REGION Network 13: HOPPER TEMPERATURE LINE 2
   RUNG wire#powerrail
      Contact( #HMI_INPUT_MAN_MODE )
      wire#w1
      "FC21020_FEEDER_SCALING"(DINT_INPUT_VALUE := 0, REAL_INPUT_VALUE := #"iHMI_Values Setpoints".HopperTempNominalLine2, DINT_TO_REAL := false, REAL_TRANSFORM_FOR_FEEDER := true, OUTPUT_VALUE_PLC => #oPLC_Aux.o_rHopperTempNominal_Line2, OUTPUT_VALUE_FEEDER => #ioPowder_Feeder_Unit_In_Out.Outputs."PF Setpoints, Warnings and Alarms".o_rHopperTempNominal_Line2)
   END_RUNG
   RUNG wire#w1
      Not()
      "FC21020_FEEDER_SCALING"(DINT_INPUT_VALUE := 0, REAL_INPUT_VALUE := #"iCNC_Values Setpoints".HopperTempNominalLine2, DINT_TO_REAL := false, REAL_TRANSFORM_FOR_FEEDER := true, OUTPUT_VALUE_PLC => #oPLC_Aux.o_rHopperTempNominal_Line2, OUTPUT_VALUE_FEEDER => #ioPowder_Feeder_Unit_In_Out.Outputs."PF Setpoints, Warnings and Alarms".o_rHopperTempNominal_Line2)
   END_RUNG
   // the same network as SCL:
   IF #HMI_INPUT_MAN_MODE THEN
       "FC21020_FEEDER_SCALING"(DINT_INPUT_VALUE := 0,
                               REAL_INPUT_VALUE := #"iHMI_Values Setpoints".HopperTempNominalLine2,
                               DINT_TO_REAL := false,
                               REAL_TRANSFORM_FOR_FEEDER := true,
                               OUTPUT_VALUE_PLC => #oPLC_Aux.o_rHopperTempNominal_Line2,
                               OUTPUT_VALUE_FEEDER => #ioPowder_Feeder_Unit_In_Out.Outputs."PF Setpoints, Warnings and Alarms".o_rHopperTempNominal_Line2);
   END_IF;
   IF NOT #HMI_INPUT_MAN_MODE THEN
       "FC21020_FEEDER_SCALING"(DINT_INPUT_VALUE := 0,
                               REAL_INPUT_VALUE := #"iCNC_Values Setpoints".HopperTempNominalLine2,
                               DINT_TO_REAL := false,
                               REAL_TRANSFORM_FOR_FEEDER := true,
                               OUTPUT_VALUE_PLC => #oPLC_Aux.o_rHopperTempNominal_Line2,
                               OUTPUT_VALUE_FEEDER => #ioPowder_Feeder_Unit_In_Out.Outputs."PF Setpoints, Warnings and Alarms".o_rHopperTempNominal_Line2);
   END_IF;
END_REGION

REGION Network 14: COMMUNICATION IS RUNNING
   RUNG wire#powerrail
      Contact( "M_ONE" )
      wire#w1
      Coil( #ioPowder_Feeder_Unit_In_Out.Outputs.o_fCommunicationOk_Line1 )
   END_RUNG
   RUNG wire#w1
      Coil( #ioPowder_Feeder_Unit_In_Out.Outputs.o_fCommunicationOk_Line2 )
   END_RUNG
   // the same network as SCL:
   #ioPowder_Feeder_Unit_In_Out.Outputs.o_fCommunicationOk_Line1 := "M_ONE";
   #ioPowder_Feeder_Unit_In_Out.Outputs.o_fCommunicationOk_Line2 := "M_ONE";
END_REGION

REGION Network 15: VOLUMETRIC MODE ON
   // Volumetric Mode On = 1 for Twin 150
   // Gravimetric Mode - n/a for Twin 150
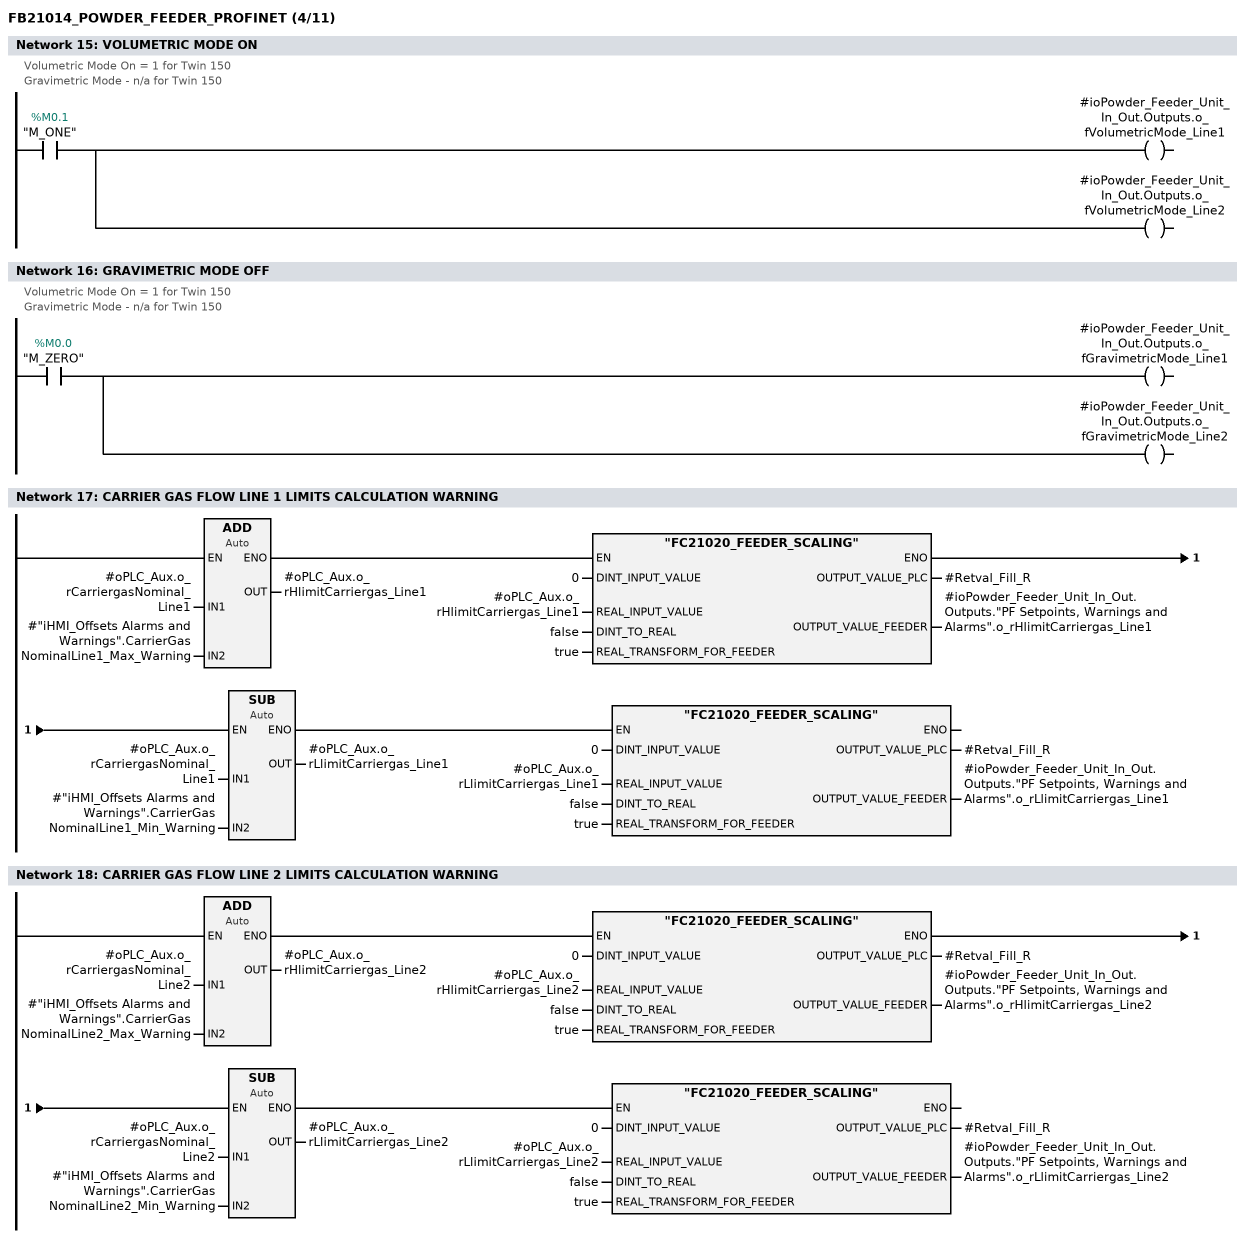
   RUNG wire#powerrail
      Contact( "M_ONE" )
      wire#w1
      Coil( #ioPowder_Feeder_Unit_In_Out.Outputs.o_fVolumetricMode_Line1 )
   END_RUNG
   RUNG wire#w1
      Coil( #ioPowder_Feeder_Unit_In_Out.Outputs.o_fVolumetricMode_Line2 )
   END_RUNG
   // the same network as SCL:
   #ioPowder_Feeder_Unit_In_Out.Outputs.o_fVolumetricMode_Line1 := "M_ONE";
   #ioPowder_Feeder_Unit_In_Out.Outputs.o_fVolumetricMode_Line2 := "M_ONE";
END_REGION

REGION Network 16: GRAVIMETRIC MODE OFF
   // Volumetric Mode On = 1 for Twin 150
   // Gravimetric Mode - n/a for Twin 150
   RUNG wire#powerrail
      Contact( "M_ZERO" )
      wire#w1
      Coil( #ioPowder_Feeder_Unit_In_Out.Outputs.o_fGravimetricMode_Line1 )
   END_RUNG
   RUNG wire#w1
      Coil( #ioPowder_Feeder_Unit_In_Out.Outputs.o_fGravimetricMode_Line2 )
   END_RUNG
   // the same network as SCL:
   #ioPowder_Feeder_Unit_In_Out.Outputs.o_fGravimetricMode_Line1 := "M_ZERO";
   #ioPowder_Feeder_Unit_In_Out.Outputs.o_fGravimetricMode_Line2 := "M_ZERO";
END_REGION

REGION Network 17: CARRIER GAS FLOW LINE 1 LIMITS CALCULATION WARNING
   RUNG wire#powerrail
      Add(in1 := #oPLC_Aux.o_rCarriergasNominal_Line1, in2 := #"iHMI_Offsets Alarms and Warnings".CarrierGasNominalLine1_Max_Warning, out => #oPLC_Aux.o_rHlimitCarriergas_Line1)
      "FC21020_FEEDER_SCALING"(DINT_INPUT_VALUE := 0, REAL_INPUT_VALUE := #oPLC_Aux.o_rHlimitCarriergas_Line1, DINT_TO_REAL := false, REAL_TRANSFORM_FOR_FEEDER := true, OUTPUT_VALUE_PLC => #Retval_Fill_R, OUTPUT_VALUE_FEEDER => #ioPowder_Feeder_Unit_In_Out.Outputs."PF Setpoints, Warnings and Alarms".o_rHlimitCarriergas_Line1)
      Sub(in1 := #oPLC_Aux.o_rCarriergasNominal_Line1, in2 := #"iHMI_Offsets Alarms and Warnings".CarrierGasNominalLine1_Min_Warning, out => #oPLC_Aux.o_rLlimitCarriergas_Line1)
      "FC21020_FEEDER_SCALING"(DINT_INPUT_VALUE := 0, REAL_INPUT_VALUE := #oPLC_Aux.o_rLlimitCarriergas_Line1, DINT_TO_REAL := false, REAL_TRANSFORM_FOR_FEEDER := true, OUTPUT_VALUE_PLC => #Retval_Fill_R, OUTPUT_VALUE_FEEDER => #ioPowder_Feeder_Unit_In_Out.Outputs."PF Setpoints, Warnings and Alarms".o_rLlimitCarriergas_Line1)
   END_RUNG
   // the same network as SCL:
   #oPLC_Aux.o_rHlimitCarriergas_Line1 := #oPLC_Aux.o_rCarriergasNominal_Line1 + #"iHMI_Offsets Alarms and Warnings".CarrierGasNominalLine1_Max_Warning;
   "FC21020_FEEDER_SCALING"(DINT_INPUT_VALUE := 0,
                           REAL_INPUT_VALUE := #oPLC_Aux.o_rHlimitCarriergas_Line1,
                           DINT_TO_REAL := false,
                           REAL_TRANSFORM_FOR_FEEDER := true,
                           OUTPUT_VALUE_PLC => #Retval_Fill_R,
                           OUTPUT_VALUE_FEEDER => #ioPowder_Feeder_Unit_In_Out.Outputs."PF Setpoints, Warnings and Alarms".o_rHlimitCarriergas_Line1,
                           ENO => #_w1);
   IF #_w1 THEN
       #oPLC_Aux.o_rLlimitCarriergas_Line1 := #oPLC_Aux.o_rCarriergasNominal_Line1 - #"iHMI_Offsets Alarms and Warnings".CarrierGasNominalLine1_Min_Warning;
       "FC21020_FEEDER_SCALING"(DINT_INPUT_VALUE := 0,
                               REAL_INPUT_VALUE := #oPLC_Aux.o_rLlimitCarriergas_Line1,
                               DINT_TO_REAL := false,
                               REAL_TRANSFORM_FOR_FEEDER := true,
                               OUTPUT_VALUE_PLC => #Retval_Fill_R,
                               OUTPUT_VALUE_FEEDER => #ioPowder_Feeder_Unit_In_Out.Outputs."PF Setpoints, Warnings and Alarms".o_rLlimitCarriergas_Line1);
   END_IF;
END_REGION

REGION Network 18: CARRIER GAS FLOW LINE 2 LIMITS CALCULATION WARNING
   RUNG wire#powerrail
      Add(in1 := #oPLC_Aux.o_rCarriergasNominal_Line2, in2 := #"iHMI_Offsets Alarms and Warnings".CarrierGasNominalLine2_Max_Warning, out => #oPLC_Aux.o_rHlimitCarriergas_Line2)
      "FC21020_FEEDER_SCALING"(DINT_INPUT_VALUE := 0, REAL_INPUT_VALUE := #oPLC_Aux.o_rHlimitCarriergas_Line2, DINT_TO_REAL := false, REAL_TRANSFORM_FOR_FEEDER := true, OUTPUT_VALUE_PLC => #Retval_Fill_R, OUTPUT_VALUE_FEEDER => #ioPowder_Feeder_Unit_In_Out.Outputs."PF Setpoints, Warnings and Alarms".o_rHlimitCarriergas_Line2)
      Sub(in1 := #oPLC_Aux.o_rCarriergasNominal_Line2, in2 := #"iHMI_Offsets Alarms and Warnings".CarrierGasNominalLine2_Min_Warning, out => #oPLC_Aux.o_rLlimitCarriergas_Line2)
      "FC21020_FEEDER_SCALING"(DINT_INPUT_VALUE := 0, REAL_INPUT_VALUE := #oPLC_Aux.o_rLlimitCarriergas_Line2, DINT_TO_REAL := false, REAL_TRANSFORM_FOR_FEEDER := true, OUTPUT_VALUE_PLC => #Retval_Fill_R, OUTPUT_VALUE_FEEDER => #ioPowder_Feeder_Unit_In_Out.Outputs."PF Setpoints, Warnings and Alarms".o_rLlimitCarriergas_Line2)
   END_RUNG
   // the same network as SCL:
   #oPLC_Aux.o_rHlimitCarriergas_Line2 := #oPLC_Aux.o_rCarriergasNominal_Line2 + #"iHMI_Offsets Alarms and Warnings".CarrierGasNominalLine2_Max_Warning;
   "FC21020_FEEDER_SCALING"(DINT_INPUT_VALUE := 0,
                           REAL_INPUT_VALUE := #oPLC_Aux.o_rHlimitCarriergas_Line2,
                           DINT_TO_REAL := false,
                           REAL_TRANSFORM_FOR_FEEDER := true,
                           OUTPUT_VALUE_PLC => #Retval_Fill_R,
                           OUTPUT_VALUE_FEEDER => #ioPowder_Feeder_Unit_In_Out.Outputs."PF Setpoints, Warnings and Alarms".o_rHlimitCarriergas_Line2,
                           ENO => #_w1);
   IF #_w1 THEN
       #oPLC_Aux.o_rLlimitCarriergas_Line2 := #oPLC_Aux.o_rCarriergasNominal_Line2 - #"iHMI_Offsets Alarms and Warnings".CarrierGasNominalLine2_Min_Warning;
       "FC21020_FEEDER_SCALING"(DINT_INPUT_VALUE := 0,
                               REAL_INPUT_VALUE := #oPLC_Aux.o_rLlimitCarriergas_Line2,
                               DINT_TO_REAL := false,
                               REAL_TRANSFORM_FOR_FEEDER := true,
                               OUTPUT_VALUE_PLC => #Retval_Fill_R,
                               OUTPUT_VALUE_FEEDER => #ioPowder_Feeder_Unit_In_Out.Outputs."PF Setpoints, Warnings and Alarms".o_rLlimitCarriergas_Line2);
   END_IF;
END_REGION

REGION Network 19: CARRIER GAS FLOW LINE 1 LIMITS CALCULATION ALARM
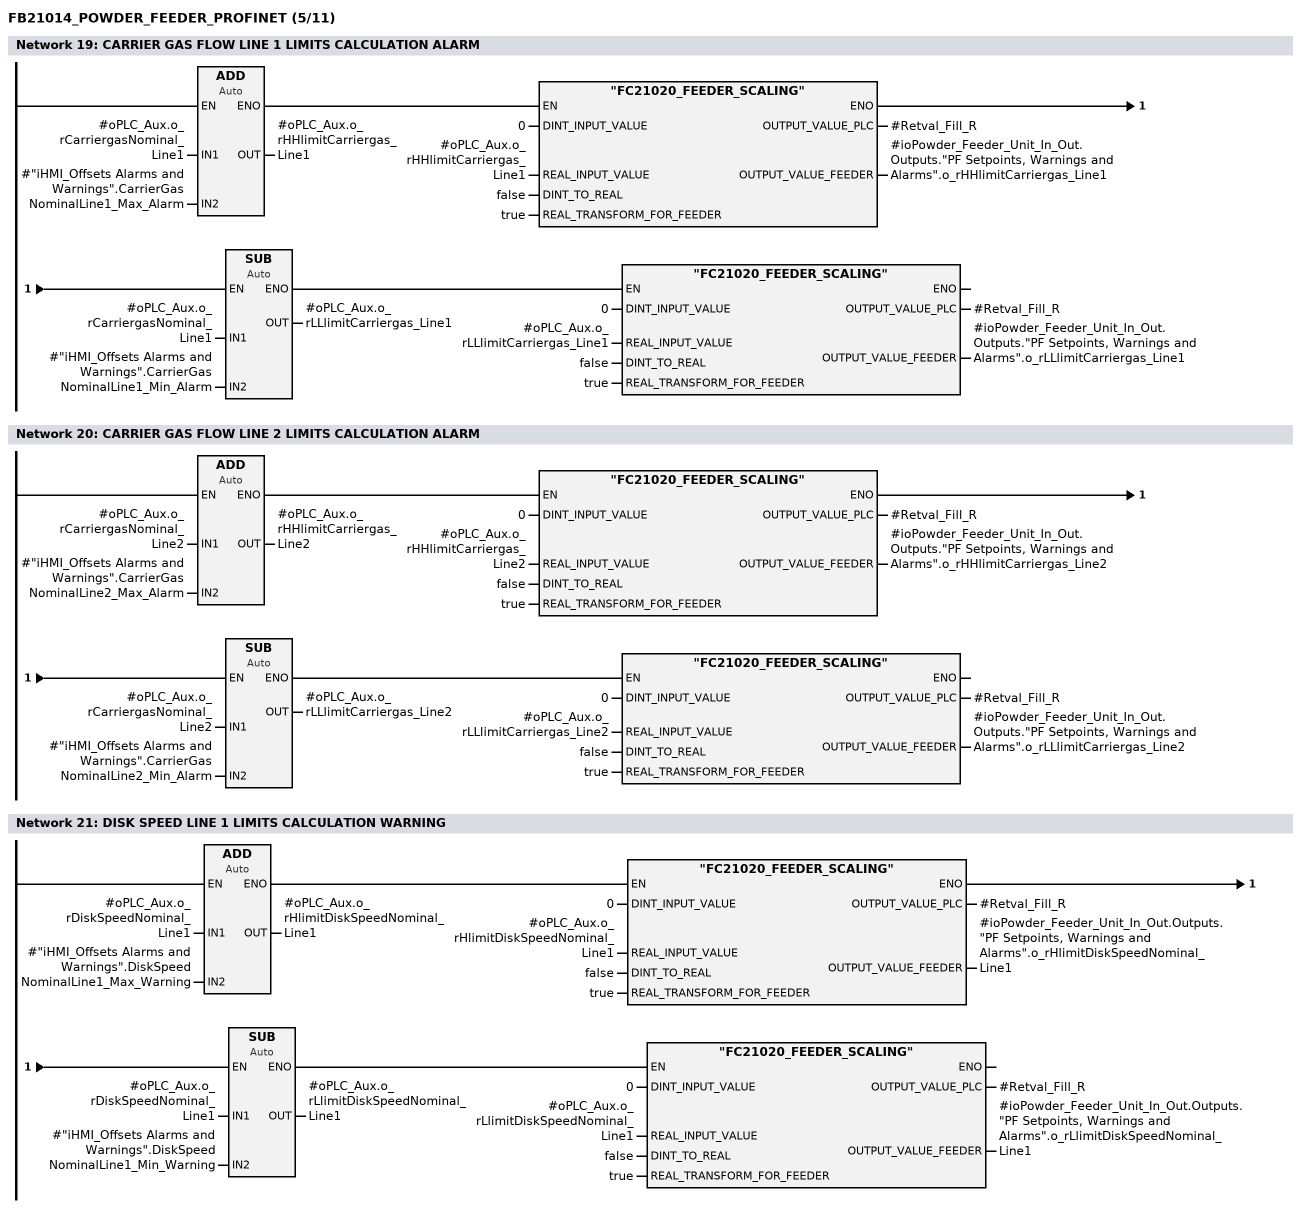
   RUNG wire#powerrail
      Add(in1 := #oPLC_Aux.o_rCarriergasNominal_Line1, in2 := #"iHMI_Offsets Alarms and Warnings".CarrierGasNominalLine1_Max_Alarm, out => #oPLC_Aux.o_rHHlimitCarriergas_Line1)
      "FC21020_FEEDER_SCALING"(DINT_INPUT_VALUE := 0, REAL_INPUT_VALUE := #oPLC_Aux.o_rHHlimitCarriergas_Line1, DINT_TO_REAL := false, REAL_TRANSFORM_FOR_FEEDER := true, OUTPUT_VALUE_PLC => #Retval_Fill_R, OUTPUT_VALUE_FEEDER => #ioPowder_Feeder_Unit_In_Out.Outputs."PF Setpoints, Warnings and Alarms".o_rHHlimitCarriergas_Line1)
      Sub(in1 := #oPLC_Aux.o_rCarriergasNominal_Line1, in2 := #"iHMI_Offsets Alarms and Warnings".CarrierGasNominalLine1_Min_Alarm, out => #oPLC_Aux.o_rLLlimitCarriergas_Line1)
      "FC21020_FEEDER_SCALING"(DINT_INPUT_VALUE := 0, REAL_INPUT_VALUE := #oPLC_Aux.o_rLLlimitCarriergas_Line1, DINT_TO_REAL := false, REAL_TRANSFORM_FOR_FEEDER := true, OUTPUT_VALUE_PLC => #Retval_Fill_R, OUTPUT_VALUE_FEEDER => #ioPowder_Feeder_Unit_In_Out.Outputs."PF Setpoints, Warnings and Alarms".o_rLLlimitCarriergas_Line1)
   END_RUNG
   // the same network as SCL:
   #oPLC_Aux.o_rHHlimitCarriergas_Line1 := #oPLC_Aux.o_rCarriergasNominal_Line1 + #"iHMI_Offsets Alarms and Warnings".CarrierGasNominalLine1_Max_Alarm;
   "FC21020_FEEDER_SCALING"(DINT_INPUT_VALUE := 0,
                           REAL_INPUT_VALUE := #oPLC_Aux.o_rHHlimitCarriergas_Line1,
                           DINT_TO_REAL := false,
                           REAL_TRANSFORM_FOR_FEEDER := true,
                           OUTPUT_VALUE_PLC => #Retval_Fill_R,
                           OUTPUT_VALUE_FEEDER => #ioPowder_Feeder_Unit_In_Out.Outputs."PF Setpoints, Warnings and Alarms".o_rHHlimitCarriergas_Line1,
                           ENO => #_w1);
   IF #_w1 THEN
       #oPLC_Aux.o_rLLlimitCarriergas_Line1 := #oPLC_Aux.o_rCarriergasNominal_Line1 - #"iHMI_Offsets Alarms and Warnings".CarrierGasNominalLine1_Min_Alarm;
       "FC21020_FEEDER_SCALING"(DINT_INPUT_VALUE := 0,
                               REAL_INPUT_VALUE := #oPLC_Aux.o_rLLlimitCarriergas_Line1,
                               DINT_TO_REAL := false,
                               REAL_TRANSFORM_FOR_FEEDER := true,
                               OUTPUT_VALUE_PLC => #Retval_Fill_R,
                               OUTPUT_VALUE_FEEDER => #ioPowder_Feeder_Unit_In_Out.Outputs."PF Setpoints, Warnings and Alarms".o_rLLlimitCarriergas_Line1);
   END_IF;
END_REGION

REGION Network 20: CARRIER GAS FLOW LINE 2 LIMITS CALCULATION ALARM
   RUNG wire#powerrail
      Add(in1 := #oPLC_Aux.o_rCarriergasNominal_Line2, in2 := #"iHMI_Offsets Alarms and Warnings".CarrierGasNominalLine2_Max_Alarm, out => #oPLC_Aux.o_rHHlimitCarriergas_Line2)
      "FC21020_FEEDER_SCALING"(DINT_INPUT_VALUE := 0, REAL_INPUT_VALUE := #oPLC_Aux.o_rHHlimitCarriergas_Line2, DINT_TO_REAL := false, REAL_TRANSFORM_FOR_FEEDER := true, OUTPUT_VALUE_PLC => #Retval_Fill_R, OUTPUT_VALUE_FEEDER => #ioPowder_Feeder_Unit_In_Out.Outputs."PF Setpoints, Warnings and Alarms".o_rHHlimitCarriergas_Line2)
      Sub(in1 := #oPLC_Aux.o_rCarriergasNominal_Line2, in2 := #"iHMI_Offsets Alarms and Warnings".CarrierGasNominalLine2_Min_Alarm, out => #oPLC_Aux.o_rLLlimitCarriergas_Line2)
      "FC21020_FEEDER_SCALING"(DINT_INPUT_VALUE := 0, REAL_INPUT_VALUE := #oPLC_Aux.o_rLLlimitCarriergas_Line2, DINT_TO_REAL := false, REAL_TRANSFORM_FOR_FEEDER := true, OUTPUT_VALUE_PLC => #Retval_Fill_R, OUTPUT_VALUE_FEEDER => #ioPowder_Feeder_Unit_In_Out.Outputs."PF Setpoints, Warnings and Alarms".o_rLLlimitCarriergas_Line2)
   END_RUNG
   // the same network as SCL:
   #oPLC_Aux.o_rHHlimitCarriergas_Line2 := #oPLC_Aux.o_rCarriergasNominal_Line2 + #"iHMI_Offsets Alarms and Warnings".CarrierGasNominalLine2_Max_Alarm;
   "FC21020_FEEDER_SCALING"(DINT_INPUT_VALUE := 0,
                           REAL_INPUT_VALUE := #oPLC_Aux.o_rHHlimitCarriergas_Line2,
                           DINT_TO_REAL := false,
                           REAL_TRANSFORM_FOR_FEEDER := true,
                           OUTPUT_VALUE_PLC => #Retval_Fill_R,
                           OUTPUT_VALUE_FEEDER => #ioPowder_Feeder_Unit_In_Out.Outputs."PF Setpoints, Warnings and Alarms".o_rHHlimitCarriergas_Line2,
                           ENO => #_w1);
   IF #_w1 THEN
       #oPLC_Aux.o_rLLlimitCarriergas_Line2 := #oPLC_Aux.o_rCarriergasNominal_Line2 - #"iHMI_Offsets Alarms and Warnings".CarrierGasNominalLine2_Min_Alarm;
       "FC21020_FEEDER_SCALING"(DINT_INPUT_VALUE := 0,
                               REAL_INPUT_VALUE := #oPLC_Aux.o_rLLlimitCarriergas_Line2,
                               DINT_TO_REAL := false,
                               REAL_TRANSFORM_FOR_FEEDER := true,
                               OUTPUT_VALUE_PLC => #Retval_Fill_R,
                               OUTPUT_VALUE_FEEDER => #ioPowder_Feeder_Unit_In_Out.Outputs."PF Setpoints, Warnings and Alarms".o_rLLlimitCarriergas_Line2);
   END_IF;
END_REGION

REGION Network 21: DISK SPEED LINE 1 LIMITS CALCULATION WARNING
   RUNG wire#powerrail
      Add(in1 := #oPLC_Aux.o_rDiskSpeedNominal_Line1, in2 := #"iHMI_Offsets Alarms and Warnings".DiskSpeedNominalLine1_Max_Warning, out => #oPLC_Aux.o_rHlimitDiskSpeedNominal_Line1)
      "FC21020_FEEDER_SCALING"(DINT_INPUT_VALUE := 0, REAL_INPUT_VALUE := #oPLC_Aux.o_rHlimitDiskSpeedNominal_Line1, DINT_TO_REAL := false, REAL_TRANSFORM_FOR_FEEDER := true, OUTPUT_VALUE_PLC => #Retval_Fill_R, OUTPUT_VALUE_FEEDER => #ioPowder_Feeder_Unit_In_Out.Outputs."PF Setpoints, Warnings and Alarms".o_rHlimitDiskSpeedNominal_Line1)
      Sub(in1 := #oPLC_Aux.o_rDiskSpeedNominal_Line1, in2 := #"iHMI_Offsets Alarms and Warnings".DiskSpeedNominalLine1_Min_Warning, out => #oPLC_Aux.o_rLlimitDiskSpeedNominal_Line1)
      "FC21020_FEEDER_SCALING"(DINT_INPUT_VALUE := 0, REAL_INPUT_VALUE := #oPLC_Aux.o_rLlimitDiskSpeedNominal_Line1, DINT_TO_REAL := false, REAL_TRANSFORM_FOR_FEEDER := true, OUTPUT_VALUE_PLC => #Retval_Fill_R, OUTPUT_VALUE_FEEDER => #ioPowder_Feeder_Unit_In_Out.Outputs."PF Setpoints, Warnings and Alarms".o_rLlimitDiskSpeedNominal_Line1)
   END_RUNG
   // the same network as SCL:
   #oPLC_Aux.o_rHlimitDiskSpeedNominal_Line1 := #oPLC_Aux.o_rDiskSpeedNominal_Line1 + #"iHMI_Offsets Alarms and Warnings".DiskSpeedNominalLine1_Max_Warning;
   "FC21020_FEEDER_SCALING"(DINT_INPUT_VALUE := 0,
                           REAL_INPUT_VALUE := #oPLC_Aux.o_rHlimitDiskSpeedNominal_Line1,
                           DINT_TO_REAL := false,
                           REAL_TRANSFORM_FOR_FEEDER := true,
                           OUTPUT_VALUE_PLC => #Retval_Fill_R,
                           OUTPUT_VALUE_FEEDER => #ioPowder_Feeder_Unit_In_Out.Outputs."PF Setpoints, Warnings and Alarms".o_rHlimitDiskSpeedNominal_Line1,
                           ENO => #_w1);
   IF #_w1 THEN
       #oPLC_Aux.o_rLlimitDiskSpeedNominal_Line1 := #oPLC_Aux.o_rDiskSpeedNominal_Line1 - #"iHMI_Offsets Alarms and Warnings".DiskSpeedNominalLine1_Min_Warning;
       "FC21020_FEEDER_SCALING"(DINT_INPUT_VALUE := 0,
                               REAL_INPUT_VALUE := #oPLC_Aux.o_rLlimitDiskSpeedNominal_Line1,
                               DINT_TO_REAL := false,
                               REAL_TRANSFORM_FOR_FEEDER := true,
                               OUTPUT_VALUE_PLC => #Retval_Fill_R,
                               OUTPUT_VALUE_FEEDER => #ioPowder_Feeder_Unit_In_Out.Outputs."PF Setpoints, Warnings and Alarms".o_rLlimitDiskSpeedNominal_Line1);
   END_IF;
END_REGION

REGION Network 22: DISK SPEED LINE 2 LIMITS CALCULATION WARNING
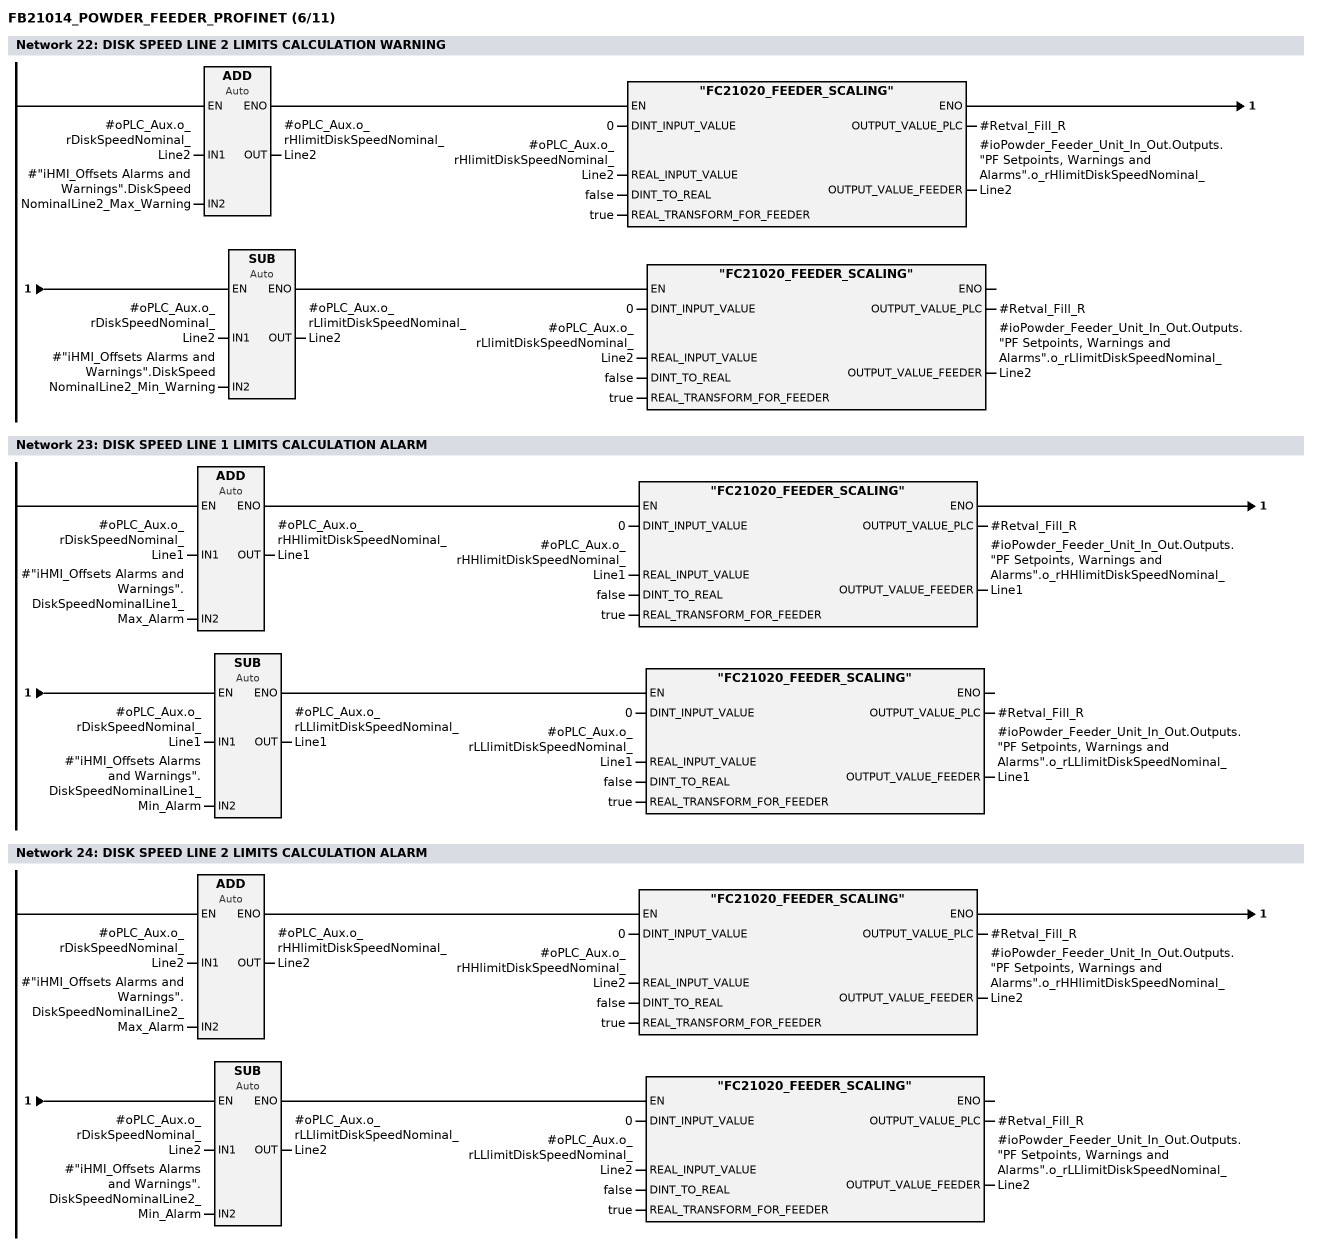
   RUNG wire#powerrail
      Add(in1 := #oPLC_Aux.o_rDiskSpeedNominal_Line2, in2 := #"iHMI_Offsets Alarms and Warnings".DiskSpeedNominalLine2_Max_Warning, out => #oPLC_Aux.o_rHlimitDiskSpeedNominal_Line2)
      "FC21020_FEEDER_SCALING"(DINT_INPUT_VALUE := 0, REAL_INPUT_VALUE := #oPLC_Aux.o_rHlimitDiskSpeedNominal_Line2, DINT_TO_REAL := false, REAL_TRANSFORM_FOR_FEEDER := true, OUTPUT_VALUE_PLC => #Retval_Fill_R, OUTPUT_VALUE_FEEDER => #ioPowder_Feeder_Unit_In_Out.Outputs."PF Setpoints, Warnings and Alarms".o_rHlimitDiskSpeedNominal_Line2)
      Sub(in1 := #oPLC_Aux.o_rDiskSpeedNominal_Line2, in2 := #"iHMI_Offsets Alarms and Warnings".DiskSpeedNominalLine2_Min_Warning, out => #oPLC_Aux.o_rLlimitDiskSpeedNominal_Line2)
      "FC21020_FEEDER_SCALING"(DINT_INPUT_VALUE := 0, REAL_INPUT_VALUE := #oPLC_Aux.o_rLlimitDiskSpeedNominal_Line2, DINT_TO_REAL := false, REAL_TRANSFORM_FOR_FEEDER := true, OUTPUT_VALUE_PLC => #Retval_Fill_R, OUTPUT_VALUE_FEEDER => #ioPowder_Feeder_Unit_In_Out.Outputs."PF Setpoints, Warnings and Alarms".o_rLlimitDiskSpeedNominal_Line2)
   END_RUNG
   // the same network as SCL:
   #oPLC_Aux.o_rHlimitDiskSpeedNominal_Line2 := #oPLC_Aux.o_rDiskSpeedNominal_Line2 + #"iHMI_Offsets Alarms and Warnings".DiskSpeedNominalLine2_Max_Warning;
   "FC21020_FEEDER_SCALING"(DINT_INPUT_VALUE := 0,
                           REAL_INPUT_VALUE := #oPLC_Aux.o_rHlimitDiskSpeedNominal_Line2,
                           DINT_TO_REAL := false,
                           REAL_TRANSFORM_FOR_FEEDER := true,
                           OUTPUT_VALUE_PLC => #Retval_Fill_R,
                           OUTPUT_VALUE_FEEDER => #ioPowder_Feeder_Unit_In_Out.Outputs."PF Setpoints, Warnings and Alarms".o_rHlimitDiskSpeedNominal_Line2,
                           ENO => #_w1);
   IF #_w1 THEN
       #oPLC_Aux.o_rLlimitDiskSpeedNominal_Line2 := #oPLC_Aux.o_rDiskSpeedNominal_Line2 - #"iHMI_Offsets Alarms and Warnings".DiskSpeedNominalLine2_Min_Warning;
       "FC21020_FEEDER_SCALING"(DINT_INPUT_VALUE := 0,
                               REAL_INPUT_VALUE := #oPLC_Aux.o_rLlimitDiskSpeedNominal_Line2,
                               DINT_TO_REAL := false,
                               REAL_TRANSFORM_FOR_FEEDER := true,
                               OUTPUT_VALUE_PLC => #Retval_Fill_R,
                               OUTPUT_VALUE_FEEDER => #ioPowder_Feeder_Unit_In_Out.Outputs."PF Setpoints, Warnings and Alarms".o_rLlimitDiskSpeedNominal_Line2);
   END_IF;
END_REGION

REGION Network 23: DISK SPEED LINE 1 LIMITS CALCULATION ALARM
   RUNG wire#powerrail
      Add(in1 := #oPLC_Aux.o_rDiskSpeedNominal_Line1, in2 := #"iHMI_Offsets Alarms and Warnings".DiskSpeedNominalLine1_Max_Alarm, out => #oPLC_Aux.o_rHHlimitDiskSpeedNominal_Line1)
      "FC21020_FEEDER_SCALING"(DINT_INPUT_VALUE := 0, REAL_INPUT_VALUE := #oPLC_Aux.o_rHHlimitDiskSpeedNominal_Line1, DINT_TO_REAL := false, REAL_TRANSFORM_FOR_FEEDER := true, OUTPUT_VALUE_PLC => #Retval_Fill_R, OUTPUT_VALUE_FEEDER => #ioPowder_Feeder_Unit_In_Out.Outputs."PF Setpoints, Warnings and Alarms".o_rHHlimitDiskSpeedNominal_Line1)
      Sub(in1 := #oPLC_Aux.o_rDiskSpeedNominal_Line1, in2 := #"iHMI_Offsets Alarms and Warnings".DiskSpeedNominalLine1_Min_Alarm, out => #oPLC_Aux.o_rLLlimitDiskSpeedNominal_Line1)
      "FC21020_FEEDER_SCALING"(DINT_INPUT_VALUE := 0, REAL_INPUT_VALUE := #oPLC_Aux.o_rLLlimitDiskSpeedNominal_Line1, DINT_TO_REAL := false, REAL_TRANSFORM_FOR_FEEDER := true, OUTPUT_VALUE_PLC => #Retval_Fill_R, OUTPUT_VALUE_FEEDER => #ioPowder_Feeder_Unit_In_Out.Outputs."PF Setpoints, Warnings and Alarms".o_rLLlimitDiskSpeedNominal_Line1)
   END_RUNG
   // the same network as SCL:
   #oPLC_Aux.o_rHHlimitDiskSpeedNominal_Line1 := #oPLC_Aux.o_rDiskSpeedNominal_Line1 + #"iHMI_Offsets Alarms and Warnings".DiskSpeedNominalLine1_Max_Alarm;
   "FC21020_FEEDER_SCALING"(DINT_INPUT_VALUE := 0,
                           REAL_INPUT_VALUE := #oPLC_Aux.o_rHHlimitDiskSpeedNominal_Line1,
                           DINT_TO_REAL := false,
                           REAL_TRANSFORM_FOR_FEEDER := true,
                           OUTPUT_VALUE_PLC => #Retval_Fill_R,
                           OUTPUT_VALUE_FEEDER => #ioPowder_Feeder_Unit_In_Out.Outputs."PF Setpoints, Warnings and Alarms".o_rHHlimitDiskSpeedNominal_Line1,
                           ENO => #_w1);
   IF #_w1 THEN
       #oPLC_Aux.o_rLLlimitDiskSpeedNominal_Line1 := #oPLC_Aux.o_rDiskSpeedNominal_Line1 - #"iHMI_Offsets Alarms and Warnings".DiskSpeedNominalLine1_Min_Alarm;
       "FC21020_FEEDER_SCALING"(DINT_INPUT_VALUE := 0,
                               REAL_INPUT_VALUE := #oPLC_Aux.o_rLLlimitDiskSpeedNominal_Line1,
                               DINT_TO_REAL := false,
                               REAL_TRANSFORM_FOR_FEEDER := true,
                               OUTPUT_VALUE_PLC => #Retval_Fill_R,
                               OUTPUT_VALUE_FEEDER => #ioPowder_Feeder_Unit_In_Out.Outputs."PF Setpoints, Warnings and Alarms".o_rLLlimitDiskSpeedNominal_Line1);
   END_IF;
END_REGION

REGION Network 24: DISK SPEED LINE 2 LIMITS CALCULATION ALARM
   RUNG wire#powerrail
      Add(in1 := #oPLC_Aux.o_rDiskSpeedNominal_Line2, in2 := #"iHMI_Offsets Alarms and Warnings".DiskSpeedNominalLine2_Max_Alarm, out => #oPLC_Aux.o_rHHlimitDiskSpeedNominal_Line2)
      "FC21020_FEEDER_SCALING"(DINT_INPUT_VALUE := 0, REAL_INPUT_VALUE := #oPLC_Aux.o_rHHlimitDiskSpeedNominal_Line2, DINT_TO_REAL := false, REAL_TRANSFORM_FOR_FEEDER := true, OUTPUT_VALUE_PLC => #Retval_Fill_R, OUTPUT_VALUE_FEEDER => #ioPowder_Feeder_Unit_In_Out.Outputs."PF Setpoints, Warnings and Alarms".o_rHHlimitDiskSpeedNominal_Line2)
      Sub(in1 := #oPLC_Aux.o_rDiskSpeedNominal_Line2, in2 := #"iHMI_Offsets Alarms and Warnings".DiskSpeedNominalLine2_Min_Alarm, out => #oPLC_Aux.o_rLLlimitDiskSpeedNominal_Line2)
      "FC21020_FEEDER_SCALING"(DINT_INPUT_VALUE := 0, REAL_INPUT_VALUE := #oPLC_Aux.o_rLLlimitDiskSpeedNominal_Line2, DINT_TO_REAL := false, REAL_TRANSFORM_FOR_FEEDER := true, OUTPUT_VALUE_PLC => #Retval_Fill_R, OUTPUT_VALUE_FEEDER => #ioPowder_Feeder_Unit_In_Out.Outputs."PF Setpoints, Warnings and Alarms".o_rLLlimitDiskSpeedNominal_Line2)
   END_RUNG
   // the same network as SCL:
   #oPLC_Aux.o_rHHlimitDiskSpeedNominal_Line2 := #oPLC_Aux.o_rDiskSpeedNominal_Line2 + #"iHMI_Offsets Alarms and Warnings".DiskSpeedNominalLine2_Max_Alarm;
   "FC21020_FEEDER_SCALING"(DINT_INPUT_VALUE := 0,
                           REAL_INPUT_VALUE := #oPLC_Aux.o_rHHlimitDiskSpeedNominal_Line2,
                           DINT_TO_REAL := false,
                           REAL_TRANSFORM_FOR_FEEDER := true,
                           OUTPUT_VALUE_PLC => #Retval_Fill_R,
                           OUTPUT_VALUE_FEEDER => #ioPowder_Feeder_Unit_In_Out.Outputs."PF Setpoints, Warnings and Alarms".o_rHHlimitDiskSpeedNominal_Line2,
                           ENO => #_w1);
   IF #_w1 THEN
       #oPLC_Aux.o_rLLlimitDiskSpeedNominal_Line2 := #oPLC_Aux.o_rDiskSpeedNominal_Line2 - #"iHMI_Offsets Alarms and Warnings".DiskSpeedNominalLine2_Min_Alarm;
       "FC21020_FEEDER_SCALING"(DINT_INPUT_VALUE := 0,
                               REAL_INPUT_VALUE := #oPLC_Aux.o_rLLlimitDiskSpeedNominal_Line2,
                               DINT_TO_REAL := false,
                               REAL_TRANSFORM_FOR_FEEDER := true,
                               OUTPUT_VALUE_PLC => #Retval_Fill_R,
                               OUTPUT_VALUE_FEEDER => #ioPowder_Feeder_Unit_In_Out.Outputs."PF Setpoints, Warnings and Alarms".o_rLLlimitDiskSpeedNominal_Line2);
   END_IF;
END_REGION

REGION Network 25: STIRRER SPEED LINE 1 LIMITS CALCULATION WARNING
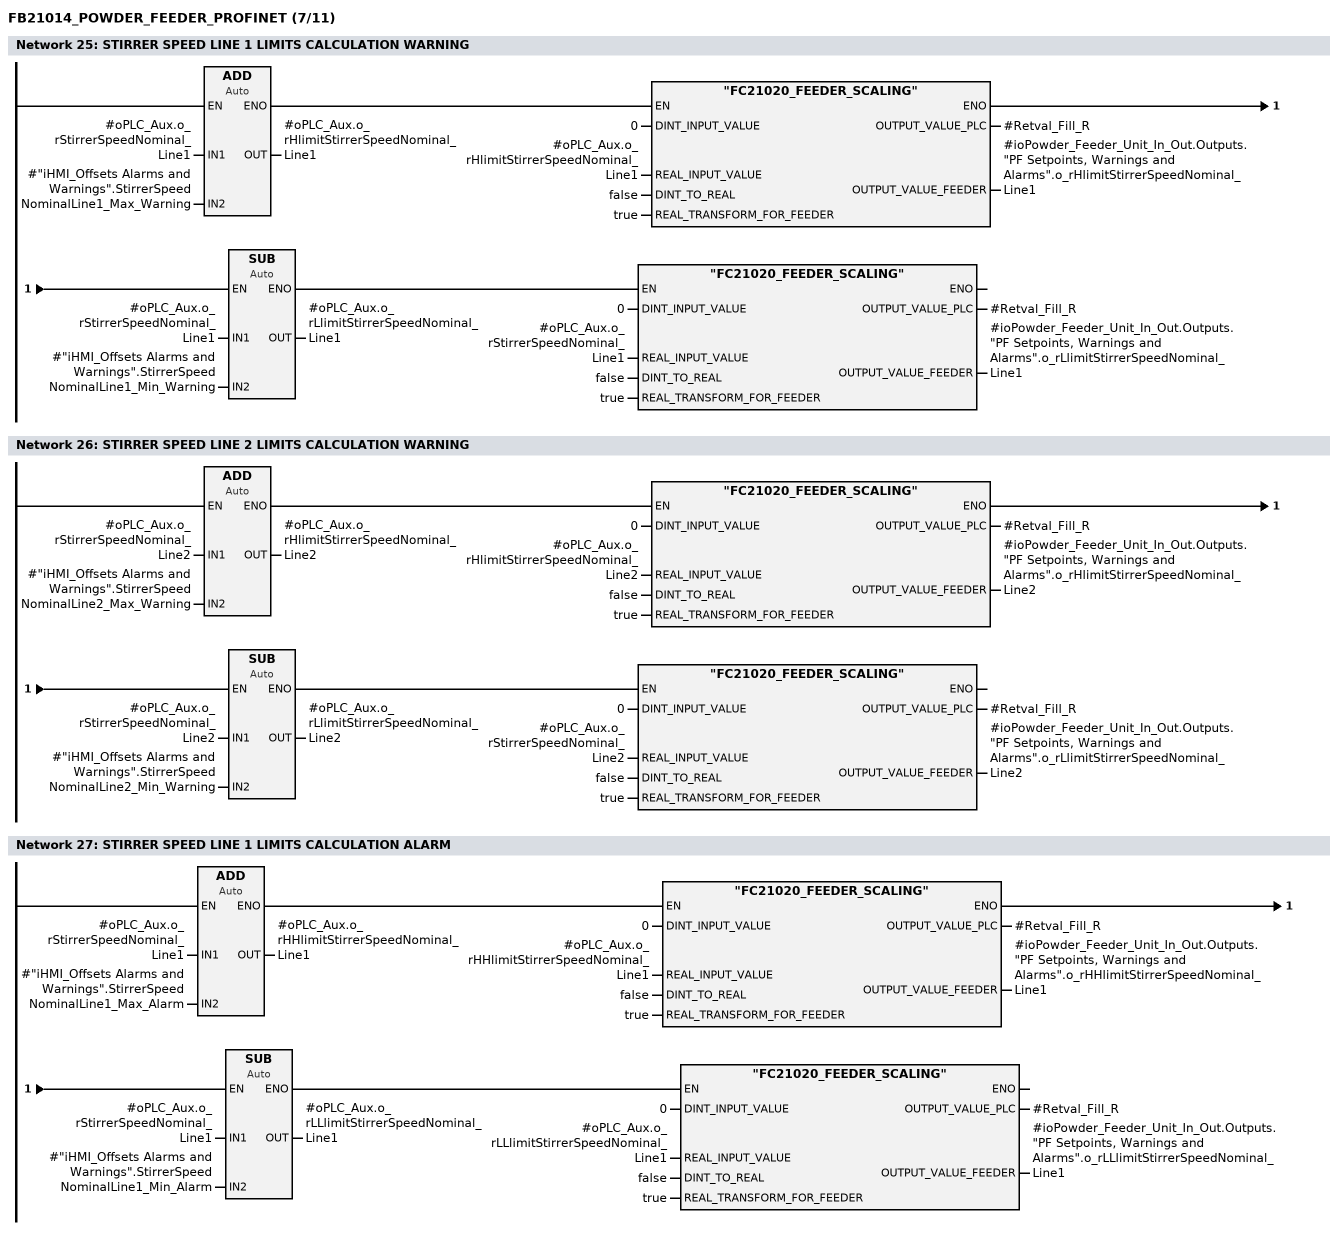
   RUNG wire#powerrail
      Add(in1 := #oPLC_Aux.o_rStirrerSpeedNominal_Line1, in2 := #"iHMI_Offsets Alarms and Warnings".StirrerSpeedNominalLine1_Max_Warning, out => #oPLC_Aux.o_rHlimitStirrerSpeedNominal_Line1)
      "FC21020_FEEDER_SCALING"(DINT_INPUT_VALUE := 0, REAL_INPUT_VALUE := #oPLC_Aux.o_rHlimitStirrerSpeedNominal_Line1, DINT_TO_REAL := false, REAL_TRANSFORM_FOR_FEEDER := true, OUTPUT_VALUE_PLC => #Retval_Fill_R, OUTPUT_VALUE_FEEDER => #ioPowder_Feeder_Unit_In_Out.Outputs."PF Setpoints, Warnings and Alarms".o_rHlimitStirrerSpeedNominal_Line1)
      Sub(in1 := #oPLC_Aux.o_rStirrerSpeedNominal_Line1, in2 := #"iHMI_Offsets Alarms and Warnings".StirrerSpeedNominalLine1_Min_Warning, out => #oPLC_Aux.o_rLlimitStirrerSpeedNominal_Line1)
      "FC21020_FEEDER_SCALING"(DINT_INPUT_VALUE := 0, REAL_INPUT_VALUE := #oPLC_Aux.o_rStirrerSpeedNominal_Line1, DINT_TO_REAL := false, REAL_TRANSFORM_FOR_FEEDER := true, OUTPUT_VALUE_PLC => #Retval_Fill_R, OUTPUT_VALUE_FEEDER => #ioPowder_Feeder_Unit_In_Out.Outputs."PF Setpoints, Warnings and Alarms".o_rLlimitStirrerSpeedNominal_Line1)
   END_RUNG
   // the same network as SCL:
   #oPLC_Aux.o_rHlimitStirrerSpeedNominal_Line1 := #oPLC_Aux.o_rStirrerSpeedNominal_Line1 + #"iHMI_Offsets Alarms and Warnings".StirrerSpeedNominalLine1_Max_Warning;
   "FC21020_FEEDER_SCALING"(DINT_INPUT_VALUE := 0,
                           REAL_INPUT_VALUE := #oPLC_Aux.o_rHlimitStirrerSpeedNominal_Line1,
                           DINT_TO_REAL := false,
                           REAL_TRANSFORM_FOR_FEEDER := true,
                           OUTPUT_VALUE_PLC => #Retval_Fill_R,
                           OUTPUT_VALUE_FEEDER => #ioPowder_Feeder_Unit_In_Out.Outputs."PF Setpoints, Warnings and Alarms".o_rHlimitStirrerSpeedNominal_Line1,
                           ENO => #_w1);
   IF #_w1 THEN
       #oPLC_Aux.o_rLlimitStirrerSpeedNominal_Line1 := #oPLC_Aux.o_rStirrerSpeedNominal_Line1 - #"iHMI_Offsets Alarms and Warnings".StirrerSpeedNominalLine1_Min_Warning;
       "FC21020_FEEDER_SCALING"(DINT_INPUT_VALUE := 0,
                               REAL_INPUT_VALUE := #oPLC_Aux.o_rStirrerSpeedNominal_Line1,
                               DINT_TO_REAL := false,
                               REAL_TRANSFORM_FOR_FEEDER := true,
                               OUTPUT_VALUE_PLC => #Retval_Fill_R,
                               OUTPUT_VALUE_FEEDER => #ioPowder_Feeder_Unit_In_Out.Outputs."PF Setpoints, Warnings and Alarms".o_rLlimitStirrerSpeedNominal_Line1);
   END_IF;
END_REGION

REGION Network 26: STIRRER SPEED LINE 2 LIMITS CALCULATION WARNING
   RUNG wire#powerrail
      Add(in1 := #oPLC_Aux.o_rStirrerSpeedNominal_Line2, in2 := #"iHMI_Offsets Alarms and Warnings".StirrerSpeedNominalLine2_Max_Warning, out => #oPLC_Aux.o_rHlimitStirrerSpeedNominal_Line2)
      "FC21020_FEEDER_SCALING"(DINT_INPUT_VALUE := 0, REAL_INPUT_VALUE := #oPLC_Aux.o_rHlimitStirrerSpeedNominal_Line2, DINT_TO_REAL := false, REAL_TRANSFORM_FOR_FEEDER := true, OUTPUT_VALUE_PLC => #Retval_Fill_R, OUTPUT_VALUE_FEEDER => #ioPowder_Feeder_Unit_In_Out.Outputs."PF Setpoints, Warnings and Alarms".o_rHlimitStirrerSpeedNominal_Line2)
      Sub(in1 := #oPLC_Aux.o_rStirrerSpeedNominal_Line2, in2 := #"iHMI_Offsets Alarms and Warnings".StirrerSpeedNominalLine2_Min_Warning, out => #oPLC_Aux.o_rLlimitStirrerSpeedNominal_Line2)
      "FC21020_FEEDER_SCALING"(DINT_INPUT_VALUE := 0, REAL_INPUT_VALUE := #oPLC_Aux.o_rStirrerSpeedNominal_Line2, DINT_TO_REAL := false, REAL_TRANSFORM_FOR_FEEDER := true, OUTPUT_VALUE_PLC => #Retval_Fill_R, OUTPUT_VALUE_FEEDER => #ioPowder_Feeder_Unit_In_Out.Outputs."PF Setpoints, Warnings and Alarms".o_rLlimitStirrerSpeedNominal_Line2)
   END_RUNG
   // the same network as SCL:
   #oPLC_Aux.o_rHlimitStirrerSpeedNominal_Line2 := #oPLC_Aux.o_rStirrerSpeedNominal_Line2 + #"iHMI_Offsets Alarms and Warnings".StirrerSpeedNominalLine2_Max_Warning;
   "FC21020_FEEDER_SCALING"(DINT_INPUT_VALUE := 0,
                           REAL_INPUT_VALUE := #oPLC_Aux.o_rHlimitStirrerSpeedNominal_Line2,
                           DINT_TO_REAL := false,
                           REAL_TRANSFORM_FOR_FEEDER := true,
                           OUTPUT_VALUE_PLC => #Retval_Fill_R,
                           OUTPUT_VALUE_FEEDER => #ioPowder_Feeder_Unit_In_Out.Outputs."PF Setpoints, Warnings and Alarms".o_rHlimitStirrerSpeedNominal_Line2,
                           ENO => #_w1);
   IF #_w1 THEN
       #oPLC_Aux.o_rLlimitStirrerSpeedNominal_Line2 := #oPLC_Aux.o_rStirrerSpeedNominal_Line2 - #"iHMI_Offsets Alarms and Warnings".StirrerSpeedNominalLine2_Min_Warning;
       "FC21020_FEEDER_SCALING"(DINT_INPUT_VALUE := 0,
                               REAL_INPUT_VALUE := #oPLC_Aux.o_rStirrerSpeedNominal_Line2,
                               DINT_TO_REAL := false,
                               REAL_TRANSFORM_FOR_FEEDER := true,
                               OUTPUT_VALUE_PLC => #Retval_Fill_R,
                               OUTPUT_VALUE_FEEDER => #ioPowder_Feeder_Unit_In_Out.Outputs."PF Setpoints, Warnings and Alarms".o_rLlimitStirrerSpeedNominal_Line2);
   END_IF;
END_REGION

REGION Network 27: STIRRER SPEED LINE 1 LIMITS CALCULATION ALARM
   RUNG wire#powerrail
      Add(in1 := #oPLC_Aux.o_rStirrerSpeedNominal_Line1, in2 := #"iHMI_Offsets Alarms and Warnings".StirrerSpeedNominalLine1_Max_Alarm, out => #oPLC_Aux.o_rHHlimitStirrerSpeedNominal_Line1)
      "FC21020_FEEDER_SCALING"(DINT_INPUT_VALUE := 0, REAL_INPUT_VALUE := #oPLC_Aux.o_rHHlimitStirrerSpeedNominal_Line1, DINT_TO_REAL := false, REAL_TRANSFORM_FOR_FEEDER := true, OUTPUT_VALUE_PLC => #Retval_Fill_R, OUTPUT_VALUE_FEEDER => #ioPowder_Feeder_Unit_In_Out.Outputs."PF Setpoints, Warnings and Alarms".o_rHHlimitStirrerSpeedNominal_Line1)
      Sub(in1 := #oPLC_Aux.o_rStirrerSpeedNominal_Line1, in2 := #"iHMI_Offsets Alarms and Warnings".StirrerSpeedNominalLine1_Min_Alarm, out => #oPLC_Aux.o_rLLlimitStirrerSpeedNominal_Line1)
      "FC21020_FEEDER_SCALING"(DINT_INPUT_VALUE := 0, REAL_INPUT_VALUE := #oPLC_Aux.o_rLLlimitStirrerSpeedNominal_Line1, DINT_TO_REAL := false, REAL_TRANSFORM_FOR_FEEDER := true, OUTPUT_VALUE_PLC => #Retval_Fill_R, OUTPUT_VALUE_FEEDER => #ioPowder_Feeder_Unit_In_Out.Outputs."PF Setpoints, Warnings and Alarms".o_rLLlimitStirrerSpeedNominal_Line1)
   END_RUNG
   // the same network as SCL:
   #oPLC_Aux.o_rHHlimitStirrerSpeedNominal_Line1 := #oPLC_Aux.o_rStirrerSpeedNominal_Line1 + #"iHMI_Offsets Alarms and Warnings".StirrerSpeedNominalLine1_Max_Alarm;
   "FC21020_FEEDER_SCALING"(DINT_INPUT_VALUE := 0,
                           REAL_INPUT_VALUE := #oPLC_Aux.o_rHHlimitStirrerSpeedNominal_Line1,
                           DINT_TO_REAL := false,
                           REAL_TRANSFORM_FOR_FEEDER := true,
                           OUTPUT_VALUE_PLC => #Retval_Fill_R,
                           OUTPUT_VALUE_FEEDER => #ioPowder_Feeder_Unit_In_Out.Outputs."PF Setpoints, Warnings and Alarms".o_rHHlimitStirrerSpeedNominal_Line1,
                           ENO => #_w1);
   IF #_w1 THEN
       #oPLC_Aux.o_rLLlimitStirrerSpeedNominal_Line1 := #oPLC_Aux.o_rStirrerSpeedNominal_Line1 - #"iHMI_Offsets Alarms and Warnings".StirrerSpeedNominalLine1_Min_Alarm;
       "FC21020_FEEDER_SCALING"(DINT_INPUT_VALUE := 0,
                               REAL_INPUT_VALUE := #oPLC_Aux.o_rLLlimitStirrerSpeedNominal_Line1,
                               DINT_TO_REAL := false,
                               REAL_TRANSFORM_FOR_FEEDER := true,
                               OUTPUT_VALUE_PLC => #Retval_Fill_R,
                               OUTPUT_VALUE_FEEDER => #ioPowder_Feeder_Unit_In_Out.Outputs."PF Setpoints, Warnings and Alarms".o_rLLlimitStirrerSpeedNominal_Line1);
   END_IF;
END_REGION

REGION Network 28: STIRRER SPEED LINE 2 LIMITS CALCULATION ALARM
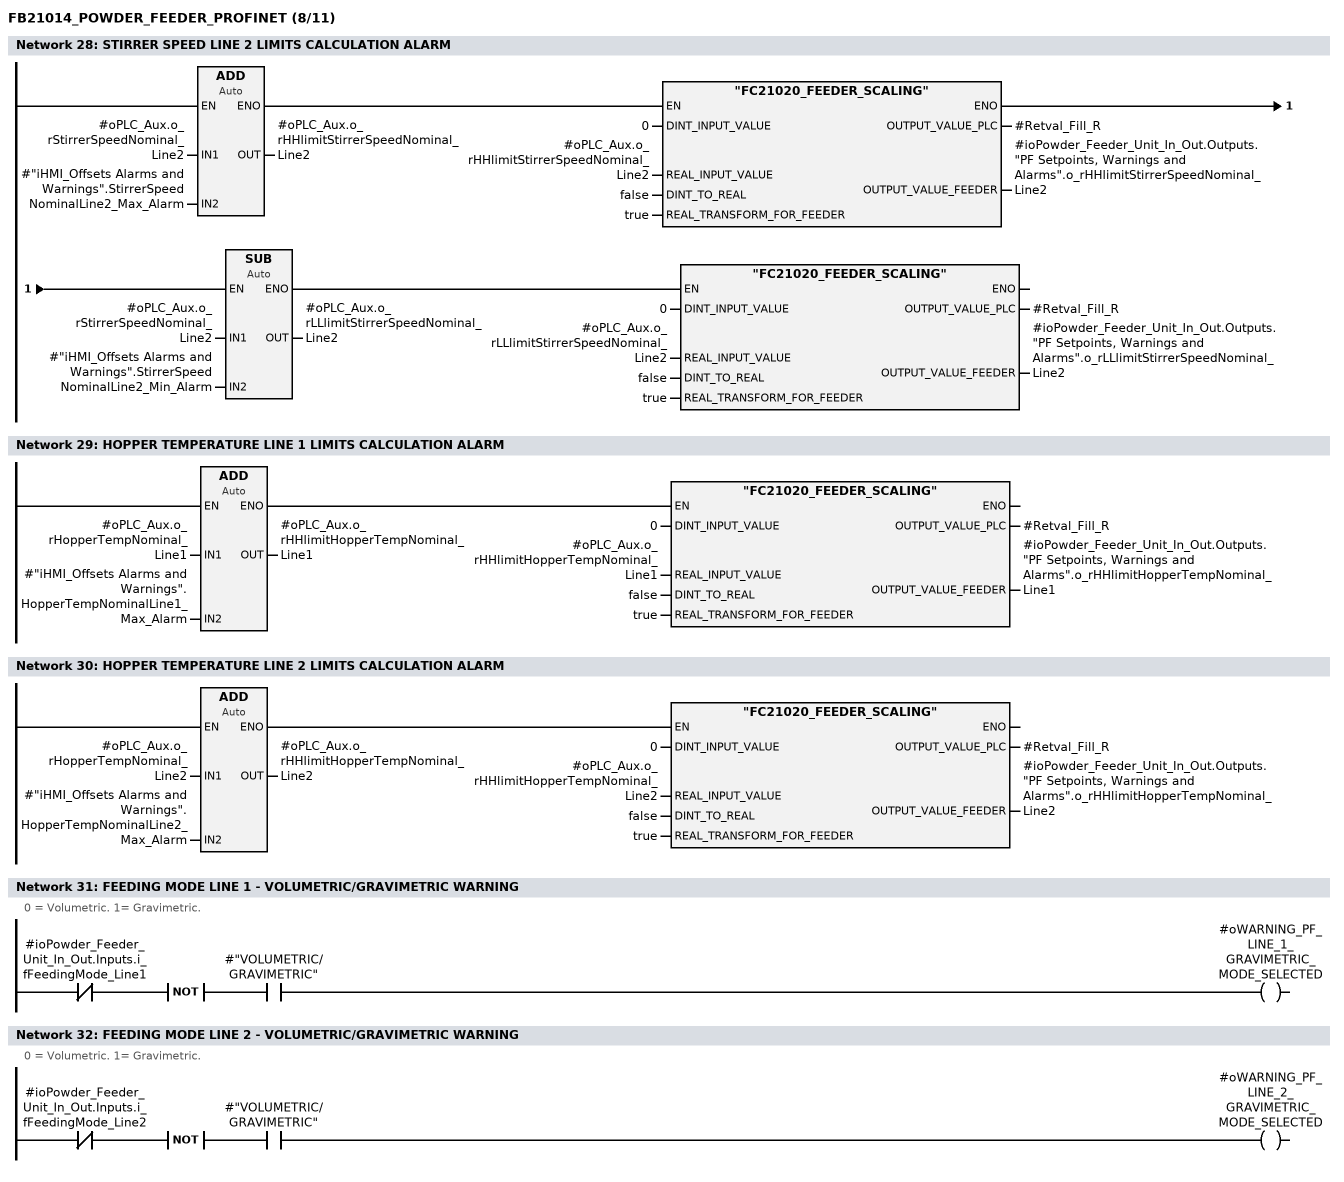
   RUNG wire#powerrail
      Add(in1 := #oPLC_Aux.o_rStirrerSpeedNominal_Line2, in2 := #"iHMI_Offsets Alarms and Warnings".StirrerSpeedNominalLine2_Max_Alarm, out => #oPLC_Aux.o_rHHlimitStirrerSpeedNominal_Line2)
      "FC21020_FEEDER_SCALING"(DINT_INPUT_VALUE := 0, REAL_INPUT_VALUE := #oPLC_Aux.o_rHHlimitStirrerSpeedNominal_Line2, DINT_TO_REAL := false, REAL_TRANSFORM_FOR_FEEDER := true, OUTPUT_VALUE_PLC => #Retval_Fill_R, OUTPUT_VALUE_FEEDER => #ioPowder_Feeder_Unit_In_Out.Outputs."PF Setpoints, Warnings and Alarms".o_rHHlimitStirrerSpeedNominal_Line2)
      Sub(in1 := #oPLC_Aux.o_rStirrerSpeedNominal_Line2, in2 := #"iHMI_Offsets Alarms and Warnings".StirrerSpeedNominalLine2_Min_Alarm, out => #oPLC_Aux.o_rLLlimitStirrerSpeedNominal_Line2)
      "FC21020_FEEDER_SCALING"(DINT_INPUT_VALUE := 0, REAL_INPUT_VALUE := #oPLC_Aux.o_rLLlimitStirrerSpeedNominal_Line2, DINT_TO_REAL := false, REAL_TRANSFORM_FOR_FEEDER := true, OUTPUT_VALUE_PLC => #Retval_Fill_R, OUTPUT_VALUE_FEEDER => #ioPowder_Feeder_Unit_In_Out.Outputs."PF Setpoints, Warnings and Alarms".o_rLLlimitStirrerSpeedNominal_Line2)
   END_RUNG
   // the same network as SCL:
   #oPLC_Aux.o_rHHlimitStirrerSpeedNominal_Line2 := #oPLC_Aux.o_rStirrerSpeedNominal_Line2 + #"iHMI_Offsets Alarms and Warnings".StirrerSpeedNominalLine2_Max_Alarm;
   "FC21020_FEEDER_SCALING"(DINT_INPUT_VALUE := 0,
                           REAL_INPUT_VALUE := #oPLC_Aux.o_rHHlimitStirrerSpeedNominal_Line2,
                           DINT_TO_REAL := false,
                           REAL_TRANSFORM_FOR_FEEDER := true,
                           OUTPUT_VALUE_PLC => #Retval_Fill_R,
                           OUTPUT_VALUE_FEEDER => #ioPowder_Feeder_Unit_In_Out.Outputs."PF Setpoints, Warnings and Alarms".o_rHHlimitStirrerSpeedNominal_Line2,
                           ENO => #_w1);
   IF #_w1 THEN
       #oPLC_Aux.o_rLLlimitStirrerSpeedNominal_Line2 := #oPLC_Aux.o_rStirrerSpeedNominal_Line2 - #"iHMI_Offsets Alarms and Warnings".StirrerSpeedNominalLine2_Min_Alarm;
       "FC21020_FEEDER_SCALING"(DINT_INPUT_VALUE := 0,
                               REAL_INPUT_VALUE := #oPLC_Aux.o_rLLlimitStirrerSpeedNominal_Line2,
                               DINT_TO_REAL := false,
                               REAL_TRANSFORM_FOR_FEEDER := true,
                               OUTPUT_VALUE_PLC => #Retval_Fill_R,
                               OUTPUT_VALUE_FEEDER => #ioPowder_Feeder_Unit_In_Out.Outputs."PF Setpoints, Warnings and Alarms".o_rLLlimitStirrerSpeedNominal_Line2);
   END_IF;
END_REGION

REGION Network 29: HOPPER TEMPERATURE LINE 1 LIMITS CALCULATION ALARM
   RUNG wire#powerrail
      Add(in1 := #oPLC_Aux.o_rHopperTempNominal_Line1, in2 := #"iHMI_Offsets Alarms and Warnings".HopperTempNominalLine1_Max_Alarm, out => #oPLC_Aux.o_rHHlimitHopperTempNominal_Line1)
      "FC21020_FEEDER_SCALING"(DINT_INPUT_VALUE := 0, REAL_INPUT_VALUE := #oPLC_Aux.o_rHHlimitHopperTempNominal_Line1, DINT_TO_REAL := false, REAL_TRANSFORM_FOR_FEEDER := true, OUTPUT_VALUE_PLC => #Retval_Fill_R, OUTPUT_VALUE_FEEDER => #ioPowder_Feeder_Unit_In_Out.Outputs."PF Setpoints, Warnings and Alarms".o_rHHlimitHopperTempNominal_Line1)
   END_RUNG
   // the same network as SCL:
   #oPLC_Aux.o_rHHlimitHopperTempNominal_Line1 := #oPLC_Aux.o_rHopperTempNominal_Line1 + #"iHMI_Offsets Alarms and Warnings".HopperTempNominalLine1_Max_Alarm;
   "FC21020_FEEDER_SCALING"(DINT_INPUT_VALUE := 0,
                           REAL_INPUT_VALUE := #oPLC_Aux.o_rHHlimitHopperTempNominal_Line1,
                           DINT_TO_REAL := false,
                           REAL_TRANSFORM_FOR_FEEDER := true,
                           OUTPUT_VALUE_PLC => #Retval_Fill_R,
                           OUTPUT_VALUE_FEEDER => #ioPowder_Feeder_Unit_In_Out.Outputs."PF Setpoints, Warnings and Alarms".o_rHHlimitHopperTempNominal_Line1);
END_REGION

REGION Network 30: HOPPER TEMPERATURE LINE 2 LIMITS CALCULATION ALARM
   RUNG wire#powerrail
      Add(in1 := #oPLC_Aux.o_rHopperTempNominal_Line2, in2 := #"iHMI_Offsets Alarms and Warnings".HopperTempNominalLine2_Max_Alarm, out => #oPLC_Aux.o_rHHlimitHopperTempNominal_Line2)
      "FC21020_FEEDER_SCALING"(DINT_INPUT_VALUE := 0, REAL_INPUT_VALUE := #oPLC_Aux.o_rHHlimitHopperTempNominal_Line2, DINT_TO_REAL := false, REAL_TRANSFORM_FOR_FEEDER := true, OUTPUT_VALUE_PLC => #Retval_Fill_R, OUTPUT_VALUE_FEEDER => #ioPowder_Feeder_Unit_In_Out.Outputs."PF Setpoints, Warnings and Alarms".o_rHHlimitHopperTempNominal_Line2)
   END_RUNG
   // the same network as SCL:
   #oPLC_Aux.o_rHHlimitHopperTempNominal_Line2 := #oPLC_Aux.o_rHopperTempNominal_Line2 + #"iHMI_Offsets Alarms and Warnings".HopperTempNominalLine2_Max_Alarm;
   "FC21020_FEEDER_SCALING"(DINT_INPUT_VALUE := 0,
                           REAL_INPUT_VALUE := #oPLC_Aux.o_rHHlimitHopperTempNominal_Line2,
                           DINT_TO_REAL := false,
                           REAL_TRANSFORM_FOR_FEEDER := true,
                           OUTPUT_VALUE_PLC => #Retval_Fill_R,
                           OUTPUT_VALUE_FEEDER => #ioPowder_Feeder_Unit_In_Out.Outputs."PF Setpoints, Warnings and Alarms".o_rHHlimitHopperTempNominal_Line2);
END_REGION

REGION Network 31: FEEDING MODE LINE 1 - VOLUMETRIC/GRAVIMETRIC WARNING
   // 0 = Volumetric. 1= Gravimetric.
   RUNG wire#powerrail
      I_Contact( #ioPowder_Feeder_Unit_In_Out.Inputs.i_fFeedingMode_Line1 )
      Not()
      Contact( #"VOLUMETRIC/GRAVIMETRIC" )
      Coil( #oWARNING_PF_LINE_1_GRAVIMETRIC_MODE_SELECTED )
   END_RUNG
   // the same network as SCL:
   #oWARNING_PF_LINE_1_GRAVIMETRIC_MODE_SELECTED := NOT (NOT #ioPowder_Feeder_Unit_In_Out.Inputs.i_fFeedingMode_Line1) AND #"VOLUMETRIC/GRAVIMETRIC";
END_REGION

REGION Network 32: FEEDING MODE LINE 2 - VOLUMETRIC/GRAVIMETRIC WARNING
   // 0 = Volumetric. 1= Gravimetric.
   RUNG wire#powerrail
      I_Contact( #ioPowder_Feeder_Unit_In_Out.Inputs.i_fFeedingMode_Line2 )
      Not()
      Contact( #"VOLUMETRIC/GRAVIMETRIC" )
      Coil( #oWARNING_PF_LINE_2_GRAVIMETRIC_MODE_SELECTED )
   END_RUNG
   // the same network as SCL:
   #oWARNING_PF_LINE_2_GRAVIMETRIC_MODE_SELECTED := NOT (NOT #ioPowder_Feeder_Unit_In_Out.Inputs.i_fFeedingMode_Line2) AND #"VOLUMETRIC/GRAVIMETRIC";
END_REGION

REGION Network 33: WARNING
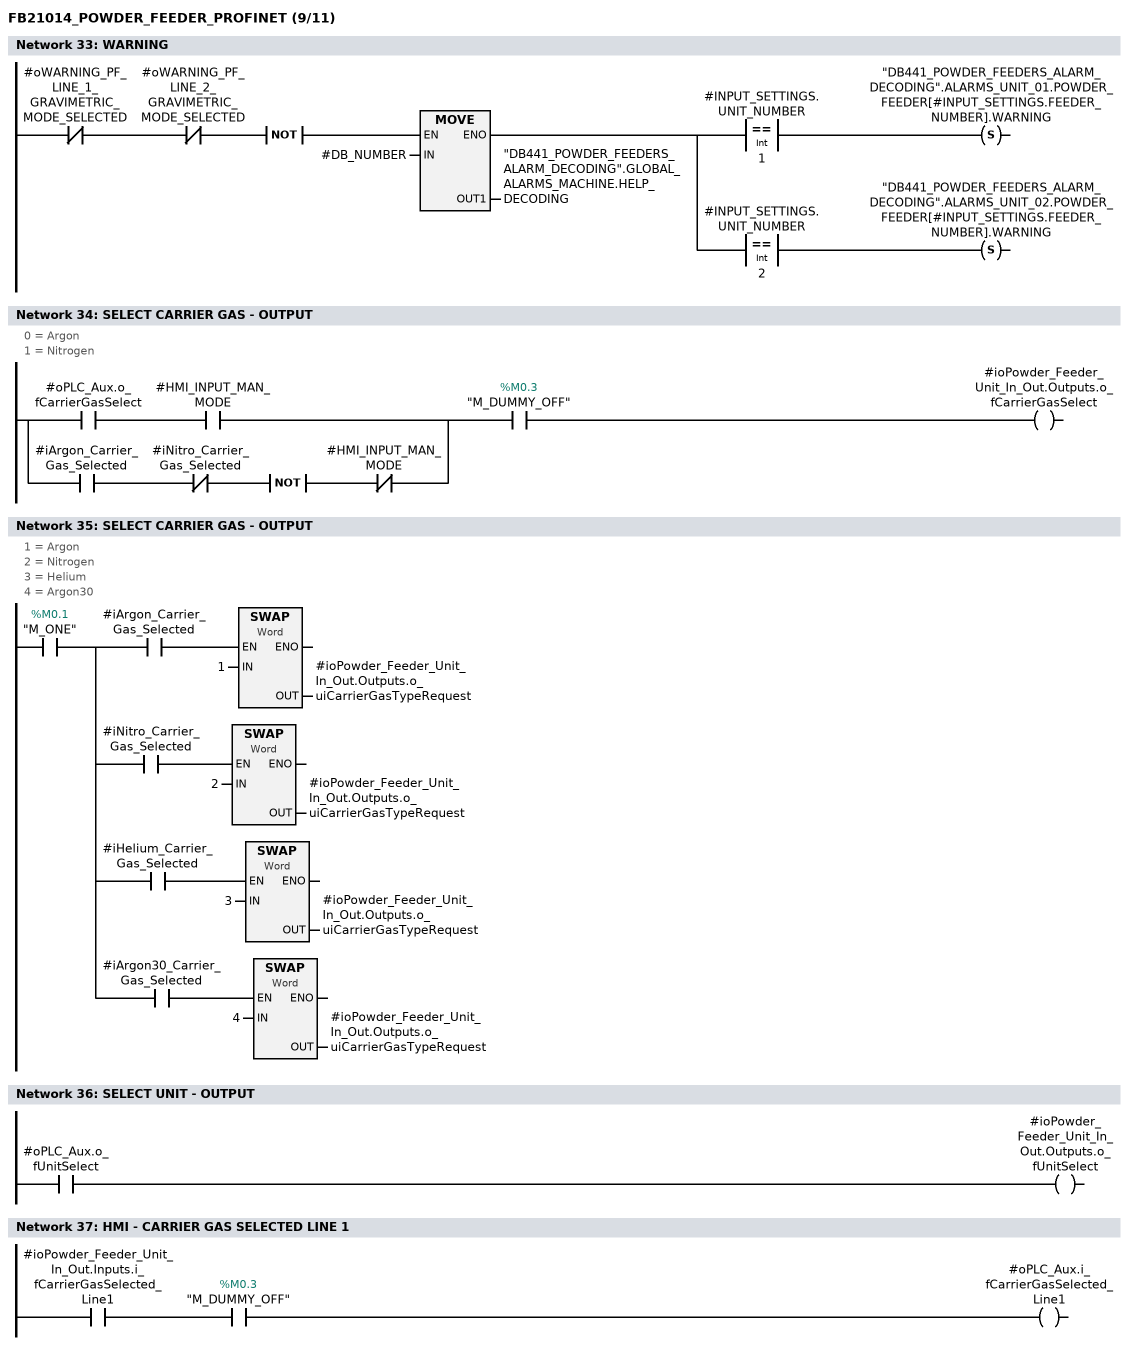
   RUNG wire#powerrail
      I_Contact( #oWARNING_PF_LINE_1_GRAVIMETRIC_MODE_SELECTED )
      I_Contact( #oWARNING_PF_LINE_2_GRAVIMETRIC_MODE_SELECTED )
      Not()
      Move(in := #DB_NUMBER, out1 => "DB441_POWDER_FEEDERS_ALARM_DECODING".GLOBAL_ALARMS_MACHINE.HELP_DECODING)
      wire#w1
      { S7_Templates := "SrcType := Int" } EQ_Contact(in1 := #INPUT_SETTINGS.UNIT_NUMBER, in2 := 1)
      S_Coil( "DB441_POWDER_FEEDERS_ALARM_DECODING".ALARMS_UNIT_01.POWDER_FEEDER[#INPUT_SETTINGS.FEEDER_NUMBER].WARNING )
   END_RUNG
   RUNG wire#w1
      { S7_Templates := "SrcType := Int" } EQ_Contact(in1 := #INPUT_SETTINGS.UNIT_NUMBER, in2 := 2)
      S_Coil( "DB441_POWDER_FEEDERS_ALARM_DECODING".ALARMS_UNIT_02.POWDER_FEEDER[#INPUT_SETTINGS.FEEDER_NUMBER].WARNING )
   END_RUNG
   // the same network as SCL:
   #_w1 := NOT (NOT #oWARNING_PF_LINE_1_GRAVIMETRIC_MODE_SELECTED AND NOT #oWARNING_PF_LINE_2_GRAVIMETRIC_MODE_SELECTED);
   IF #_w1 THEN
       "DB441_POWDER_FEEDERS_ALARM_DECODING".GLOBAL_ALARMS_MACHINE.HELP_DECODING := #DB_NUMBER;
   END_IF;
   IF #_w1 AND (#INPUT_SETTINGS.UNIT_NUMBER = 1) THEN
       "DB441_POWDER_FEEDERS_ALARM_DECODING".ALARMS_UNIT_01.POWDER_FEEDER[#INPUT_SETTINGS.FEEDER_NUMBER].WARNING := TRUE;
   END_IF;
   IF #_w1 AND (#INPUT_SETTINGS.UNIT_NUMBER = 2) THEN
       "DB441_POWDER_FEEDERS_ALARM_DECODING".ALARMS_UNIT_02.POWDER_FEEDER[#INPUT_SETTINGS.FEEDER_NUMBER].WARNING := TRUE;
   END_IF;
END_REGION

REGION Network 34: SELECT CARRIER GAS - OUTPUT
   // 0 = Argon
   // 1 = Nitrogen
   RUNG wire#powerrail
      Contact( #oPLC_Aux.o_fCarrierGasSelect )
      Contact( #HMI_INPUT_MAN_MODE )
      wire#w1
      Contact( "M_DUMMY_OFF" )
      Coil( #ioPowder_Feeder_Unit_In_Out.Outputs.o_fCarrierGasSelect )
   END_RUNG
   RUNG wire#powerrail
      Contact( #iArgon_Carrier_Gas_Selected )
      I_Contact( #iNitro_Carrier_Gas_Selected )
      Not()
      I_Contact( #HMI_INPUT_MAN_MODE )
   END_RUNG wire#w1
   // the same network as SCL:
   #ioPowder_Feeder_Unit_In_Out.Outputs.o_fCarrierGasSelect := ((#oPLC_Aux.o_fCarrierGasSelect AND #HMI_INPUT_MAN_MODE) OR (NOT (#iArgon_Carrier_Gas_Selected AND NOT #iNitro_Carrier_Gas_Selected) AND NOT #HMI_INPUT_MAN_MODE)) AND "M_DUMMY_OFF";
END_REGION

REGION Network 35: SELECT CARRIER GAS - OUTPUT
   // 1 = Argon
   // 2 = Nitrogen
   // 3 = Helium
   // 4 = Argon30
   IF "M_ONE" AND #iArgon_Carrier_Gas_Selected THEN
       #ioPowder_Feeder_Unit_In_Out.Outputs.o_uiCarrierGasTypeRequest := SWAP(1);
   END_IF;
   IF "M_ONE" AND #iNitro_Carrier_Gas_Selected THEN
       #ioPowder_Feeder_Unit_In_Out.Outputs.o_uiCarrierGasTypeRequest := SWAP(2);
   END_IF;
   IF "M_ONE" AND #iHelium_Carrier_Gas_Selected THEN
       #ioPowder_Feeder_Unit_In_Out.Outputs.o_uiCarrierGasTypeRequest := SWAP(3);
   END_IF;
   IF "M_ONE" AND #iArgon30_Carrier_Gas_Selected THEN
       #ioPowder_Feeder_Unit_In_Out.Outputs.o_uiCarrierGasTypeRequest := SWAP(4);
   END_IF;
END_REGION

REGION Network 36: SELECT UNIT - OUTPUT
   RUNG wire#powerrail
      Contact( #oPLC_Aux.o_fUnitSelect )
      Coil( #ioPowder_Feeder_Unit_In_Out.Outputs.o_fUnitSelect )
   END_RUNG
   // the same network as SCL:
   #ioPowder_Feeder_Unit_In_Out.Outputs.o_fUnitSelect := #oPLC_Aux.o_fUnitSelect;
END_REGION

REGION Network 37: HMI - CARRIER GAS SELECTED LINE 1
   RUNG wire#powerrail
      Contact( #ioPowder_Feeder_Unit_In_Out.Inputs.i_fCarrierGasSelected_Line1 )
      Contact( "M_DUMMY_OFF" )
      Coil( #oPLC_Aux.i_fCarrierGasSelected_Line1 )
   END_RUNG
   // the same network as SCL:
   #oPLC_Aux.i_fCarrierGasSelected_Line1 := #ioPowder_Feeder_Unit_In_Out.Inputs.i_fCarrierGasSelected_Line1 AND "M_DUMMY_OFF";
END_REGION

REGION Network 38: HMI - CARRIER GAS SELECTED LINE 2
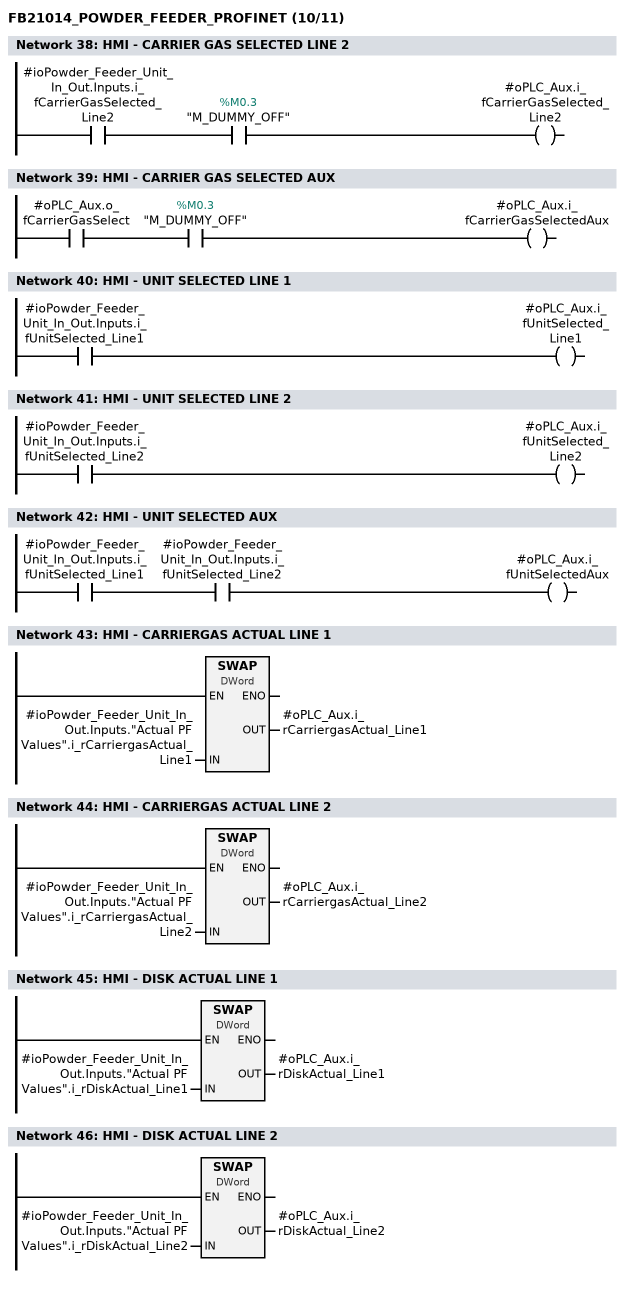
   RUNG wire#powerrail
      Contact( #ioPowder_Feeder_Unit_In_Out.Inputs.i_fCarrierGasSelected_Line2 )
      Contact( "M_DUMMY_OFF" )
      Coil( #oPLC_Aux.i_fCarrierGasSelected_Line2 )
   END_RUNG
   // the same network as SCL:
   #oPLC_Aux.i_fCarrierGasSelected_Line2 := #ioPowder_Feeder_Unit_In_Out.Inputs.i_fCarrierGasSelected_Line2 AND "M_DUMMY_OFF";
END_REGION

REGION Network 39: HMI - CARRIER GAS SELECTED AUX
   RUNG wire#powerrail
      Contact( #oPLC_Aux.o_fCarrierGasSelect )
      Contact( "M_DUMMY_OFF" )
      Coil( #oPLC_Aux.i_fCarrierGasSelectedAux )
   END_RUNG
   // the same network as SCL:
   #oPLC_Aux.i_fCarrierGasSelectedAux := #oPLC_Aux.o_fCarrierGasSelect AND "M_DUMMY_OFF";
END_REGION

REGION Network 40: HMI - UNIT SELECTED LINE 1
   RUNG wire#powerrail
      Contact( #ioPowder_Feeder_Unit_In_Out.Inputs.i_fUnitSelected_Line1 )
      Coil( #oPLC_Aux.i_fUnitSelected_Line1 )
   END_RUNG
   // the same network as SCL:
   #oPLC_Aux.i_fUnitSelected_Line1 := #ioPowder_Feeder_Unit_In_Out.Inputs.i_fUnitSelected_Line1;
END_REGION

REGION Network 41: HMI - UNIT SELECTED LINE 2
   RUNG wire#powerrail
      Contact( #ioPowder_Feeder_Unit_In_Out.Inputs.i_fUnitSelected_Line2 )
      Coil( #oPLC_Aux.i_fUnitSelected_Line2 )
   END_RUNG
   // the same network as SCL:
   #oPLC_Aux.i_fUnitSelected_Line2 := #ioPowder_Feeder_Unit_In_Out.Inputs.i_fUnitSelected_Line2;
END_REGION

REGION Network 42: HMI - UNIT SELECTED AUX
   RUNG wire#powerrail
      Contact( #ioPowder_Feeder_Unit_In_Out.Inputs.i_fUnitSelected_Line1 )
      Contact( #ioPowder_Feeder_Unit_In_Out.Inputs.i_fUnitSelected_Line2 )
      Coil( #oPLC_Aux.i_fUnitSelectedAux )
   END_RUNG
   // the same network as SCL:
   #oPLC_Aux.i_fUnitSelectedAux := #ioPowder_Feeder_Unit_In_Out.Inputs.i_fUnitSelected_Line1 AND #ioPowder_Feeder_Unit_In_Out.Inputs.i_fUnitSelected_Line2;
END_REGION

REGION Network 43: HMI - CARRIERGAS ACTUAL LINE 1
   #oPLC_Aux.i_rCarriergasActual_Line1 := SWAP(#ioPowder_Feeder_Unit_In_Out.Inputs."Actual PF Values".i_rCarriergasActual_Line1);
END_REGION

REGION Network 44: HMI - CARRIERGAS ACTUAL LINE 2
   #oPLC_Aux.i_rCarriergasActual_Line2 := SWAP(#ioPowder_Feeder_Unit_In_Out.Inputs."Actual PF Values".i_rCarriergasActual_Line2);
END_REGION

REGION Network 45: HMI - DISK ACTUAL LINE 1
   #oPLC_Aux.i_rDiskActual_Line1 := SWAP(#ioPowder_Feeder_Unit_In_Out.Inputs."Actual PF Values".i_rDiskActual_Line1);
END_REGION

REGION Network 46: HMI - DISK ACTUAL LINE 2
   #oPLC_Aux.i_rDiskActual_Line2 := SWAP(#ioPowder_Feeder_Unit_In_Out.Inputs."Actual PF Values".i_rDiskActual_Line2);
END_REGION

REGION Network 47: HMI - STIRRER ACTUAL LINE 1
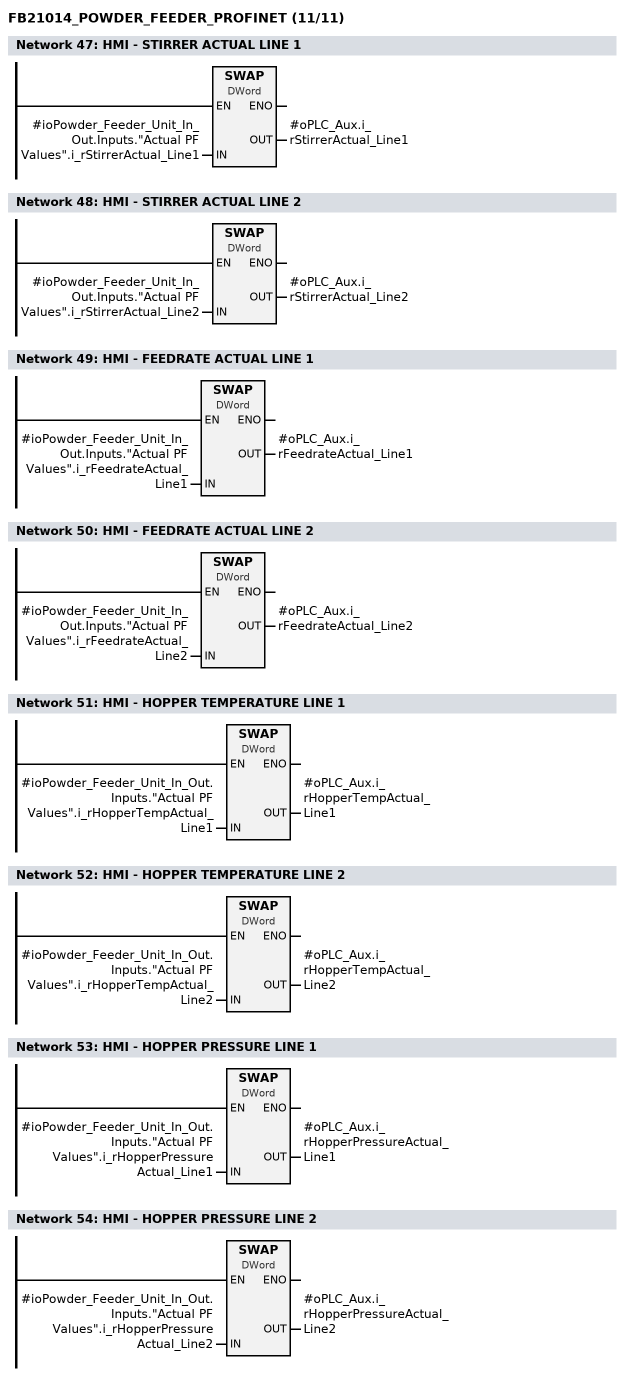
   #oPLC_Aux.i_rStirrerActual_Line1 := SWAP(#ioPowder_Feeder_Unit_In_Out.Inputs."Actual PF Values".i_rStirrerActual_Line1);
END_REGION

REGION Network 48: HMI - STIRRER ACTUAL LINE 2
   #oPLC_Aux.i_rStirrerActual_Line2 := SWAP(#ioPowder_Feeder_Unit_In_Out.Inputs."Actual PF Values".i_rStirrerActual_Line2);
END_REGION

REGION Network 49: HMI - FEEDRATE ACTUAL LINE 1
   #oPLC_Aux.i_rFeedrateActual_Line1 := SWAP(#ioPowder_Feeder_Unit_In_Out.Inputs."Actual PF Values".i_rFeedrateActual_Line1);
END_REGION

REGION Network 50: HMI - FEEDRATE ACTUAL LINE 2
   #oPLC_Aux.i_rFeedrateActual_Line2 := SWAP(#ioPowder_Feeder_Unit_In_Out.Inputs."Actual PF Values".i_rFeedrateActual_Line2);
END_REGION

REGION Network 51: HMI - HOPPER TEMPERATURE LINE 1
   #oPLC_Aux.i_rHopperTempActual_Line1 := SWAP(#ioPowder_Feeder_Unit_In_Out.Inputs."Actual PF Values".i_rHopperTempActual_Line1);
END_REGION

REGION Network 52: HMI - HOPPER TEMPERATURE LINE 2
   #oPLC_Aux.i_rHopperTempActual_Line2 := SWAP(#ioPowder_Feeder_Unit_In_Out.Inputs."Actual PF Values".i_rHopperTempActual_Line2);
END_REGION

REGION Network 53: HMI - HOPPER PRESSURE LINE 1
   #oPLC_Aux.i_rHopperPressureActual_Line1 := SWAP(#ioPowder_Feeder_Unit_In_Out.Inputs."Actual PF Values".i_rHopperPressureActual_Line1);
END_REGION

REGION Network 54: HMI - HOPPER PRESSURE LINE 2
   #oPLC_Aux.i_rHopperPressureActual_Line2 := SWAP(#ioPowder_Feeder_Unit_In_Out.Inputs."Actual PF Values".i_rHopperPressureActual_Line2);
END_REGION
END_FUNCTION_BLOCK

FUNCTION "FC21020_FEEDER_SCALING" : Void   // FC21020, LAD
TITLE = Robot-PLC Scaling
{ S7_Optimized_Access := 'TRUE' }
AUTHOR : Jbarturen
VERSION : 0.1
// stored: AutoNumber false, IsIECCheckEnabled false, SetENOAutomatically false, UDAEnableTagReadback false
   VAR_INPUT
      DINT_INPUT_VALUE : DInt;
      REAL_INPUT_VALUE : Real;
      DINT_TO_REAL : Bool;
      REAL_TRANSFORM_FOR_FEEDER : Bool;
   END_VAR
   VAR_OUTPUT
      OUTPUT_VALUE_PLC : Real;
      OUTPUT_VALUE_FEEDER : Real;
   END_VAR
   VAR_TEMP
      Value_Swapped : DInt;
      Value_Real : Real;
      Value_PLC : Real;
      Value_DWord : DWord;
      Value_DWord_Swapped : DWord;
   END_VAR
BEGIN

REGION Network 1: DATA TYPE CONVERTION / Robot-PLC
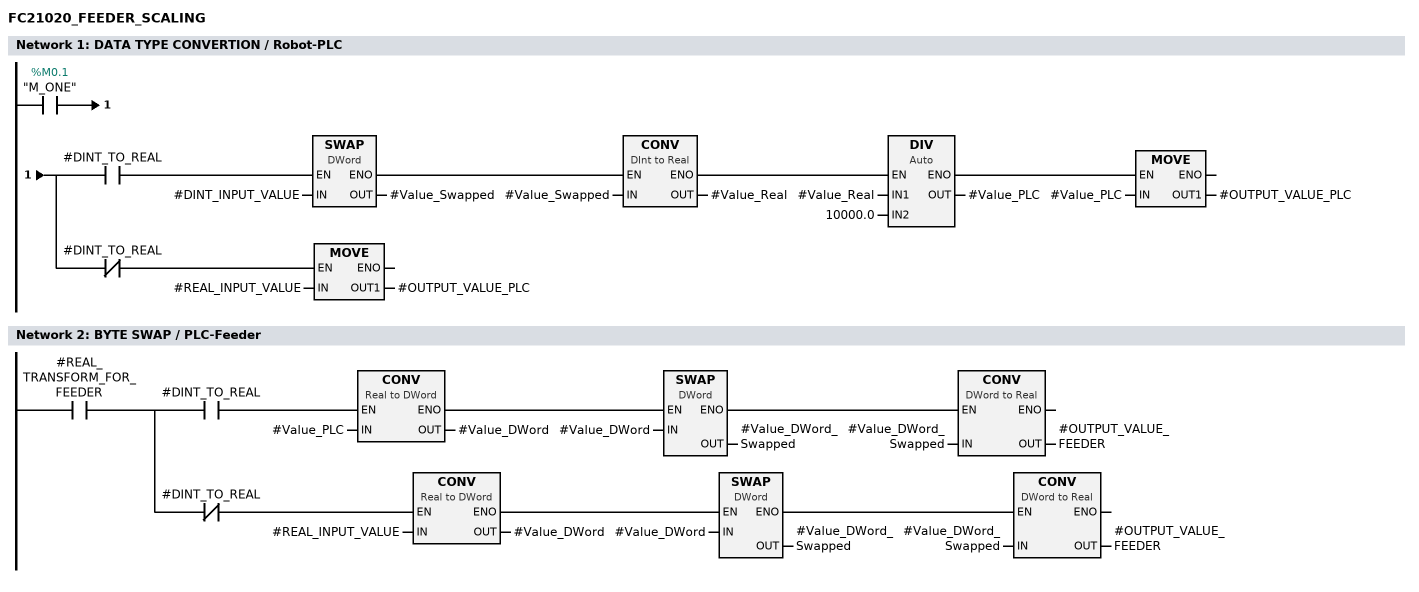
   IF "M_ONE" AND #DINT_TO_REAL THEN
       #Value_Swapped := SWAP(#DINT_INPUT_VALUE);
       #Value_Real := DINT_TO_REAL(#Value_Swapped);
       #Value_PLC := #Value_Real / 10000.0;
       #OUTPUT_VALUE_PLC := #Value_PLC;
   END_IF;
   IF "M_ONE" AND NOT #DINT_TO_REAL THEN #OUTPUT_VALUE_PLC := #REAL_INPUT_VALUE; END_IF;
END_REGION

REGION Network 2: BYTE SWAP / PLC-Feeder
   IF #REAL_TRANSFORM_FOR_FEEDER AND #DINT_TO_REAL THEN
       #Value_DWord := REAL_TO_DWORD(#Value_PLC);
       #Value_DWord_Swapped := SWAP(#Value_DWord);
       #OUTPUT_VALUE_FEEDER := DWORD_TO_REAL(#Value_DWord_Swapped);
   END_IF;
   IF #REAL_TRANSFORM_FOR_FEEDER AND NOT #DINT_TO_REAL THEN
       #Value_DWord := REAL_TO_DWORD(#REAL_INPUT_VALUE);
       #Value_DWord_Swapped := SWAP(#Value_DWord);
       #OUTPUT_VALUE_FEEDER := DWORD_TO_REAL(#Value_DWord_Swapped);
   END_IF;
END_REGION
END_FUNCTION

FUNCTION "FC21200_POWDER_FLOW_SENSOR_MEDICOAT" : Void   // FC21200, LAD
{ S7_Optimized_Access := 'TRUE' }
VERSION : 0.1
// stored: AutoNumber false, IsIECCheckEnabled false, SetENOAutomatically false, UDAEnableTagReadback false
BEGIN

REGION Network 1: /////_UNIT_01_/////
END_REGION

REGION Network 2: OERLIKON 1 LINE 1 OUTPUT MEDICOAT
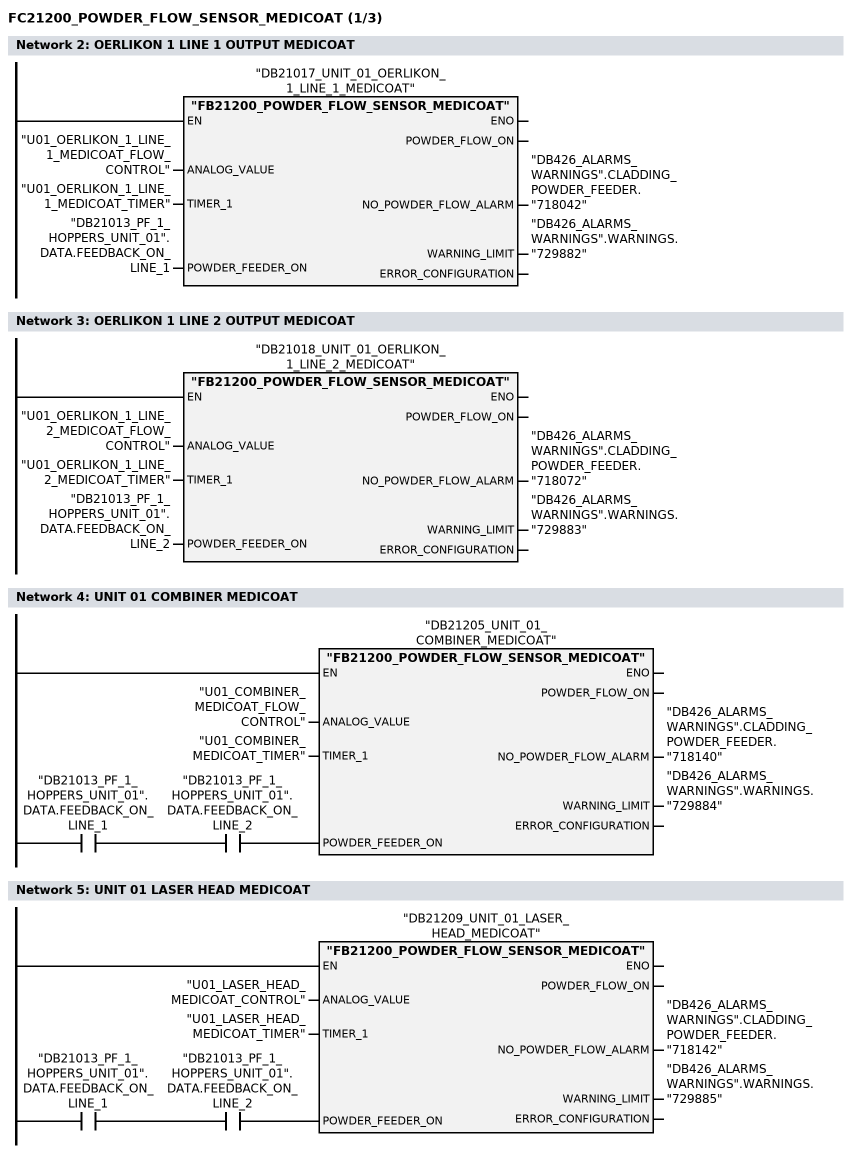
   RUNG wire#powerrail
      "DB21017_UNIT_01_OERLIKON_1_LINE_1_MEDICOAT"(ANALOG_VALUE := "U01_OERLIKON_1_LINE_1_MEDICOAT_FLOW_CONTROL", TIMER_1 := "U01_OERLIKON_1_LINE_1_MEDICOAT_TIMER", POWDER_FEEDER_ON := "DB21013_PF_1_HOPPERS_UNIT_01".DATA.FEEDBACK_ON_LINE_1, POWDER_FLOW_ON =>, NO_POWDER_FLOW_ALARM => "DB426_ALARMS_WARNINGS".CLADDING_POWDER_FEEDER."718042", WARNING_LIMIT => "DB426_ALARMS_WARNINGS".WARNINGS."729882", ERROR_CONFIGURATION =>)
   END_RUNG
   // the same network as SCL:
   "DB21017_UNIT_01_OERLIKON_1_LINE_1_MEDICOAT"(ANALOG_VALUE := "U01_OERLIKON_1_LINE_1_MEDICOAT_FLOW_CONTROL",   // "FB21200_POWDER_FLOW_SENSOR_MEDICOAT"
                           TIMER_1 := "U01_OERLIKON_1_LINE_1_MEDICOAT_TIMER",
                           POWDER_FEEDER_ON := "DB21013_PF_1_HOPPERS_UNIT_01".DATA.FEEDBACK_ON_LINE_1,
                           NO_POWDER_FLOW_ALARM => "DB426_ALARMS_WARNINGS".CLADDING_POWDER_FEEDER."718042",
                           WARNING_LIMIT => "DB426_ALARMS_WARNINGS".WARNINGS."729882");
END_REGION

REGION Network 3: OERLIKON 1 LINE 2 OUTPUT MEDICOAT
   RUNG wire#powerrail
      "DB21018_UNIT_01_OERLIKON_1_LINE_2_MEDICOAT"(ANALOG_VALUE := "U01_OERLIKON_1_LINE_2_MEDICOAT_FLOW_CONTROL", TIMER_1 := "U01_OERLIKON_1_LINE_2_MEDICOAT_TIMER", POWDER_FEEDER_ON := "DB21013_PF_1_HOPPERS_UNIT_01".DATA.FEEDBACK_ON_LINE_2, POWDER_FLOW_ON =>, NO_POWDER_FLOW_ALARM => "DB426_ALARMS_WARNINGS".CLADDING_POWDER_FEEDER."718072", WARNING_LIMIT => "DB426_ALARMS_WARNINGS".WARNINGS."729883", ERROR_CONFIGURATION =>)
   END_RUNG
   // the same network as SCL:
   "DB21018_UNIT_01_OERLIKON_1_LINE_2_MEDICOAT"(ANALOG_VALUE := "U01_OERLIKON_1_LINE_2_MEDICOAT_FLOW_CONTROL",   // "FB21200_POWDER_FLOW_SENSOR_MEDICOAT"
                           TIMER_1 := "U01_OERLIKON_1_LINE_2_MEDICOAT_TIMER",
                           POWDER_FEEDER_ON := "DB21013_PF_1_HOPPERS_UNIT_01".DATA.FEEDBACK_ON_LINE_2,
                           NO_POWDER_FLOW_ALARM => "DB426_ALARMS_WARNINGS".CLADDING_POWDER_FEEDER."718072",
                           WARNING_LIMIT => "DB426_ALARMS_WARNINGS".WARNINGS."729883");
END_REGION

REGION Network 4: UNIT 01 COMBINER MEDICOAT
   RUNG wire#powerrail
      "DB21205_UNIT_01_COMBINER_MEDICOAT"(POWDER_FEEDER_ON := wire#w1, ANALOG_VALUE := "U01_COMBINER_MEDICOAT_FLOW_CONTROL", TIMER_1 := "U01_COMBINER_MEDICOAT_TIMER", POWDER_FLOW_ON =>, NO_POWDER_FLOW_ALARM => "DB426_ALARMS_WARNINGS".CLADDING_POWDER_FEEDER."718140", WARNING_LIMIT => "DB426_ALARMS_WARNINGS".WARNINGS."729884", ERROR_CONFIGURATION =>)
   END_RUNG
   RUNG wire#powerrail
      Contact( "DB21013_PF_1_HOPPERS_UNIT_01".DATA.FEEDBACK_ON_LINE_1 )
      Contact( "DB21013_PF_1_HOPPERS_UNIT_01".DATA.FEEDBACK_ON_LINE_2 )
   END_RUNG wire#w1
   // the same network as SCL:
   "DB21205_UNIT_01_COMBINER_MEDICOAT"(ANALOG_VALUE := "U01_COMBINER_MEDICOAT_FLOW_CONTROL",   // "FB21200_POWDER_FLOW_SENSOR_MEDICOAT"
                           TIMER_1 := "U01_COMBINER_MEDICOAT_TIMER",
                           POWDER_FEEDER_ON := "DB21013_PF_1_HOPPERS_UNIT_01".DATA.FEEDBACK_ON_LINE_1 AND "DB21013_PF_1_HOPPERS_UNIT_01".DATA.FEEDBACK_ON_LINE_2,
                           NO_POWDER_FLOW_ALARM => "DB426_ALARMS_WARNINGS".CLADDING_POWDER_FEEDER."718140",
                           WARNING_LIMIT => "DB426_ALARMS_WARNINGS".WARNINGS."729884");
END_REGION

REGION Network 5: UNIT 01 LASER HEAD MEDICOAT
   RUNG wire#powerrail
      "DB21209_UNIT_01_LASER_HEAD_MEDICOAT"(POWDER_FEEDER_ON := wire#w1, ANALOG_VALUE := "U01_LASER_HEAD_MEDICOAT_CONTROL", TIMER_1 := "U01_LASER_HEAD_MEDICOAT_TIMER", POWDER_FLOW_ON =>, NO_POWDER_FLOW_ALARM => "DB426_ALARMS_WARNINGS".CLADDING_POWDER_FEEDER."718142", WARNING_LIMIT => "DB426_ALARMS_WARNINGS".WARNINGS."729885", ERROR_CONFIGURATION =>)
   END_RUNG
   RUNG wire#powerrail
      Contact( "DB21013_PF_1_HOPPERS_UNIT_01".DATA.FEEDBACK_ON_LINE_1 )
      Contact( "DB21013_PF_1_HOPPERS_UNIT_01".DATA.FEEDBACK_ON_LINE_2 )
   END_RUNG wire#w1
   // the same network as SCL:
   "DB21209_UNIT_01_LASER_HEAD_MEDICOAT"(ANALOG_VALUE := "U01_LASER_HEAD_MEDICOAT_CONTROL",   // "FB21200_POWDER_FLOW_SENSOR_MEDICOAT"
                           TIMER_1 := "U01_LASER_HEAD_MEDICOAT_TIMER",
                           POWDER_FEEDER_ON := "DB21013_PF_1_HOPPERS_UNIT_01".DATA.FEEDBACK_ON_LINE_1 AND "DB21013_PF_1_HOPPERS_UNIT_01".DATA.FEEDBACK_ON_LINE_2,
                           NO_POWDER_FLOW_ALARM => "DB426_ALARMS_WARNINGS".CLADDING_POWDER_FEEDER."718142",
                           WARNING_LIMIT => "DB426_ALARMS_WARNINGS".WARNINGS."729885");
END_REGION

REGION Network 6: /////_UNIT_02_/////
END_REGION

REGION Network 7: UNIT 02 OERLIKON 1 LINE 1 OUTPUT MEDICOAT
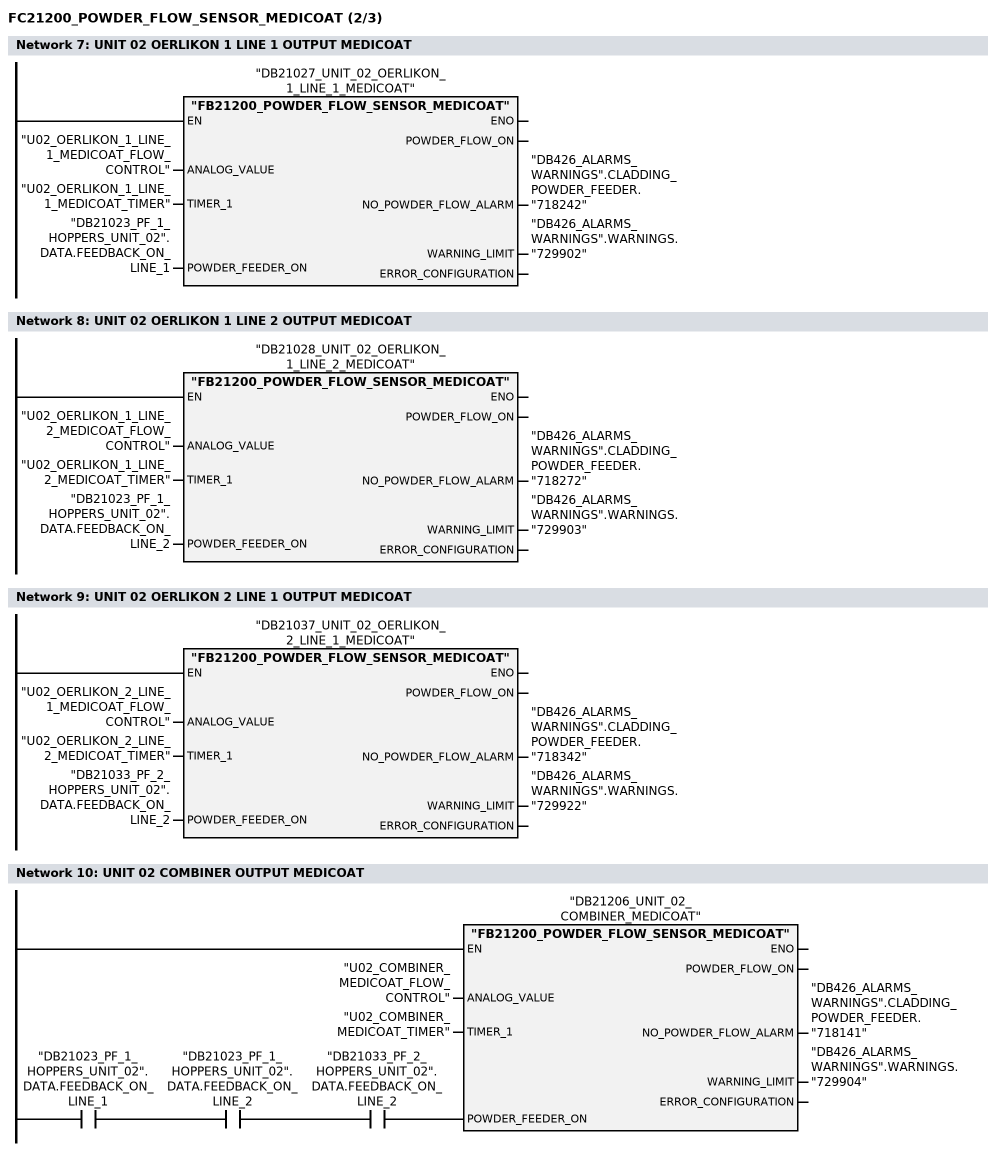
   RUNG wire#powerrail
      "DB21027_UNIT_02_OERLIKON_1_LINE_1_MEDICOAT"(ANALOG_VALUE := "U02_OERLIKON_1_LINE_1_MEDICOAT_FLOW_CONTROL", TIMER_1 := "U02_OERLIKON_1_LINE_1_MEDICOAT_TIMER", POWDER_FEEDER_ON := "DB21023_PF_1_HOPPERS_UNIT_02".DATA.FEEDBACK_ON_LINE_1, POWDER_FLOW_ON =>, NO_POWDER_FLOW_ALARM => "DB426_ALARMS_WARNINGS".CLADDING_POWDER_FEEDER."718242", WARNING_LIMIT => "DB426_ALARMS_WARNINGS".WARNINGS."729902", ERROR_CONFIGURATION =>)
   END_RUNG
   // the same network as SCL:
   "DB21027_UNIT_02_OERLIKON_1_LINE_1_MEDICOAT"(ANALOG_VALUE := "U02_OERLIKON_1_LINE_1_MEDICOAT_FLOW_CONTROL",   // "FB21200_POWDER_FLOW_SENSOR_MEDICOAT"
                           TIMER_1 := "U02_OERLIKON_1_LINE_1_MEDICOAT_TIMER",
                           POWDER_FEEDER_ON := "DB21023_PF_1_HOPPERS_UNIT_02".DATA.FEEDBACK_ON_LINE_1,
                           NO_POWDER_FLOW_ALARM => "DB426_ALARMS_WARNINGS".CLADDING_POWDER_FEEDER."718242",
                           WARNING_LIMIT => "DB426_ALARMS_WARNINGS".WARNINGS."729902");
END_REGION

REGION Network 8: UNIT 02 OERLIKON 1 LINE 2 OUTPUT MEDICOAT
   RUNG wire#powerrail
      "DB21028_UNIT_02_OERLIKON_1_LINE_2_MEDICOAT"(ANALOG_VALUE := "U02_OERLIKON_1_LINE_2_MEDICOAT_FLOW_CONTROL", TIMER_1 := "U02_OERLIKON_1_LINE_2_MEDICOAT_TIMER", POWDER_FEEDER_ON := "DB21023_PF_1_HOPPERS_UNIT_02".DATA.FEEDBACK_ON_LINE_2, POWDER_FLOW_ON =>, NO_POWDER_FLOW_ALARM => "DB426_ALARMS_WARNINGS".CLADDING_POWDER_FEEDER."718272", WARNING_LIMIT => "DB426_ALARMS_WARNINGS".WARNINGS."729903", ERROR_CONFIGURATION =>)
   END_RUNG
   // the same network as SCL:
   "DB21028_UNIT_02_OERLIKON_1_LINE_2_MEDICOAT"(ANALOG_VALUE := "U02_OERLIKON_1_LINE_2_MEDICOAT_FLOW_CONTROL",   // "FB21200_POWDER_FLOW_SENSOR_MEDICOAT"
                           TIMER_1 := "U02_OERLIKON_1_LINE_2_MEDICOAT_TIMER",
                           POWDER_FEEDER_ON := "DB21023_PF_1_HOPPERS_UNIT_02".DATA.FEEDBACK_ON_LINE_2,
                           NO_POWDER_FLOW_ALARM => "DB426_ALARMS_WARNINGS".CLADDING_POWDER_FEEDER."718272",
                           WARNING_LIMIT => "DB426_ALARMS_WARNINGS".WARNINGS."729903");
END_REGION

REGION Network 9: UNIT 02 OERLIKON 2 LINE 1 OUTPUT MEDICOAT
   RUNG wire#powerrail
      "DB21037_UNIT_02_OERLIKON_2_LINE_1_MEDICOAT"(ANALOG_VALUE := "U02_OERLIKON_2_LINE_1_MEDICOAT_FLOW_CONTROL", TIMER_1 := "U02_OERLIKON_2_LINE_2_MEDICOAT_TIMER", POWDER_FEEDER_ON := "DB21033_PF_2_HOPPERS_UNIT_02".DATA.FEEDBACK_ON_LINE_2, POWDER_FLOW_ON =>, NO_POWDER_FLOW_ALARM => "DB426_ALARMS_WARNINGS".CLADDING_POWDER_FEEDER."718342", WARNING_LIMIT => "DB426_ALARMS_WARNINGS".WARNINGS."729922", ERROR_CONFIGURATION =>)
   END_RUNG
   // the same network as SCL:
   "DB21037_UNIT_02_OERLIKON_2_LINE_1_MEDICOAT"(ANALOG_VALUE := "U02_OERLIKON_2_LINE_1_MEDICOAT_FLOW_CONTROL",   // "FB21200_POWDER_FLOW_SENSOR_MEDICOAT"
                           TIMER_1 := "U02_OERLIKON_2_LINE_2_MEDICOAT_TIMER",
                           POWDER_FEEDER_ON := "DB21033_PF_2_HOPPERS_UNIT_02".DATA.FEEDBACK_ON_LINE_2,
                           NO_POWDER_FLOW_ALARM => "DB426_ALARMS_WARNINGS".CLADDING_POWDER_FEEDER."718342",
                           WARNING_LIMIT => "DB426_ALARMS_WARNINGS".WARNINGS."729922");
END_REGION

REGION Network 10: UNIT 02 COMBINER OUTPUT MEDICOAT
   RUNG wire#powerrail
      "DB21206_UNIT_02_COMBINER_MEDICOAT"(POWDER_FEEDER_ON := wire#w1, ANALOG_VALUE := "U02_COMBINER_MEDICOAT_FLOW_CONTROL", TIMER_1 := "U02_COMBINER_MEDICOAT_TIMER", POWDER_FLOW_ON =>, NO_POWDER_FLOW_ALARM => "DB426_ALARMS_WARNINGS".CLADDING_POWDER_FEEDER."718141", WARNING_LIMIT => "DB426_ALARMS_WARNINGS".WARNINGS."729904", ERROR_CONFIGURATION =>)
   END_RUNG
   RUNG wire#powerrail
      Contact( "DB21023_PF_1_HOPPERS_UNIT_02".DATA.FEEDBACK_ON_LINE_1 )
      Contact( "DB21023_PF_1_HOPPERS_UNIT_02".DATA.FEEDBACK_ON_LINE_2 )
      Contact( "DB21033_PF_2_HOPPERS_UNIT_02".DATA.FEEDBACK_ON_LINE_2 )
   END_RUNG wire#w1
   // the same network as SCL:
   "DB21206_UNIT_02_COMBINER_MEDICOAT"(ANALOG_VALUE := "U02_COMBINER_MEDICOAT_FLOW_CONTROL",   // "FB21200_POWDER_FLOW_SENSOR_MEDICOAT"
                           TIMER_1 := "U02_COMBINER_MEDICOAT_TIMER",
                           POWDER_FEEDER_ON := "DB21023_PF_1_HOPPERS_UNIT_02".DATA.FEEDBACK_ON_LINE_1 AND "DB21023_PF_1_HOPPERS_UNIT_02".DATA.FEEDBACK_ON_LINE_2 AND "DB21033_PF_2_HOPPERS_UNIT_02".DATA.FEEDBACK_ON_LINE_2,
                           NO_POWDER_FLOW_ALARM => "DB426_ALARMS_WARNINGS".CLADDING_POWDER_FEEDER."718141",
                           WARNING_LIMIT => "DB426_ALARMS_WARNINGS".WARNINGS."729904");
END_REGION

REGION Network 11: UNIT 02 LASER HEAD OUTPUT MEDICOAT
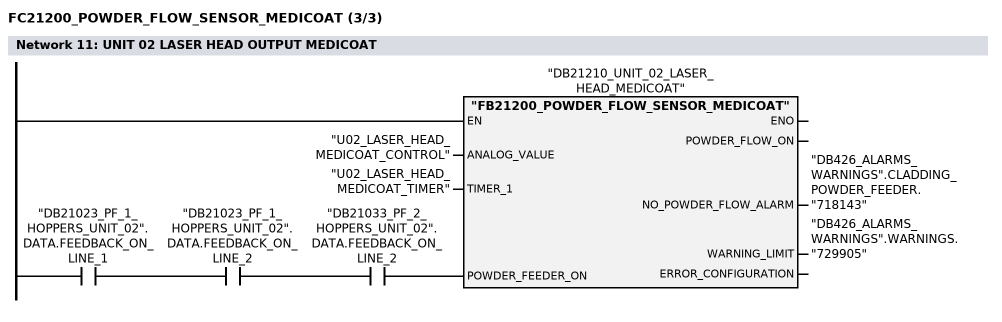
   RUNG wire#powerrail
      "DB21210_UNIT_02_LASER_HEAD_MEDICOAT"(POWDER_FEEDER_ON := wire#w1, ANALOG_VALUE := "U02_LASER_HEAD_MEDICOAT_CONTROL", TIMER_1 := "U02_LASER_HEAD_MEDICOAT_TIMER", POWDER_FLOW_ON =>, NO_POWDER_FLOW_ALARM => "DB426_ALARMS_WARNINGS".CLADDING_POWDER_FEEDER."718143", WARNING_LIMIT => "DB426_ALARMS_WARNINGS".WARNINGS."729905", ERROR_CONFIGURATION =>)
   END_RUNG
   RUNG wire#powerrail
      Contact( "DB21023_PF_1_HOPPERS_UNIT_02".DATA.FEEDBACK_ON_LINE_1 )
      Contact( "DB21023_PF_1_HOPPERS_UNIT_02".DATA.FEEDBACK_ON_LINE_2 )
      Contact( "DB21033_PF_2_HOPPERS_UNIT_02".DATA.FEEDBACK_ON_LINE_2 )
   END_RUNG wire#w1
   // the same network as SCL:
   "DB21210_UNIT_02_LASER_HEAD_MEDICOAT"(ANALOG_VALUE := "U02_LASER_HEAD_MEDICOAT_CONTROL",   // "FB21200_POWDER_FLOW_SENSOR_MEDICOAT"
                           TIMER_1 := "U02_LASER_HEAD_MEDICOAT_TIMER",
                           POWDER_FEEDER_ON := "DB21023_PF_1_HOPPERS_UNIT_02".DATA.FEEDBACK_ON_LINE_1 AND "DB21023_PF_1_HOPPERS_UNIT_02".DATA.FEEDBACK_ON_LINE_2 AND "DB21033_PF_2_HOPPERS_UNIT_02".DATA.FEEDBACK_ON_LINE_2,
                           NO_POWDER_FLOW_ALARM => "DB426_ALARMS_WARNINGS".CLADDING_POWDER_FEEDER."718143",
                           WARNING_LIMIT => "DB426_ALARMS_WARNINGS".WARNINGS."729905");
END_REGION
END_FUNCTION

FUNCTION_BLOCK "FB21200_POWDER_FLOW_SENSOR_MEDICOAT"   // FB21200, LAD
{ S7_Optimized_Access := 'FALSE' }
VERSION : 0.1
// stored: AutoNumber false, IsIECCheckEnabled false, SetENOAutomatically false, UDAEnableTagReadback false
   VAR_INPUT
      ANALOG_VALUE : Int;   // SENSOR VALUE INPUT
      TIMER_1 : Timer;   // TIMER FOR NOT FLOW ALARM
      POWDER_FEEDER_ON { ExternalVisible := 'False'; ExternalWritable := 'False'} : Bool;   // POWDER FEEDER SWITCHED ON
   END_VAR
   VAR_OUTPUT
      POWDER_FLOW_ON : Bool;   // POWDER FLOW OK
      NO_POWDER_FLOW_ALARM : Bool;   // NO POWDER FLOW ALARM
      WARNING_LIMIT : Bool;   // WARNING FLOW OUT OF LIMITS
      ERROR_CONFIGURATION : Bool;   // WRONG CONFIGURATION ERROR
   END_VAR
   VAR DB_SPECIFIC
      OUTPUT : Struct
         VALUE_REAL : Real;   // POWDER FLOW VALUE
         VALUE_INT : Int;
      END_STRUCT;
      INPUT_SETTINGS : Struct
         LOW_RANGE : Real;   // LOWER VALUE TO SCALE ANALOG SIGNAL
         HIGH_RANGE : Real;   // HIGHER VALUE TO SCALE ANALOG SIGNAL
         LOW_LIMIT_TO_POWDER_FLOW_ON : Real;   // MINIMUM VALUE TO POWDER FLOW OK
         UNIT_NUMBER : Int;
         FEEDER_NUMBER : Int;
      END_STRUCT;
      ALARMS_SETTINGS : Struct
         WARN_LIMIT_LOW : Real;   // LOWER LIMIT FOR WARNING
         WARN_LIMIT_HIGH : Real;   // HIGHER LIMIT FOR WARNING
      END_STRUCT;
      LOG : Struct
         DATE_MAX_MASS : Date_And_Time;
         VALUE_MAX_MASS : Real;
      END_STRUCT;
   END_VAR
   VAR_TEMP
      NORM_VALUE : Real;
      RETVAL : Word;
      DB_NUMBER : DInt;
   END_VAR
   VAR_TEMP   // added for the SCL form of the ladder/FBD networks
      _w1 : Bool;
      _s5time1 : S5Time;
   END_VAR
BEGIN

NETWORK
TITLE = READ INSTANCE DB NUMBER
      L     DINO;
      +     10#800000;
      T     #DB_NUMBER;

REGION Network 2: INPUTS
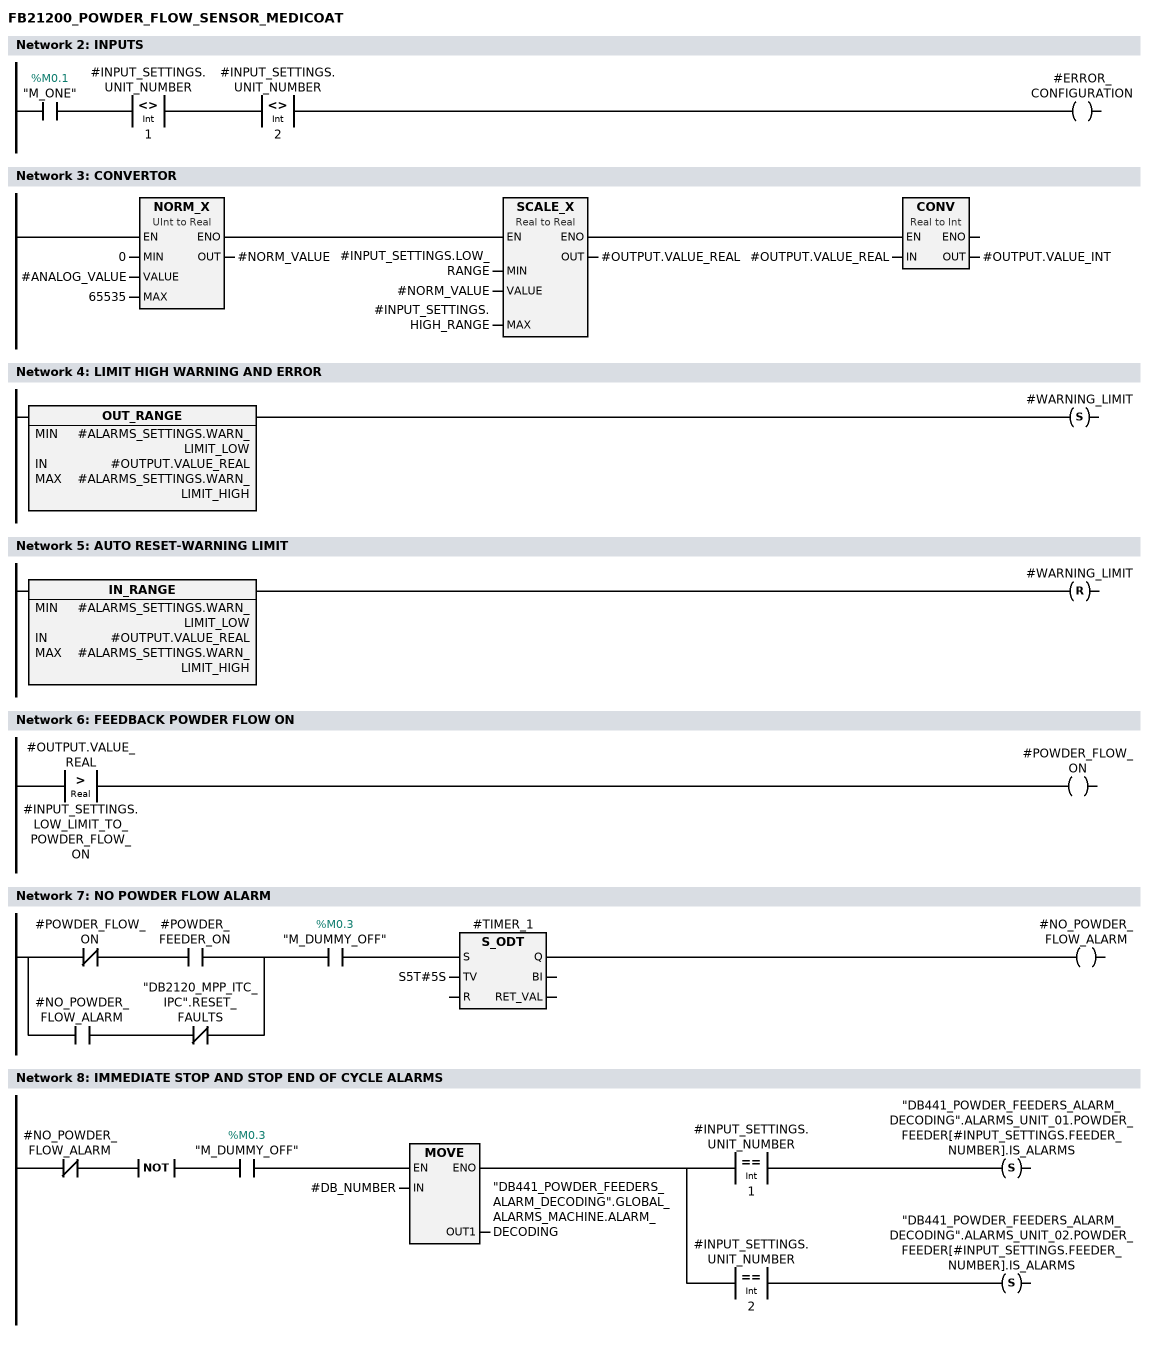
   RUNG wire#powerrail
      Contact( "M_ONE" )
      { S7_Templates := "SrcType := Int" } NE_Contact(in1 := #INPUT_SETTINGS.UNIT_NUMBER, in2 := 1)
      { S7_Templates := "SrcType := Int" } NE_Contact(in1 := #INPUT_SETTINGS.UNIT_NUMBER, in2 := 2)
      Coil( #ERROR_CONFIGURATION )
   END_RUNG
   // the same network as SCL:
   #ERROR_CONFIGURATION := "M_ONE" AND (#INPUT_SETTINGS.UNIT_NUMBER <> 1) AND (#INPUT_SETTINGS.UNIT_NUMBER <> 2);
END_REGION

REGION Network 3: CONVERTOR
   RUNG wire#powerrail
      { S7_Templates := "[SrcType := UInt, DestType := Real]" } Normalize(min := 0, value := #ANALOG_VALUE, max := 65535, out => #NORM_VALUE)
      { S7_Templates := "[SrcType := Real, DestType := Real]" } Scale(min := #INPUT_SETTINGS.LOW_RANGE, value := #NORM_VALUE, max := #INPUT_SETTINGS.HIGH_RANGE, out => #OUTPUT.VALUE_REAL)
      { S7_Templates := "[SrcType := Real, DestType := Int]" } Convert(in := #OUTPUT.VALUE_REAL, out => #OUTPUT.VALUE_INT)
   END_RUNG
   // the same network as SCL:
   #NORM_VALUE := NORM_X(MIN := 0, VALUE := #ANALOG_VALUE, MAX := 65535);
   #OUTPUT.VALUE_REAL := SCALE_X(MIN := #INPUT_SETTINGS.LOW_RANGE, VALUE := #NORM_VALUE, MAX := #INPUT_SETTINGS.HIGH_RANGE);
   #OUTPUT.VALUE_INT := REAL_TO_INT(#OUTPUT.VALUE_REAL);
END_REGION

REGION Network 4: LIMIT HIGH WARNING AND ERROR
   IF (#OUTPUT.VALUE_REAL < #ALARMS_SETTINGS.WARN_LIMIT_LOW) OR (#OUTPUT.VALUE_REAL > #ALARMS_SETTINGS.WARN_LIMIT_HIGH) THEN
       #WARNING_LIMIT := TRUE;
   END_IF;
END_REGION

REGION Network 5: AUTO RESET-WARNING LIMIT
   RUNG wire#powerrail
      { S7_Templates := "SrcType := Real" } InRange(min := #ALARMS_SETTINGS.WARN_LIMIT_LOW, in := #OUTPUT.VALUE_REAL, max := #ALARMS_SETTINGS.WARN_LIMIT_HIGH)
      R_Coil( #WARNING_LIMIT )
   END_RUNG
   // the same network as SCL:
   IF (#ALARMS_SETTINGS.WARN_LIMIT_LOW <= #OUTPUT.VALUE_REAL) AND (#OUTPUT.VALUE_REAL <= #ALARMS_SETTINGS.WARN_LIMIT_HIGH) THEN
       #WARNING_LIMIT := FALSE;
   END_IF;
END_REGION

REGION Network 6: FEEDBACK POWDER FLOW ON
   RUNG wire#powerrail
      { S7_Templates := "SrcType := Real" } GT_Contact(in1 := #OUTPUT.VALUE_REAL, in2 := #INPUT_SETTINGS.LOW_LIMIT_TO_POWDER_FLOW_ON)
      Coil( #POWDER_FLOW_ON )
   END_RUNG
   // the same network as SCL:
   #POWDER_FLOW_ON := #OUTPUT.VALUE_REAL > #INPUT_SETTINGS.LOW_LIMIT_TO_POWDER_FLOW_ON;
END_REGION

REGION Network 7: NO POWDER FLOW ALARM
   RUNG wire#powerrail
      I_Contact( #POWDER_FLOW_ON )
      Contact( #POWDER_FEEDER_ON )
      wire#w1
      Contact( "M_DUMMY_OFF" )
      S_ODT(T_NO := #TIMER_1, TV := S5T#5S, R :=, BI =>, RET_VAL =>)
      Coil( #NO_POWDER_FLOW_ALARM )
   END_RUNG
   RUNG wire#powerrail
      Contact( #NO_POWDER_FLOW_ALARM )
      I_Contact( "DB2120_MPP_ITC_IPC".RESET_FAULTS )
   END_RUNG wire#w1
   // the same network as SCL:
   #_s5time1 := S_ODT(T_NO := #TIMER_1,
                      S := ((NOT #POWDER_FLOW_ON AND #POWDER_FEEDER_ON) OR (#NO_POWDER_FLOW_ALARM AND NOT "DB2120_MPP_ITC_IPC".RESET_FAULTS)) AND "M_DUMMY_OFF",
                      TV := S5T#5S,
                      Q => #_w1);
   #NO_POWDER_FLOW_ALARM := #_w1;
END_REGION

REGION Network 8: IMMEDIATE STOP AND STOP END OF CYCLE ALARMS
   RUNG wire#powerrail
      I_Contact( #NO_POWDER_FLOW_ALARM )
      Not()
      Contact( "M_DUMMY_OFF" )
      Move(in := #DB_NUMBER, out1 => "DB441_POWDER_FEEDERS_ALARM_DECODING".GLOBAL_ALARMS_MACHINE.ALARM_DECODING)
      wire#w1
      { S7_Templates := "SrcType := Int" } EQ_Contact(in1 := #INPUT_SETTINGS.UNIT_NUMBER, in2 := 1)
      S_Coil( "DB441_POWDER_FEEDERS_ALARM_DECODING".ALARMS_UNIT_01.POWDER_FEEDER[#INPUT_SETTINGS.FEEDER_NUMBER].IS_ALARMS )
   END_RUNG
   RUNG wire#w1
      { S7_Templates := "SrcType := Int" } EQ_Contact(in1 := #INPUT_SETTINGS.UNIT_NUMBER, in2 := 2)
      S_Coil( "DB441_POWDER_FEEDERS_ALARM_DECODING".ALARMS_UNIT_02.POWDER_FEEDER[#INPUT_SETTINGS.FEEDER_NUMBER].IS_ALARMS )
   END_RUNG
   // the same network as SCL:
   #_w1 := NOT (NOT #NO_POWDER_FLOW_ALARM) AND "M_DUMMY_OFF";
   IF #_w1 THEN
       "DB441_POWDER_FEEDERS_ALARM_DECODING".GLOBAL_ALARMS_MACHINE.ALARM_DECODING := #DB_NUMBER;
   END_IF;
   IF #_w1 AND (#INPUT_SETTINGS.UNIT_NUMBER = 1) THEN
       "DB441_POWDER_FEEDERS_ALARM_DECODING".ALARMS_UNIT_01.POWDER_FEEDER[#INPUT_SETTINGS.FEEDER_NUMBER].IS_ALARMS := TRUE;
   END_IF;
   IF #_w1 AND (#INPUT_SETTINGS.UNIT_NUMBER = 2) THEN
       "DB441_POWDER_FEEDERS_ALARM_DECODING".ALARMS_UNIT_02.POWDER_FEEDER[#INPUT_SETTINGS.FEEDER_NUMBER].IS_ALARMS := TRUE;
   END_IF;
END_REGION
END_FUNCTION_BLOCK

FUNCTION "FC16000_OPC_UA_GENERAL" : Void   // FC16000, LAD
{ S7_Optimized_Access := 'TRUE' }
VERSION : 0.1
// stored: AutoNumber false, IsIECCheckEnabled false, SetENOAutomatically false, UDAEnableTagReadback false
BEGIN

REGION Network 1
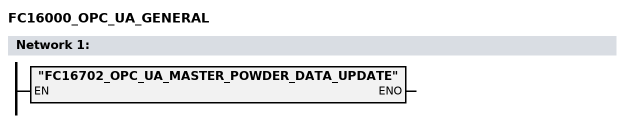
   RUNG wire#powerrail
      "FC16702_OPC_UA_MASTER_POWDER_DATA_UPDATE"()
   END_RUNG
   // the same network as SCL:
   "FC16702_OPC_UA_MASTER_POWDER_DATA_UPDATE"();
END_REGION
END_FUNCTION

ORGANIZATION_BLOCK "Cyclic interrupt"   // OB30, LAD, CyclicInterrupt
{ S7_Optimized_Access := 'TRUE' }
VERSION : 0.1
// stored: AutoNumber false, IsIECCheckEnabled false, SetENOAutomatically false
   VAR_INPUT
      Initial_Call : Bool;   // Initial call of this OB
      Event_Count : Int;   // Events discarded
   END_VAR
   VAR_TEMP
      LOOP_COUNT : Int;
   END_VAR
BEGIN

REGION Network 1: INITIALIZING OF ARRAY POINTERS FOR LOOP / Initializing of array pointers for loop
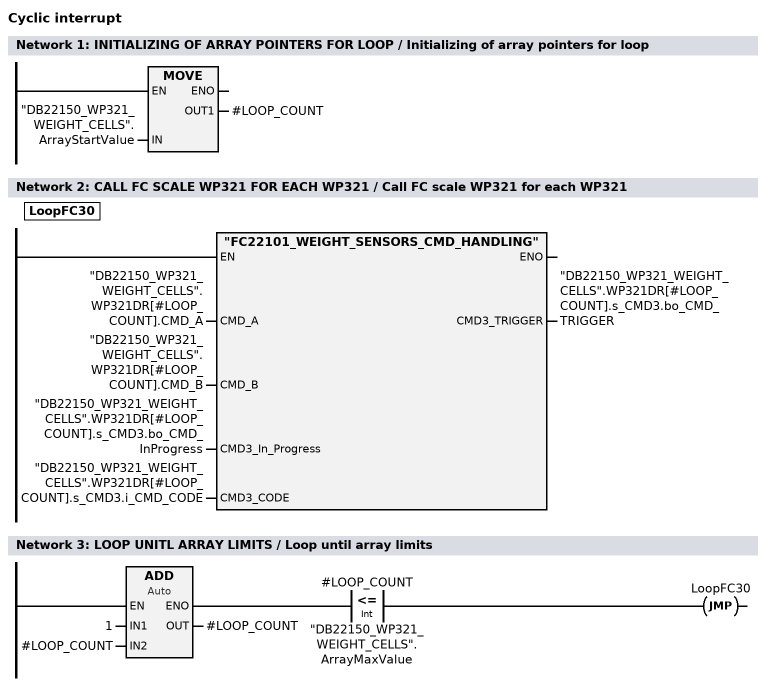
   RUNG wire#powerrail
      Move(in := "DB22150_WP321_WEIGHT_CELLS".ArrayStartValue, out1 => #LOOP_COUNT)
   END_RUNG
   // the same network as SCL:
   #LOOP_COUNT := "DB22150_WP321_WEIGHT_CELLS".ArrayStartValue;
END_REGION

REGION Network 2: CALL FC SCALE WP321 FOR EACH WP321 / Call FC scale WP321 for each WP321
   Label( LoopFC30 )
   RUNG wire#powerrail
      "FC22101_WEIGHT_SENSORS_CMD_HANDLING"(CMD_A := "DB22150_WP321_WEIGHT_CELLS".WP321DR[#LOOP_COUNT].CMD_A, CMD_B := "DB22150_WP321_WEIGHT_CELLS".WP321DR[#LOOP_COUNT].CMD_B, CMD3_In_Progress := "DB22150_WP321_WEIGHT_CELLS".WP321DR[#LOOP_COUNT].s_CMD3.bo_CMD_InProgress, CMD3_CODE := "DB22150_WP321_WEIGHT_CELLS".WP321DR[#LOOP_COUNT].s_CMD3.i_CMD_CODE, CMD3_TRIGGER => "DB22150_WP321_WEIGHT_CELLS".WP321DR[#LOOP_COUNT].s_CMD3.bo_CMD_TRIGGER)
   END_RUNG
   // the same network as SCL:
   LoopFC30:
   "FC22101_WEIGHT_SENSORS_CMD_HANDLING"(CMD_A := "DB22150_WP321_WEIGHT_CELLS".WP321DR[#LOOP_COUNT].CMD_A,
                           CMD_B := "DB22150_WP321_WEIGHT_CELLS".WP321DR[#LOOP_COUNT].CMD_B,
                           CMD3_In_Progress := "DB22150_WP321_WEIGHT_CELLS".WP321DR[#LOOP_COUNT].s_CMD3.bo_CMD_InProgress,
                           CMD3_CODE := "DB22150_WP321_WEIGHT_CELLS".WP321DR[#LOOP_COUNT].s_CMD3.i_CMD_CODE,
                           CMD3_TRIGGER => "DB22150_WP321_WEIGHT_CELLS".WP321DR[#LOOP_COUNT].s_CMD3.bo_CMD_TRIGGER);
END_REGION

REGION Network 3: LOOP UNITL ARRAY LIMITS / Loop until array limits
   RUNG wire#powerrail
      Add(in1 := 1, in2 := #LOOP_COUNT, out => #LOOP_COUNT)
      { S7_Templates := "SrcType := Int" } LE_Contact(in1 := #LOOP_COUNT, in2 := "DB22150_WP321_WEIGHT_CELLS".ArrayMaxValue)
      JumpCoil( LoopFC30 )
   END_RUNG
   // the same network as SCL:
   #LOOP_COUNT := 1 + #LOOP_COUNT;
   IF #LOOP_COUNT <= "DB22150_WP321_WEIGHT_CELLS".ArrayMaxValue THEN GOTO LoopFC30; END_IF;
END_REGION
END_ORGANIZATION_BLOCK

ORGANIZATION_BLOCK "OB100_RESTART"   // OB100, LAD, Startup
TITLE = "Complete Restart"
{ S7_Optimized_Access := 'FALSE' }
AUTHOR : ETXETAR
VERSION : 1.0
// stored: AutoNumber false, IsIECCheckEnabled false, SetENOAutomatically false
   VAR_TEMP
      OB100_EV_CLASS : Byte;
      OB100_STRTUP : Byte;
      OB100_PRIORITY : Byte;
      OB100_OB_NUMBR : Byte;
      OB100_RESERVED_1 : Byte;
      OB100_RESERVED_2 : Byte;
      OB100_STOP : Word;
      OB100_RESERVED_3 : Word;
      OB100_RESERVED_4 : Word;
      OB100_DATE_TIME : Date_And_Time;
      __PlcmigTempFillBits_20B0 : Array[0..7] of Bool;
   END_VAR
BEGIN

REGION Network 1: M_ONE / ESTABLISH "LOGIC 1" BIT
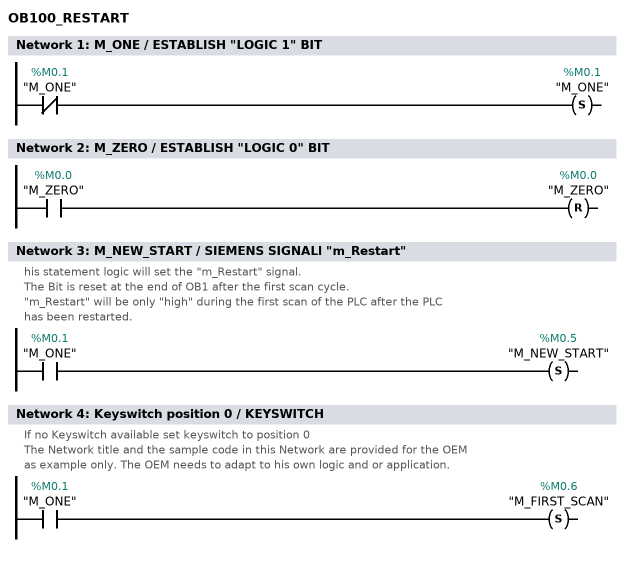
   RUNG wire#powerrail
      I_Contact( "M_ONE" )
      S_Coil( "M_ONE" )
   END_RUNG
   // the same network as SCL:
   IF NOT "M_ONE" THEN "M_ONE" := TRUE; END_IF;
END_REGION

REGION Network 2: M_ZERO / ESTABLISH "LOGIC 0" BIT
   RUNG wire#powerrail
      Contact( "M_ZERO" )
      R_Coil( "M_ZERO" )
   END_RUNG
   // the same network as SCL:
   IF "M_ZERO" THEN "M_ZERO" := FALSE; END_IF;
END_REGION

REGION Network 3: M_NEW_START / SIEMENS SIGNALl "m_Restart"
   // his statement logic will set the "m_Restart" signal.
   // The Bit is reset at the end of OB1 after the first scan cycle.
   // 
   // "m_Restart" will be only "high" during the first scan of the PLC after the PLC 
   // has been restarted.
   RUNG wire#powerrail
      Contact( "M_ONE" )
      S_Coil( "M_NEW_START" )
   END_RUNG
   // the same network as SCL:
   IF "M_ONE" THEN "M_NEW_START" := TRUE; END_IF;
END_REGION

REGION Network 4: Keyswitch position 0 / KEYSWITCH
   // If no Keyswitch available set keyswitch to position 0
   // 
   // The Network title and the sample code in this Network are provided for the OEM 
   // as example only. The OEM needs to adapt to his own logic and or application.
   RUNG wire#powerrail
      Contact( "M_ONE" )
      S_Coil( "M_FIRST_SCAN" )
   END_RUNG
   // the same network as SCL:
   IF "M_ONE" THEN "M_FIRST_SCAN" := TRUE; END_IF;
END_REGION
END_ORGANIZATION_BLOCK

ORGANIZATION_BLOCK "OB121_SYNCHRONF1"   // OB121, LAD, ProgrammingError
{ S7_Optimized_Access := 'FALSE' }
VERSION : 0.0
// stored: IsIECCheckEnabled false, SetENOAutomatically false
   VAR_TEMP
      TEMP0 : Byte;
      TEMP1 : Byte;
      TEMP2 : Byte;
      TEMP3 : Byte;
      TEMP4 : Byte;
      TEMP5 : Byte;
      TEMP6 : Word;
      TEMP7 : Word;
      TEMP8 : Word;
      TEMP9 : Date_And_Time;
   END_VAR
BEGIN
END_ORGANIZATION_BLOCK

ORGANIZATION_BLOCK "OB122_SYNCHRONF2"   // OB122, LAD, IOAccessError
{ S7_Optimized_Access := 'FALSE' }
VERSION : 0.0
// stored: IsIECCheckEnabled false, SetENOAutomatically false
   VAR_TEMP
      TEMP0 : Byte;
      TEMP1 : Byte;
      TEMP2 : Byte;
      TEMP3 : Byte;
      TEMP4 : Byte;
      TEMP5 : Byte;
      TEMP6 : Word;
      TEMP7 : Word;
      TEMP8 : Word;
      TEMP9 : Date_And_Time;
   END_VAR
BEGIN
END_ORGANIZATION_BLOCK

ORGANIZATION_BLOCK "OB40 Hardware interrupt"   // OB40, LAD, HardwareInterrupt
{ S7_Optimized_Access := 'TRUE' }
VERSION : 0.1
// stored: AutoNumber true, IsIECCheckEnabled false, SetENOAutomatically false
   VAR_INPUT
      LADDR : HW_IO;   // Hardware identifier
      USI : Word;   // User structure identifier
      IChannel : USInt;   // Interrupt channel number
      EventType : Byte;   // EventType
      PointAddr : DWord;
   END_VAR
   VAR_TEMP
      FLAG : Variant;
   END_VAR
BEGIN
END_ORGANIZATION_BLOCK

FUNCTION "FC2142_HOPPERS_SIGNAL_TOWER" : Void   // FC2142, LAD
{ S7_Optimized_Access := 'TRUE' }
VERSION : 0.1
// stored: AutoNumber false, IsIECCheckEnabled false, SetENOAutomatically false, UDAEnableTagReadback false
BEGIN

REGION Network 2: SIGNAL TOWER GREEN LIGHT OUTPUT / SIGNAL TOWER, GREEN LIGHT
   // M0.3 agregar las señales de starved y blocked de la celula / GREEN LIGHT
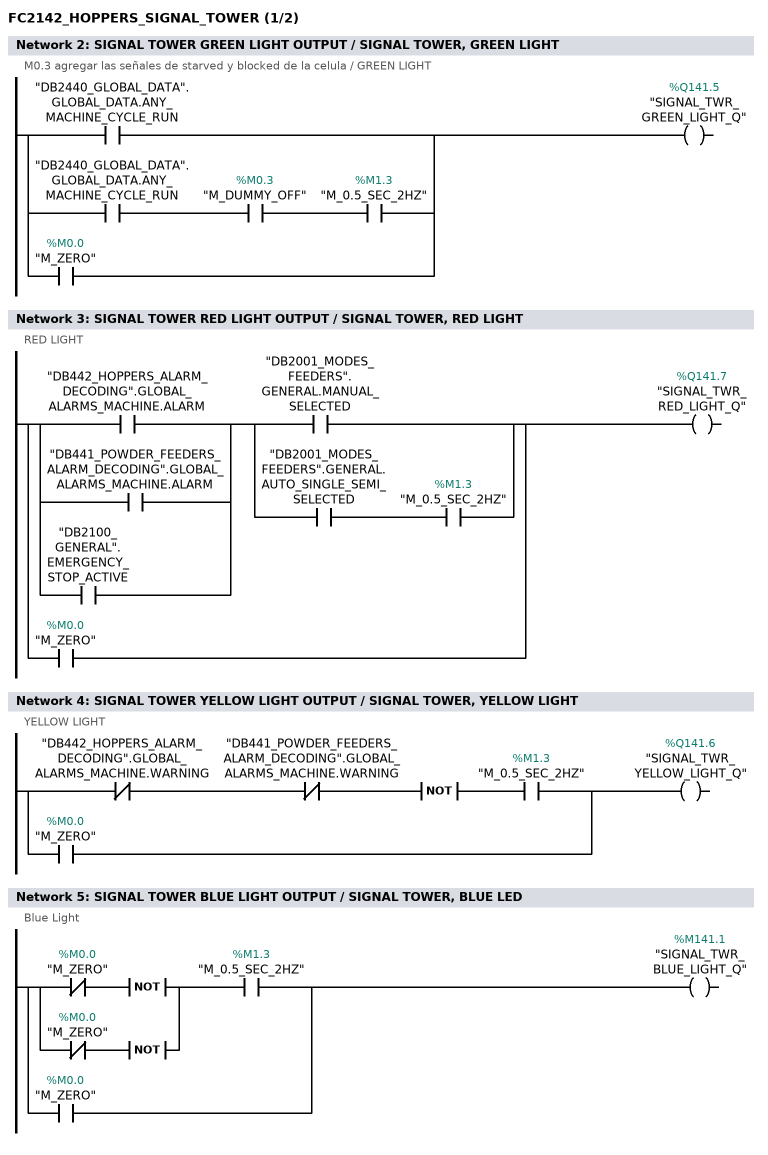
   RUNG wire#powerrail
      Contact( "DB2440_GLOBAL_DATA".GLOBAL_DATA.ANY_MACHINE_CYCLE_RUN )
      wire#w1
      Coil( "SIGNAL_TWR_GREEN_LIGHT_Q" )
   END_RUNG
   RUNG wire#powerrail
      Contact( "DB2440_GLOBAL_DATA".GLOBAL_DATA.ANY_MACHINE_CYCLE_RUN )
      Contact( "M_DUMMY_OFF" )
      Contact( "M_0.5_SEC_2HZ" )
   END_RUNG wire#w1
   RUNG wire#powerrail
      Contact( "M_ZERO" )
   END_RUNG wire#w1
   // the same network as SCL:
   "SIGNAL_TWR_GREEN_LIGHT_Q" := "DB2440_GLOBAL_DATA".GLOBAL_DATA.ANY_MACHINE_CYCLE_RUN OR ("DB2440_GLOBAL_DATA".GLOBAL_DATA.ANY_MACHINE_CYCLE_RUN AND "M_DUMMY_OFF" AND "M_0.5_SEC_2HZ") OR "M_ZERO";
END_REGION

REGION Network 3: SIGNAL TOWER RED LIGHT OUTPUT / SIGNAL TOWER, RED LIGHT
   // RED LIGHT
   RUNG wire#powerrail
      Contact( "DB442_HOPPERS_ALARM_DECODING".GLOBAL_ALARMS_MACHINE.ALARM )
      wire#w1
      Contact( "DB2001_MODES_FEEDERS".GENERAL.MANUAL_SELECTED )
      wire#w2
      Coil( "SIGNAL_TWR_RED_LIGHT_Q" )
   END_RUNG
   RUNG wire#powerrail
      Contact( "DB441_POWDER_FEEDERS_ALARM_DECODING".GLOBAL_ALARMS_MACHINE.ALARM )
   END_RUNG wire#w1
   RUNG wire#powerrail
      Contact( "DB2100_GENERAL".EMERGENCY_STOP_ACTIVE )
   END_RUNG wire#w1
   RUNG wire#w1
      Contact( "DB2001_MODES_FEEDERS".GENERAL.AUTO_SINGLE_SEMI_SELECTED )
      Contact( "M_0.5_SEC_2HZ" )
   END_RUNG wire#w2
   RUNG wire#powerrail
      Contact( "M_ZERO" )
   END_RUNG wire#w2
   // the same network as SCL:
   "SIGNAL_TWR_RED_LIGHT_Q" := (("DB442_HOPPERS_ALARM_DECODING".GLOBAL_ALARMS_MACHINE.ALARM OR "DB441_POWDER_FEEDERS_ALARM_DECODING".GLOBAL_ALARMS_MACHINE.ALARM OR "DB2100_GENERAL".EMERGENCY_STOP_ACTIVE) AND ("DB2001_MODES_FEEDERS".GENERAL.MANUAL_SELECTED OR ("DB2001_MODES_FEEDERS".GENERAL.AUTO_SINGLE_SEMI_SELECTED AND "M_0.5_SEC_2HZ"))) OR "M_ZERO";
END_REGION

REGION Network 4: SIGNAL TOWER YELLOW LIGHT OUTPUT / SIGNAL TOWER, YELLOW LIGHT
   // YELLOW LIGHT
   RUNG wire#powerrail
      I_Contact( "DB442_HOPPERS_ALARM_DECODING".GLOBAL_ALARMS_MACHINE.WARNING )
      I_Contact( "DB441_POWDER_FEEDERS_ALARM_DECODING".GLOBAL_ALARMS_MACHINE.WARNING )
      Not()
      Contact( "M_0.5_SEC_2HZ" )
      wire#w1
      Coil( "SIGNAL_TWR_YELLOW_LIGHT_Q" )
   END_RUNG
   RUNG wire#powerrail
      Contact( "M_ZERO" )
   END_RUNG wire#w1
   // the same network as SCL:
   "SIGNAL_TWR_YELLOW_LIGHT_Q" := (NOT (NOT "DB442_HOPPERS_ALARM_DECODING".GLOBAL_ALARMS_MACHINE.WARNING AND NOT "DB441_POWDER_FEEDERS_ALARM_DECODING".GLOBAL_ALARMS_MACHINE.WARNING) AND "M_0.5_SEC_2HZ") OR "M_ZERO";
END_REGION

REGION Network 5: SIGNAL TOWER BLUE LIGHT OUTPUT / SIGNAL TOWER, BLUE LED
   // Blue Light
   RUNG wire#powerrail
      I_Contact( "M_ZERO" )
      Not()
      wire#w1
      Contact( "M_0.5_SEC_2HZ" )
      wire#w2
      Coil( "SIGNAL_TWR_BLUE_LIGHT_Q" )
   END_RUNG
   RUNG wire#powerrail
      I_Contact( "M_ZERO" )
      Not()
   END_RUNG wire#w1
   RUNG wire#powerrail
      Contact( "M_ZERO" )
   END_RUNG wire#w2
   // the same network as SCL:
   "SIGNAL_TWR_BLUE_LIGHT_Q" := ((NOT (NOT "M_ZERO") OR NOT (NOT "M_ZERO")) AND "M_0.5_SEC_2HZ") OR "M_ZERO";
END_REGION

REGION Network 6: SIGNAL TOWER WHITE LIGHT OUTPUT / SIGNAL TOWER, BLUE LED
   // Blue Light
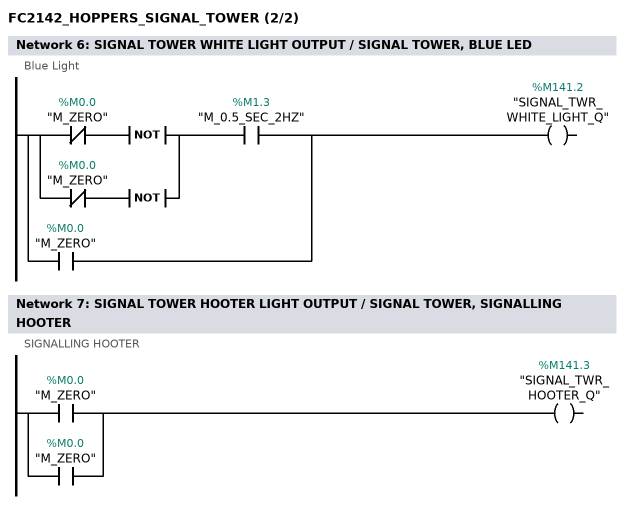
   RUNG wire#powerrail
      I_Contact( "M_ZERO" )
      Not()
      wire#w1
      Contact( "M_0.5_SEC_2HZ" )
      wire#w2
      Coil( "SIGNAL_TWR_WHITE_LIGHT_Q" )
   END_RUNG
   RUNG wire#powerrail
      I_Contact( "M_ZERO" )
      Not()
   END_RUNG wire#w1
   RUNG wire#powerrail
      Contact( "M_ZERO" )
   END_RUNG wire#w2
   // the same network as SCL:
   "SIGNAL_TWR_WHITE_LIGHT_Q" := ((NOT (NOT "M_ZERO") OR NOT (NOT "M_ZERO")) AND "M_0.5_SEC_2HZ") OR "M_ZERO";
END_REGION

REGION Network 7: SIGNAL TOWER HOOTER LIGHT OUTPUT / SIGNAL TOWER, SIGNALLING HOOTER
   // SIGNALLING HOOTER
   RUNG wire#powerrail
      Contact( "M_ZERO" )
      wire#w1
      Coil( "SIGNAL_TWR_HOOTER_Q" )
   END_RUNG
   RUNG wire#powerrail
      Contact( "M_ZERO" )
   END_RUNG wire#w1
   // the same network as SCL:
   "SIGNAL_TWR_HOOTER_Q" := "M_ZERO" OR "M_ZERO";
END_REGION
END_FUNCTION

FUNCTION_BLOCK "FB31_SPINDLE"   // FB31, LAD
{ S7_Optimized_Access := 'FALSE' }
AUTHOR : ETXETAR
VERSION : 1.0
// stored: AutoNumber false, IsIECCheckEnabled false, SetENOAutomatically false, UDAEnableTagReadback false
   VAR_INPUT
      OPTIONS_0 : Byte := 2#0000_0000;   // OPTIONS 0
      OPTIONS_1 : Byte := 2#0000_0000;   // OPTIONS 1
      SAFETY_BYPASS : Bool;   // MUST BE ALWAYS OFF, ACTIVATE ONLY FOR TEST
      OPTIMIZATION_BYPASS : Bool;   // MUST BE ALWAYS OFF, ACTIVATE ONLY FOR OPTIMIZATION TEST
      RPMS_REACHED : Bool;   // RPMS REACHED / N.O
      BELT_BROKEN : Bool;   // BELT BROKEN / N.C
      COOLING_SYS_IN_SERVICE : Bool;   // COOLING SYSTEM IN SERVICE
      MQL_HP_IN_SERVICE : Bool;   // MQL OR HP IN SERVICE
      TEMPERATURE_SENSOR : Word;   // TEMPERATURE SENSOR
      TEMPERATURE_SENSOR_PTC : Bool;   // TEMPERATURE SENSOR PTC
      VPM_READY : Bool;   // VOLTAGE PROTECTION MODULE READY
      ENABLE : Bool;   // ENABLE
      FEED_HOLD_COND : Bool;   // FEED HOLD CONDITION
      UNIT_SEQ_RUNNING : Bool;   // UNIT SEQUENCE RUNNING
      SAFE_ENABLED : Bool;   // SAFETY ENABLED
      TEST_STOP_INTERNAL_PULSES : Bool;   // TEST STOP INTERNAL PULSES
      FEED_OVERRIDE : Byte;   // FEED OVERRIDE
      SPINDLE_OVERRIDE : Byte;   // SPINDLE OVERRIDE
      HMI_SP_SELECTED : Bool;   // HMI SPINDLE SELECTED
      HMI_REQ_LINE : Bool;   // HMI REQUEST LINE
      CHANNEL_M3 : Bool;   // CHANNEL M3
      CHANNEL_M300 : Bool;   // CHANNEL M300
      M_VERIFY_CLAMP_F1 : Bool;   // M VERIFY CLAMPED FIXTURE 1
      M_VERIFY_CLAMP_F2 : Bool;   // M VERIFY CLAMPED FIXTURE 2
      SP_CLAMP : Bool;   // SPINDLE CLAMPING UNIT CLAMP
      SP_CLAMPED : Bool;   // SPINDLE CLAMPING UNIT CLAMPED
      SP_CLAMPED_WITH_TOOL : Bool;   // SPINDLE CLAMPING UNIT CLAMPED WITH TOOL
      HARDWARE_ENABLE : Bool;   // HARDWARE ENABLE
      TOOL_CHANGE_POS : Bool;   // TOOL CHANGE POSITION
      FIXTURE_1_PART_OK : Bool;   // FIXTURE 1 PART OK
      FIXTURE_2_PART_OK : Bool;   // FIXTURE 2 PART OK
      READ_POS : DWord;   // READ POSITION
      UNIT_ALARM : UInt;   // UNIT NUMBER MAX. NUMBER=10
      STATION_ALARM : UInt;   // STATION NUMBER MIN. NUMBER=0 MAX. NUMBER=4
      DESELECT_SPINDLE_STO : Bool;   // DESELECT SPINDLE STO
   END_VAR
   VAR_OUTPUT
      DELAYED_ENABLE : Bool;   // DELAYED ENABLE
      FEED_HOLD_CONDITIONS : Bool;   // FEED HOLD CONDITIONS
      FEED_HOLD_CONDITIONS_HMI : Bool;   // HMI FEED HOLD CONDITIONS
      SP_DESELECTED : Bool;   // SPINDLE DESELECTED
      SPEED_NOT_REACHED_ALARM : Bool;   // SPEED NOT REACHED ALARM
      BELT_BROKEN_ALARM : Bool;   // BELT BROKEN ALARM
      COOLING_ALARM : Bool;   // COOLING ALARM
      MQL_HP_ALARM : Bool;   // MQL HP ALARM
      HIGH_TEMP_ALARM : Bool;   // HIGH TEMPERATURE ALARM
      HIGH_TEMP_PTC_ALARM : Bool;   // HIGH TEMPERATURE PTC ALARM
      VPM_READY_ALARM : Bool;   // VPM READY ALARM
      HIGH_TEMP_PREALM : Bool;   // HIGH TEMPERATURE PREALARM
      SPINDLE_POS : Real;   // SPINDLE POSITION
      HMI_MOTION_EXECUTABILITY_LEFT : Bool;   // HMI MOTION EXECUTABILITY LEFT
      HMI_MOTION_EXECUTABILITY_RIGHT : Bool;   // HMI MOTION EXECUTABILITY RIGHT
      HMI_MOTION_END_POS_LEFT : Bool;   // HMI MOTION END POSITION LEFT
      HMI_MOTION_END_POS_RIGHT : Bool;   // HMI MOTION END POSITION RIGHT
   END_VAR
   VAR_IN_OUT
      SpindleDB : "LBP_typeAxisX";
   END_VAR
   VAR DB_SPECIFIC
      SP : "SPINDLE";
      SP_TEMPERATURE : Real;   // SPINDLE TEMPERATURE
      TEMP_MUL_VAL { S7_SetPoint := 'True'} : Real := 800.0;   // CONVERSION VALUE TO MUL THE INPUT
      TEMP_DIV_VAL { S7_SetPoint := 'True'} : Real := 16383.0;   // CONVERSION VALUE TO DIV THE MUL VALUE
      TEMP_SUB_VAL { S7_SetPoint := 'True'} : Real := 200.0;   // CONVERSION VALUE TO SUB TO THE SUB VALUE
      TEMP_PREALARM_VAL { S7_SetPoint := 'True'} : Real := 40.0;   // TEMPERATURE PREALARM VALUE
      TEMP_ALARM_VAL { S7_SetPoint := 'True'} : Real := 45.0;   // TEMPERATURE ALARM VALUE
      WARNING_GONE { S7_SetPoint := 'True'} : Bool;   // WARNING GONE
      TIMER_ENABLE_PULSE { S7_SetPoint := 'True'} : TOF_TIME;   // ENABLE PULSE TIMER
      TIMER_DELETE_DIST_TO_GO { S7_SetPoint := 'True'} : TON_TIME;   // DELETE DISTANCE TO GO TIMER
      TIMER_SPEED_NOT_REACHED { S7_SetPoint := 'True'} : TOF_TIME;   // SPEED NOT REACHED TIMER
      TIMER_BELT_BROKEN_ALARM { S7_SetPoint := 'True'} : TON_TIME;   // BELT BROKEN TIMER
      TIMER_MQL_HP_FAULT { S7_SetPoint := 'True'} : TON_TIME;   // MQL OR HP FAULT TIMER
      TIMER_COMMAND_JOG_PLUS { S7_SetPoint := 'True'} : TON_TIME;   // COMMAND JOG PLUS TIMER
   END_VAR
   VAR
      SAFETY_POSITIONS { S7_SetPoint := 'True'} : "FB33_SAFETY_POSITIONS";
   END_VAR
   VAR_TEMP
      INPUTS_MASK : Byte;   // INPUT MASK
      O_BYTE_0 : Struct   // OPTION BYTE 0
         MEASURING_SYSTEM_2 : Bool;   // MEASURING SYSTEM 2 OPTION / ALWAYS ON OR ALWAYS OFF
         BELT_BROKEN : Bool;   // BELT BROKEN OPTION
         COOLING : Bool;   // COOLING OPTION / ALWAYS ON OR ALWAYS OFF
         MQL_OR_HP : Bool;   // MQL OR HP OPTION / ALWAYS ON OR ALWAYS OFF
         ANALOG_TEMPERATURE_SENSOR : Bool;   // ANALOG TEMPERATURE SENSOR OPTION
         PTC_TEMP_SENSOR : Bool;   // PTC TEMPERATURE SENSOR OPTION
         TWIN_KESSLER_VPM_READY : Bool;   // TWIN KESSLER VPM READY OPTION
         MPP_SP_OVERRIDE : Bool;   // MPP SPINDLE OVERRIDE OPTION
      END_STRUCT;
      O_BYTE_1 : Struct   // OPTION BYTE 1
         SPARE_0 : Bool;   // SPARE OPTION / ALWAYS ON OR ALWAYS OFF
         SPARE_1 : Bool;   // SPARE OPTION
         SPARE_2 : Bool;   // SPARE OPTION / ALWAYS ON OR ALWAYS OFF
         SPARE_3 : Bool;   // SPARE OPTION / ALWAYS ON OR ALWAYS OFF
         SPARE_4 : Bool;   // SPARE OPTION
         SPARE_5 : Bool;   // SPARE OPTION
         SPARE_6 : Bool;   // SPARE OPTION
         SPARE_7 : Bool;   // SPARE OPTION
      END_STRUCT;
      TEMP_INPUT : DInt;   // TEMPERATURE INPUR SHIFTED
      TEMP_REAL : Real;   // TEMPERATURE IN REAL
      DB_NUMBER : DInt;   // DB NUMBER FOR ALARMS AND HELP DECODING
   END_VAR
   // TIMER_ENABLE_PULSE.PT := T#1s;
   // TIMER_DELETE_DIST_TO_GO.PT := T#20ms;
   // TIMER_SPEED_NOT_REACHED.PT := T#100ms;
   // TIMER_BELT_BROKEN_ALARM.PT := T#150ms;
   // TIMER_MQL_HP_FAULT.PT := T#50ms;
   // TIMER_COMMAND_JOG_PLUS.PT := T#100ms;
   VAR_TEMP   // added for the SCL form of the ladder/FBD networks
      _w1 : Bool;
      _w2 : Bool;
      _w3 : Bool;
      _w4 : Bool;
      _w5 : Bool;
      _w6 : Bool;
      _w7 : Bool;
      _w8 : Bool;
      _w9 : Bool;
      _w10 : Bool;
      _w11 : Bool;
      _w12 : Bool;
      _w13 : Bool;
      _w14 : Bool;
      _w15 : Bool;
   END_VAR
BEGIN

NETWORK
TITLE = READ INSTANCE DB
      L     DINO;
      +     10#800000;
      T     #DB_NUMBER;


REGION Network 2: OPTIONS
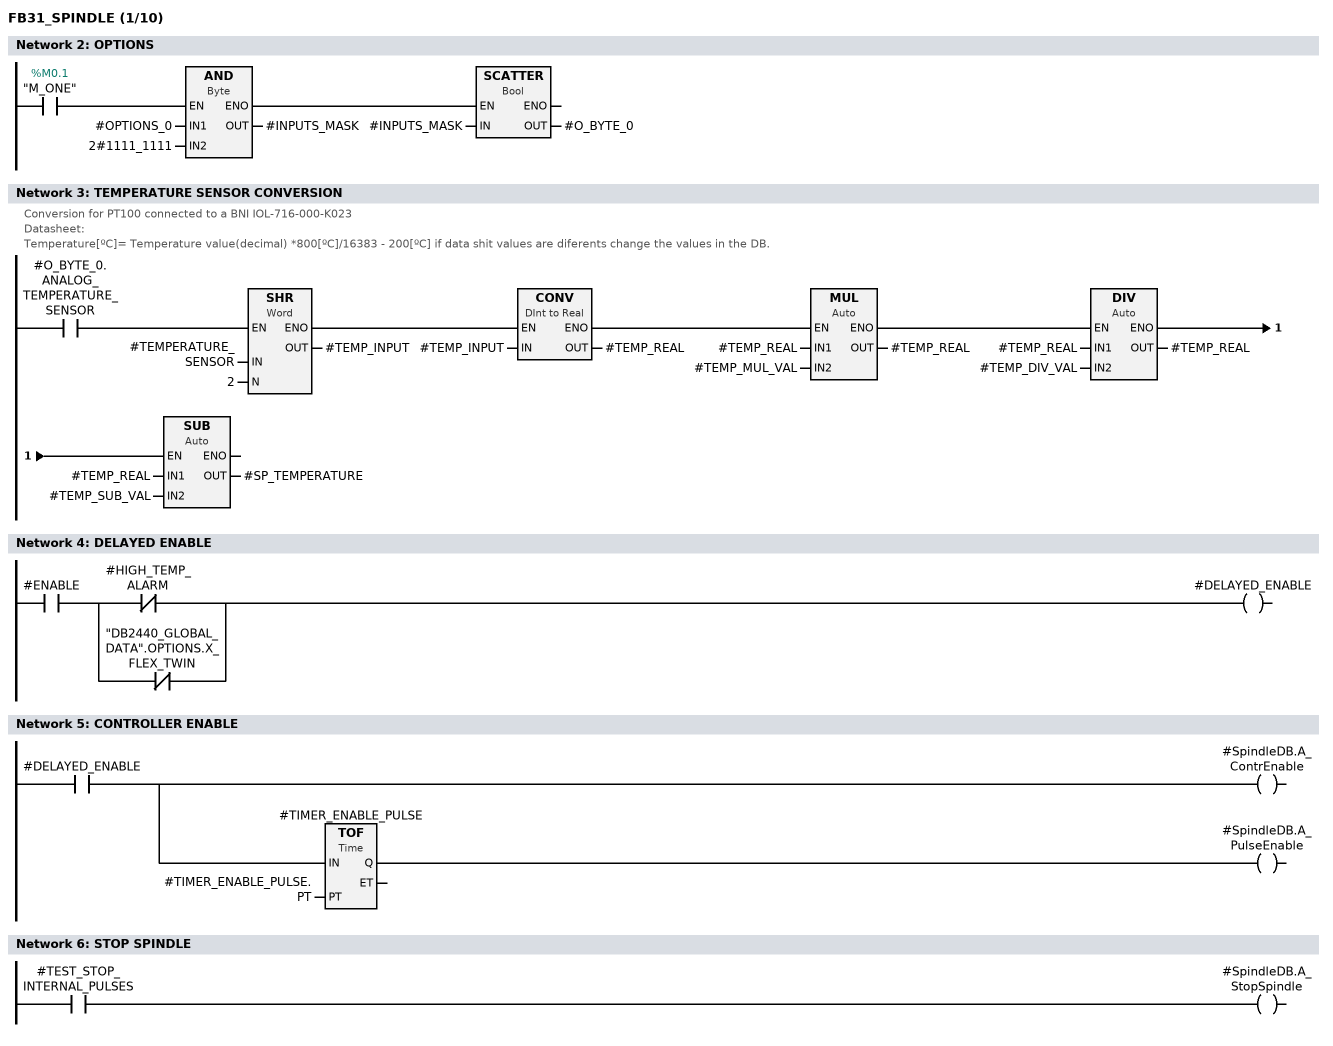
   RUNG wire#powerrail
      Contact( "M_ONE" )
      { S7_Templates := "SrcType := Byte"; S7_GenerateENO := "TRUE" } And(in1 := #OPTIONS_0, in2 := 2#1111_1111, out => #INPUTS_MASK)
      { S7_Templates := "[dest_type := Bool, src_type := Byte]" } SCATTER(IN := #INPUTS_MASK, OUT => #O_BYTE_0)
   END_RUNG
   // the same network as SCL:
   IF "M_ONE" THEN
       #INPUTS_MASK := #OPTIONS_0 AND 2#1111_1111;
       SCATTER(IN := #INPUTS_MASK, OUT => #O_BYTE_0);
   END_IF;
END_REGION

REGION Network 3: TEMPERATURE SENSOR CONVERSION
   // Conversion for PT100 connected to a BNI IOL-716-000-K023
   // 
   // Datasheet:
   // 
   //  Temperature[ºC]= Temperature value(decimal) *800[ºC]/16383 - 200[ºC] if data shit values are diferents change the values in the DB.
   RUNG wire#powerrail
      Contact( #O_BYTE_0.ANALOG_TEMPERATURE_SENSOR )
      { S7_Templates := "SrcType := Word" } Shr(in := #TEMPERATURE_SENSOR, n := 2, out => #TEMP_INPUT)
      { S7_Templates := "[SrcType := DInt, DestType := Real]" } Convert(in := #TEMP_INPUT, out => #TEMP_REAL)
      Mul(in1 := #TEMP_REAL, in2 := #TEMP_MUL_VAL, out => #TEMP_REAL)
      Div(in1 := #TEMP_REAL, in2 := #TEMP_DIV_VAL, out => #TEMP_REAL)
      Sub(in1 := #TEMP_REAL, in2 := #TEMP_SUB_VAL, out => #SP_TEMPERATURE)
   END_RUNG
   // the same network as SCL:
   IF #O_BYTE_0.ANALOG_TEMPERATURE_SENSOR THEN
       #TEMP_INPUT := SHR(IN := #TEMPERATURE_SENSOR, N := 2);
       #TEMP_REAL := DINT_TO_REAL(#TEMP_INPUT);
       #TEMP_REAL := #TEMP_REAL * #TEMP_MUL_VAL;
       #TEMP_REAL := #TEMP_REAL / #TEMP_DIV_VAL;
       #SP_TEMPERATURE := #TEMP_REAL - #TEMP_SUB_VAL;
   END_IF;
END_REGION

REGION Network 4: DELAYED ENABLE
   RUNG wire#powerrail
      Contact( #ENABLE )
      wire#w1
      I_Contact( #HIGH_TEMP_ALARM )
      wire#w2
      Coil( #DELAYED_ENABLE )
   END_RUNG
   RUNG wire#w1
      I_Contact( "DB2440_GLOBAL_DATA".OPTIONS.X_FLEX_TWIN )
   END_RUNG wire#w2
   // the same network as SCL:
   #DELAYED_ENABLE := #ENABLE AND (NOT #HIGH_TEMP_ALARM OR NOT "DB2440_GLOBAL_DATA".OPTIONS.X_FLEX_TWIN);
END_REGION

REGION Network 5: CONTROLLER ENABLE
   RUNG wire#powerrail
      Contact( #DELAYED_ENABLE )
      wire#w1
      Coil( #SpindleDB.A_ContrEnable )
   END_RUNG
   RUNG wire#w1
      { S7_Templates := "time_type := Time" } #TIMER_ENABLE_PULSE.TOF(pt := #TIMER_ENABLE_PULSE.PT, et =>)
      Coil( #SpindleDB.A_PulseEnable )
   END_RUNG
   // the same network as SCL:
   #SpindleDB.A_ContrEnable := #DELAYED_ENABLE;
   #TIMER_ENABLE_PULSE(IN := #DELAYED_ENABLE, PT := #TIMER_ENABLE_PULSE.PT);   // TOF
   #SpindleDB.A_PulseEnable := #TIMER_ENABLE_PULSE.Q;
END_REGION

REGION Network 6: STOP SPINDLE
   RUNG wire#powerrail
      Contact( #TEST_STOP_INTERNAL_PULSES )
      Coil( #SpindleDB.A_StopSpindle )
   END_RUNG
   // the same network as SCL:
   #SpindleDB.A_StopSpindle := #TEST_STOP_INTERNAL_PULSES;
END_REGION

REGION Network 7: DELETE DISTANCE TO GO / DELETE S VALUE
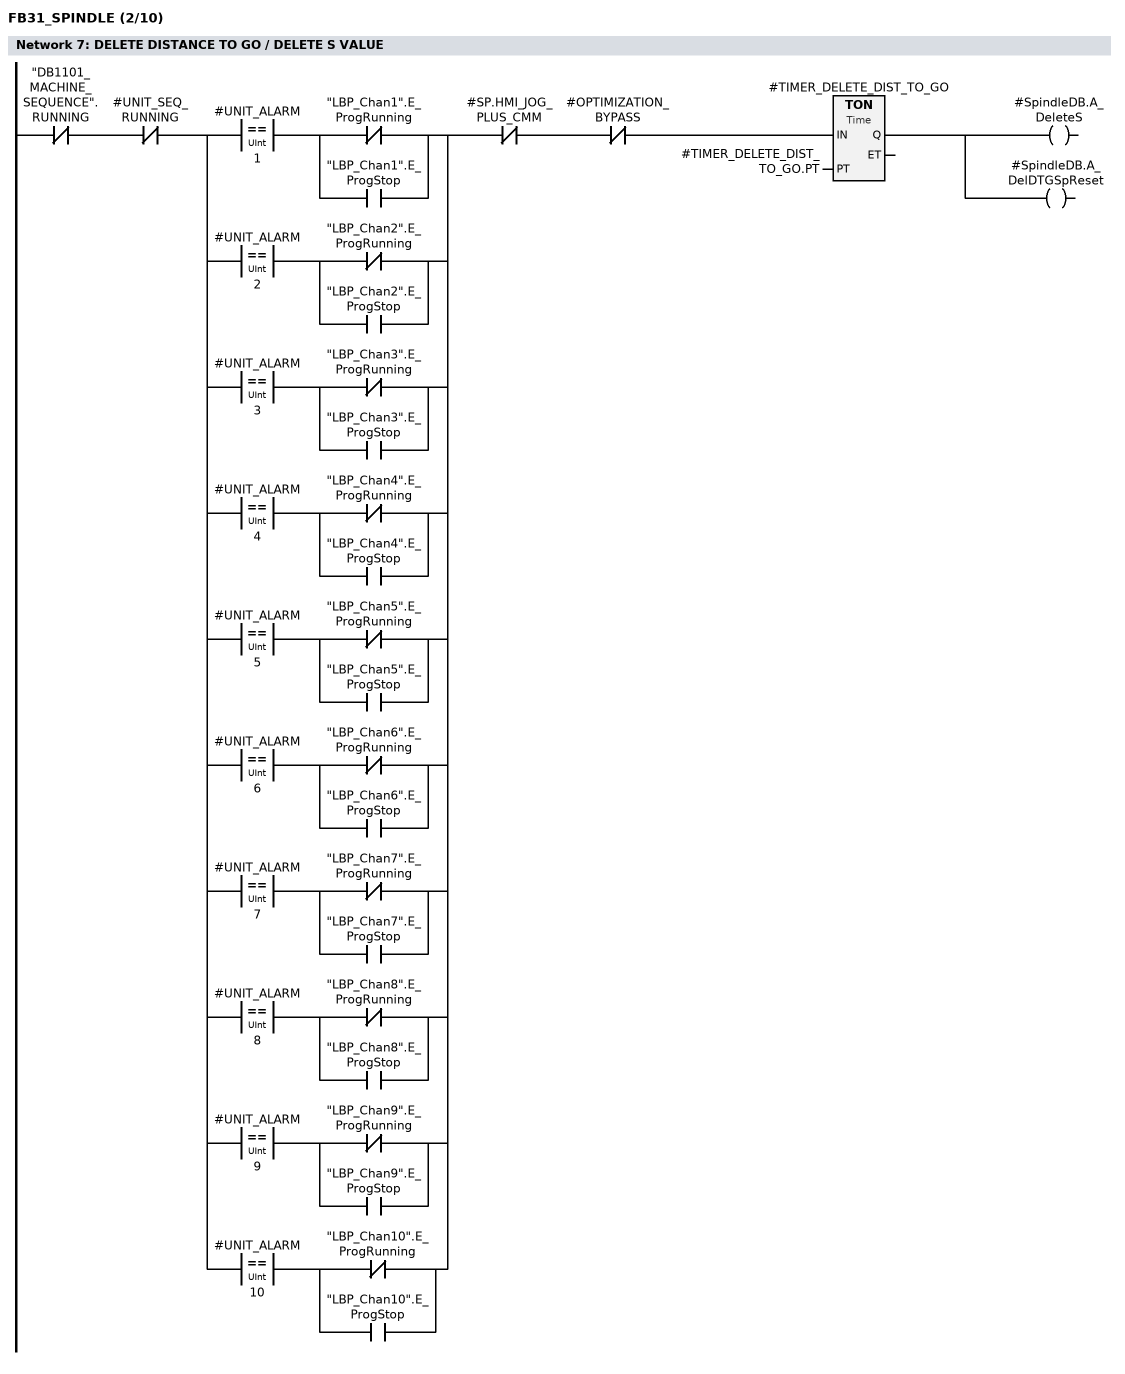
   RUNG wire#powerrail
      I_Contact( "DB1101_MACHINE_SEQUENCE".RUNNING )
      I_Contact( #UNIT_SEQ_RUNNING )
      wire#w1
      { S7_Templates := "SrcType := UInt" } EQ_Contact(in1 := #UNIT_ALARM, in2 := 1)
      wire#w2
      I_Contact( "LBP_Chan1".E_ProgRunning )
      wire#w3
      I_Contact( #SP.HMI_JOG_PLUS_CMM )
      I_Contact( #OPTIMIZATION_BYPASS )
      { S7_Templates := "time_type := Time" } #TIMER_DELETE_DIST_TO_GO.TON(pt := #TIMER_DELETE_DIST_TO_GO.PT, et =>)
      wire#w13
      Coil( #SpindleDB.A_DeleteS )
   END_RUNG
   RUNG wire#w2
      Contact( "LBP_Chan1".E_ProgStop )
   END_RUNG wire#w3
   RUNG wire#w1
      { S7_Templates := "SrcType := UInt" } EQ_Contact(in1 := #UNIT_ALARM, in2 := 2)
      wire#w4
      I_Contact( "LBP_Chan2".E_ProgRunning )
   END_RUNG wire#w3
   RUNG wire#w4
      Contact( "LBP_Chan2".E_ProgStop )
   END_RUNG wire#w3
   RUNG wire#w1
      { S7_Templates := "SrcType := UInt" } EQ_Contact(in1 := #UNIT_ALARM, in2 := 3)
      wire#w5
      I_Contact( "LBP_Chan3".E_ProgRunning )
   END_RUNG wire#w3
   RUNG wire#w5
      Contact( "LBP_Chan3".E_ProgStop )
   END_RUNG wire#w3
   RUNG wire#w1
      { S7_Templates := "SrcType := UInt" } EQ_Contact(in1 := #UNIT_ALARM, in2 := 4)
      wire#w6
      I_Contact( "LBP_Chan4".E_ProgRunning )
   END_RUNG wire#w3
   RUNG wire#w6
      Contact( "LBP_Chan4".E_ProgStop )
   END_RUNG wire#w3
   RUNG wire#w1
      { S7_Templates := "SrcType := UInt" } EQ_Contact(in1 := #UNIT_ALARM, in2 := 5)
      wire#w7
      I_Contact( "LBP_Chan5".E_ProgRunning )
   END_RUNG wire#w3
   RUNG wire#w7
      Contact( "LBP_Chan5".E_ProgStop )
   END_RUNG wire#w3
   RUNG wire#w1
      { S7_Templates := "SrcType := UInt" } EQ_Contact(in1 := #UNIT_ALARM, in2 := 6)
      wire#w8
      I_Contact( "LBP_Chan6".E_ProgRunning )
   END_RUNG wire#w3
   RUNG wire#w8
      Contact( "LBP_Chan6".E_ProgStop )
   END_RUNG wire#w3
   RUNG wire#w1
      { S7_Templates := "SrcType := UInt" } EQ_Contact(in1 := #UNIT_ALARM, in2 := 7)
      wire#w9
      I_Contact( "LBP_Chan7".E_ProgRunning )
   END_RUNG wire#w3
   RUNG wire#w9
      Contact( "LBP_Chan7".E_ProgStop )
   END_RUNG wire#w3
   RUNG wire#w1
      { S7_Templates := "SrcType := UInt" } EQ_Contact(in1 := #UNIT_ALARM, in2 := 8)
      wire#w10
      I_Contact( "LBP_Chan8".E_ProgRunning )
   END_RUNG wire#w3
   RUNG wire#w10
      Contact( "LBP_Chan8".E_ProgStop )
   END_RUNG wire#w3
   RUNG wire#w1
      { S7_Templates := "SrcType := UInt" } EQ_Contact(in1 := #UNIT_ALARM, in2 := 9)
      wire#w11
      I_Contact( "LBP_Chan9".E_ProgRunning )
   END_RUNG wire#w3
   RUNG wire#w11
      Contact( "LBP_Chan9".E_ProgStop )
   END_RUNG wire#w3
   RUNG wire#w1
      { S7_Templates := "SrcType := UInt" } EQ_Contact(in1 := #UNIT_ALARM, in2 := 10)
      wire#w12
      I_Contact( "LBP_Chan10".E_ProgRunning )
   END_RUNG wire#w3
   RUNG wire#w12
      Contact( "LBP_Chan10".E_ProgStop )
   END_RUNG wire#w3
   RUNG wire#w13
      Coil( #SpindleDB.A_DelDTGSpReset )
   END_RUNG
   // the same network as SCL:
   #TIMER_DELETE_DIST_TO_GO(IN := NOT "DB1101_MACHINE_SEQUENCE".RUNNING AND NOT #UNIT_SEQ_RUNNING AND (((#UNIT_ALARM = 1) AND (NOT "LBP_Chan1".E_ProgRunning OR "LBP_Chan1".E_ProgStop)) OR ((#UNIT_ALARM = 2) AND (NOT "LBP_Chan2".E_ProgRunning OR "LBP_Chan2".E_ProgStop)) OR ((#UNIT_ALARM = 3) AND (NOT "LBP_Chan3".E_ProgRunning OR "LBP_Chan3".E_ProgStop)) OR ((#UNIT_ALARM = 4) AND (NOT "LBP_Chan4".E_ProgRunning OR "LBP_Chan4".E_ProgStop)) OR ((#UNIT_ALARM = 5) AND (NOT "LBP_Chan5".E_ProgRunning OR "LBP_Chan5".E_ProgStop)) OR ((#UNIT_ALARM = 6) AND (NOT "LBP_Chan6".E_ProgRunning OR "LBP_Chan6".E_ProgStop)) OR ((#UNIT_ALARM = 7) AND (NOT "LBP_Chan7".E_ProgRunning OR "LBP_Chan7".E_ProgStop)) OR ((#UNIT_ALARM = 8) AND (NOT "LBP_Chan8".E_ProgRunning OR "LBP_Chan8".E_ProgStop)) OR ((#UNIT_ALARM = 9) AND (NOT "LBP_Chan9".E_ProgRunning OR "LBP_Chan9".E_ProgStop)) OR ((#UNIT_ALARM = 10) AND (NOT "LBP_Chan10".E_ProgRunning OR "LBP_Chan10".E_ProgStop))) AND NOT #SP.HMI_JOG_PLUS_CMM AND NOT #OPTIMIZATION_BYPASS,   // TON
                           PT := #TIMER_DELETE_DIST_TO_GO.PT);
   #SpindleDB.A_DeleteS := #TIMER_DELETE_DIST_TO_GO.Q;
   #SpindleDB.A_DelDTGSpReset := #TIMER_DELETE_DIST_TO_GO.Q;
END_REGION

REGION Network 8: POSITION MEASURING SYTEM
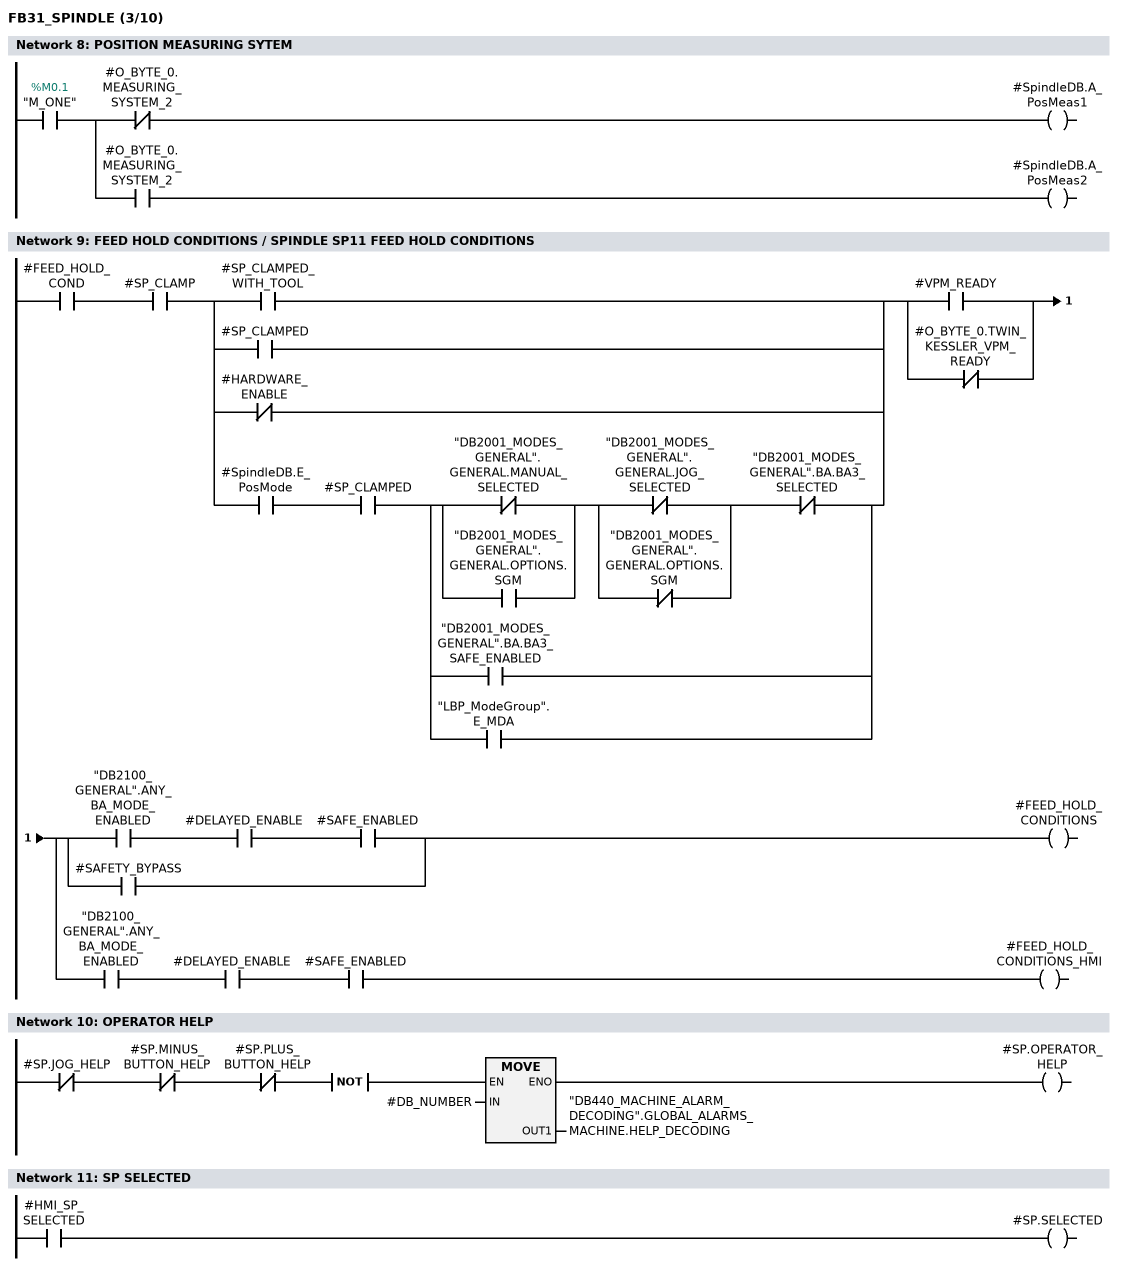
   RUNG wire#powerrail
      Contact( "M_ONE" )
      wire#w1
      I_Contact( #O_BYTE_0.MEASURING_SYSTEM_2 )
      Coil( #SpindleDB.A_PosMeas1 )
   END_RUNG
   RUNG wire#w1
      Contact( #O_BYTE_0.MEASURING_SYSTEM_2 )
      Coil( #SpindleDB.A_PosMeas2 )
   END_RUNG
   // the same network as SCL:
   #SpindleDB.A_PosMeas1 := "M_ONE" AND NOT #O_BYTE_0.MEASURING_SYSTEM_2;
   #SpindleDB.A_PosMeas2 := "M_ONE" AND #O_BYTE_0.MEASURING_SYSTEM_2;
END_REGION

REGION Network 9: FEED HOLD CONDITIONS / SPINDLE SP11 FEED HOLD CONDITIONS
   RUNG wire#powerrail
      Contact( #FEED_HOLD_COND )
      Contact( #SP_CLAMP )
      wire#w1
      Contact( #SP_CLAMPED_WITH_TOOL )
      wire#w2
      Contact( #VPM_READY )
      wire#w6
      Contact( "DB2100_GENERAL".ANY_BA_MODE_ENABLED )
      Contact( #DELAYED_ENABLE )
      Contact( #SAFE_ENABLED )
      wire#w7
      Coil( #FEED_HOLD_CONDITIONS )
   END_RUNG
   RUNG wire#w1
      Contact( #SP_CLAMPED )
   END_RUNG wire#w2
   RUNG wire#w1
      I_Contact( #HARDWARE_ENABLE )
   END_RUNG wire#w2
   RUNG wire#w1
      Contact( #SpindleDB.E_PosMode )
      Contact( #SP_CLAMPED )
      wire#w3
      I_Contact( "DB2001_MODES_GENERAL".GENERAL.MANUAL_SELECTED )
      wire#w4
      I_Contact( "DB2001_MODES_GENERAL".GENERAL.JOG_SELECTED )
      wire#w5
      I_Contact( "DB2001_MODES_GENERAL".BA.BA3_SELECTED )
   END_RUNG wire#w2
   RUNG wire#w3
      Contact( "DB2001_MODES_GENERAL".GENERAL.OPTIONS.SGM )
   END_RUNG wire#w4
   RUNG wire#w4
      I_Contact( "DB2001_MODES_GENERAL".GENERAL.OPTIONS.SGM )
   END_RUNG wire#w5
   RUNG wire#w3
      Contact( "DB2001_MODES_GENERAL".BA.BA3_SAFE_ENABLED )
   END_RUNG wire#w2
   RUNG wire#w3
      Contact( "LBP_ModeGroup".E_MDA )
   END_RUNG wire#w2
   RUNG wire#w2
      I_Contact( #O_BYTE_0.TWIN_KESSLER_VPM_READY )
   END_RUNG wire#w6
   RUNG wire#w6
      Contact( #SAFETY_BYPASS )
   END_RUNG wire#w7
   RUNG wire#w6
      Contact( "DB2100_GENERAL".ANY_BA_MODE_ENABLED )
      Contact( #DELAYED_ENABLE )
      Contact( #SAFE_ENABLED )
      Coil( #FEED_HOLD_CONDITIONS_HMI )
   END_RUNG
   // the same network as SCL:
   #_w1 := #FEED_HOLD_COND AND #SP_CLAMP AND (#SP_CLAMPED_WITH_TOOL OR #SP_CLAMPED OR NOT #HARDWARE_ENABLE OR (#SpindleDB.E_PosMode AND #SP_CLAMPED AND (((NOT "DB2001_MODES_GENERAL".GENERAL.MANUAL_SELECTED OR "DB2001_MODES_GENERAL".GENERAL.OPTIONS.SGM) AND (NOT "DB2001_MODES_GENERAL".GENERAL.JOG_SELECTED OR NOT "DB2001_MODES_GENERAL".GENERAL.OPTIONS.SGM) AND NOT "DB2001_MODES_GENERAL".BA.BA3_SELECTED) OR "DB2001_MODES_GENERAL".BA.BA3_SAFE_ENABLED OR "LBP_ModeGroup".E_MDA))) AND (#VPM_READY OR NOT #O_BYTE_0.TWIN_KESSLER_VPM_READY);
   #FEED_HOLD_CONDITIONS := #_w1 AND (("DB2100_GENERAL".ANY_BA_MODE_ENABLED AND #DELAYED_ENABLE AND #SAFE_ENABLED) OR #SAFETY_BYPASS);
   #FEED_HOLD_CONDITIONS_HMI := #_w1 AND "DB2100_GENERAL".ANY_BA_MODE_ENABLED AND #DELAYED_ENABLE AND #SAFE_ENABLED;
END_REGION

REGION Network 10: OPERATOR HELP
   RUNG wire#powerrail
      I_Contact( #SP.JOG_HELP )
      I_Contact( #SP.MINUS_BUTTON_HELP )
      I_Contact( #SP.PLUS_BUTTON_HELP )
      Not()
      { S7_GenerateENO := "TRUE" } Move(in := #DB_NUMBER, out1 => "DB440_MACHINE_ALARM_DECODING".GLOBAL_ALARMS_MACHINE.HELP_DECODING)
      Coil( #SP.OPERATOR_HELP )
   END_RUNG
   // the same network as SCL:
   // ENO of a box is taken as its EN; it also drops when the box reports an error
   #_w1 := NOT (NOT #SP.JOG_HELP AND NOT #SP.MINUS_BUTTON_HELP AND NOT #SP.PLUS_BUTTON_HELP);
   IF #_w1 THEN "DB440_MACHINE_ALARM_DECODING".GLOBAL_ALARMS_MACHINE.HELP_DECODING := #DB_NUMBER; END_IF;
   #SP.OPERATOR_HELP := #_w1;
END_REGION

REGION Network 11: SP SELECTED
   RUNG wire#powerrail
      Contact( #HMI_SP_SELECTED )
      Coil( #SP.SELECTED )
   END_RUNG
   // the same network as SCL:
   #SP.SELECTED := #HMI_SP_SELECTED;
END_REGION

REGION Network 12: SP DESELECTED
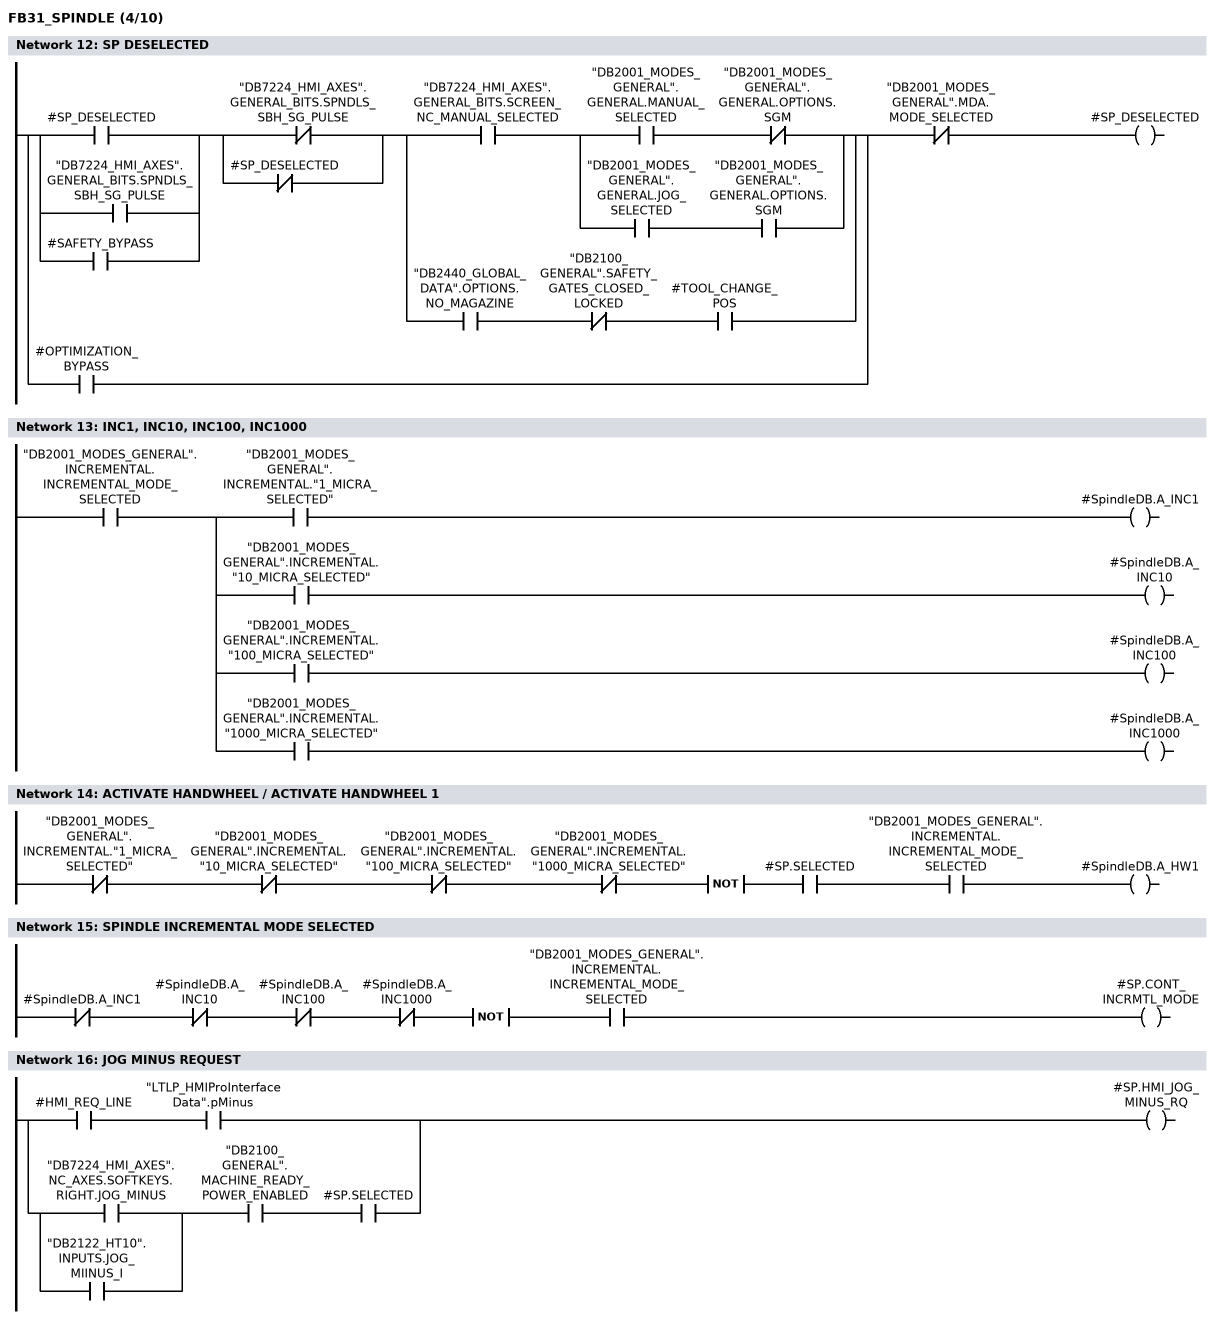
   RUNG wire#powerrail
      Contact( #SP_DESELECTED )
      wire#w1
      I_Contact( "DB7224_HMI_AXES".GENERAL_BITS.SPNDLS_SBH_SG_PULSE )
      wire#w2
      Contact( "DB7224_HMI_AXES".GENERAL_BITS.SCREEN_NC_MANUAL_SELECTED )
      wire#w3
      Contact( "DB2001_MODES_GENERAL".GENERAL.MANUAL_SELECTED )
      I_Contact( "DB2001_MODES_GENERAL".GENERAL.OPTIONS.SGM )
      wire#w4
      I_Contact( "DB2001_MODES_GENERAL".MDA.MODE_SELECTED )
      Coil( #SP_DESELECTED )
   END_RUNG
   RUNG wire#powerrail
      Contact( "DB7224_HMI_AXES".GENERAL_BITS.SPNDLS_SBH_SG_PULSE )
   END_RUNG wire#w1
   RUNG wire#powerrail
      Contact( #SAFETY_BYPASS )
   END_RUNG wire#w1
   RUNG wire#w1
      I_Contact( #SP_DESELECTED )
   END_RUNG wire#w2
   RUNG wire#w3
      Contact( "DB2001_MODES_GENERAL".GENERAL.JOG_SELECTED )
      Contact( "DB2001_MODES_GENERAL".GENERAL.OPTIONS.SGM )
   END_RUNG wire#w4
   RUNG wire#w2
      Contact( "DB2440_GLOBAL_DATA".OPTIONS.NO_MAGAZINE )
      I_Contact( "DB2100_GENERAL".SAFETY_GATES_CLOSED_LOCKED )
      Contact( #TOOL_CHANGE_POS )
   END_RUNG wire#w4
   RUNG wire#powerrail
      Contact( #OPTIMIZATION_BYPASS )
   END_RUNG wire#w4
   // the same network as SCL:
   #SP_DESELECTED := (((#SP_DESELECTED OR "DB7224_HMI_AXES".GENERAL_BITS.SPNDLS_SBH_SG_PULSE OR #SAFETY_BYPASS) AND (NOT "DB7224_HMI_AXES".GENERAL_BITS.SPNDLS_SBH_SG_PULSE OR NOT #SP_DESELECTED) AND (("DB7224_HMI_AXES".GENERAL_BITS.SCREEN_NC_MANUAL_SELECTED AND (("DB2001_MODES_GENERAL".GENERAL.MANUAL_SELECTED AND NOT "DB2001_MODES_GENERAL".GENERAL.OPTIONS.SGM) OR ("DB2001_MODES_GENERAL".GENERAL.JOG_SELECTED AND "DB2001_MODES_GENERAL".GENERAL.OPTIONS.SGM))) OR ("DB2440_GLOBAL_DATA".OPTIONS.NO_MAGAZINE AND NOT "DB2100_GENERAL".SAFETY_GATES_CLOSED_LOCKED AND #TOOL_CHANGE_POS))) OR #OPTIMIZATION_BYPASS) AND NOT "DB2001_MODES_GENERAL".MDA.MODE_SELECTED;
END_REGION

REGION Network 13: INC1, INC10, INC100, INC1000
   RUNG wire#powerrail
      Contact( "DB2001_MODES_GENERAL".INCREMENTAL.INCREMENTAL_MODE_SELECTED )
      wire#w1
      Contact( "DB2001_MODES_GENERAL".INCREMENTAL."1_MICRA_SELECTED" )
      Coil( #SpindleDB.A_INC1 )
   END_RUNG
   RUNG wire#w1
      Contact( "DB2001_MODES_GENERAL".INCREMENTAL."10_MICRA_SELECTED" )
      Coil( #SpindleDB.A_INC10 )
   END_RUNG
   RUNG wire#w1
      Contact( "DB2001_MODES_GENERAL".INCREMENTAL."100_MICRA_SELECTED" )
      Coil( #SpindleDB.A_INC100 )
   END_RUNG
   RUNG wire#w1
      Contact( "DB2001_MODES_GENERAL".INCREMENTAL."1000_MICRA_SELECTED" )
      Coil( #SpindleDB.A_INC1000 )
   END_RUNG
   // the same network as SCL:
   #SpindleDB.A_INC1 := "DB2001_MODES_GENERAL".INCREMENTAL.INCREMENTAL_MODE_SELECTED AND "DB2001_MODES_GENERAL".INCREMENTAL."1_MICRA_SELECTED";
   #SpindleDB.A_INC10 := "DB2001_MODES_GENERAL".INCREMENTAL.INCREMENTAL_MODE_SELECTED AND "DB2001_MODES_GENERAL".INCREMENTAL."10_MICRA_SELECTED";
   #SpindleDB.A_INC100 := "DB2001_MODES_GENERAL".INCREMENTAL.INCREMENTAL_MODE_SELECTED AND "DB2001_MODES_GENERAL".INCREMENTAL."100_MICRA_SELECTED";
   #SpindleDB.A_INC1000 := "DB2001_MODES_GENERAL".INCREMENTAL.INCREMENTAL_MODE_SELECTED AND "DB2001_MODES_GENERAL".INCREMENTAL."1000_MICRA_SELECTED";
END_REGION

REGION Network 14: ACTIVATE HANDWHEEL / ACTIVATE HANDWHEEL 1
   RUNG wire#powerrail
      I_Contact( "DB2001_MODES_GENERAL".INCREMENTAL."1_MICRA_SELECTED" )
      I_Contact( "DB2001_MODES_GENERAL".INCREMENTAL."10_MICRA_SELECTED" )
      I_Contact( "DB2001_MODES_GENERAL".INCREMENTAL."100_MICRA_SELECTED" )
      I_Contact( "DB2001_MODES_GENERAL".INCREMENTAL."1000_MICRA_SELECTED" )
      Not()
      Contact( #SP.SELECTED )
      Contact( "DB2001_MODES_GENERAL".INCREMENTAL.INCREMENTAL_MODE_SELECTED )
      Coil( #SpindleDB.A_HW1 )
   END_RUNG
   // the same network as SCL:
   #SpindleDB.A_HW1 := NOT (NOT "DB2001_MODES_GENERAL".INCREMENTAL."1_MICRA_SELECTED" AND NOT "DB2001_MODES_GENERAL".INCREMENTAL."10_MICRA_SELECTED" AND NOT "DB2001_MODES_GENERAL".INCREMENTAL."100_MICRA_SELECTED" AND NOT "DB2001_MODES_GENERAL".INCREMENTAL."1000_MICRA_SELECTED") AND #SP.SELECTED AND "DB2001_MODES_GENERAL".INCREMENTAL.INCREMENTAL_MODE_SELECTED;
END_REGION

REGION Network 15: SPINDLE INCREMENTAL MODE SELECTED
   RUNG wire#powerrail
      I_Contact( #SpindleDB.A_INC1 )
      I_Contact( #SpindleDB.A_INC10 )
      I_Contact( #SpindleDB.A_INC100 )
      I_Contact( #SpindleDB.A_INC1000 )
      Not()
      Contact( "DB2001_MODES_GENERAL".INCREMENTAL.INCREMENTAL_MODE_SELECTED )
      Coil( #SP.CONT_INCRMTL_MODE )
   END_RUNG
   // the same network as SCL:
   #SP.CONT_INCRMTL_MODE := NOT (NOT #SpindleDB.A_INC1 AND NOT #SpindleDB.A_INC10 AND NOT #SpindleDB.A_INC100 AND NOT #SpindleDB.A_INC1000) AND "DB2001_MODES_GENERAL".INCREMENTAL.INCREMENTAL_MODE_SELECTED;
END_REGION

REGION Network 16: JOG MINUS REQUEST
   RUNG wire#powerrail
      Contact( #HMI_REQ_LINE )
      Contact( "LTLP_HMIProInterfaceData".pMinus )
      wire#w1
      Coil( #SP.HMI_JOG_MINUS_RQ )
   END_RUNG
   RUNG wire#powerrail
      Contact( "DB7224_HMI_AXES".NC_AXES.SOFTKEYS.RIGHT.JOG_MINUS )
      wire#w2
      Contact( "DB2100_GENERAL".MACHINE_READY_POWER_ENABLED )
      Contact( #SP.SELECTED )
   END_RUNG wire#w1
   RUNG wire#powerrail
      Contact( "DB2122_HT10".INPUTS.JOG_MIINUS_I )
   END_RUNG wire#w2
   // the same network as SCL:
   #SP.HMI_JOG_MINUS_RQ := (#HMI_REQ_LINE AND "LTLP_HMIProInterfaceData".pMinus) OR (("DB7224_HMI_AXES".NC_AXES.SOFTKEYS.RIGHT.JOG_MINUS OR "DB2122_HT10".INPUTS.JOG_MIINUS_I) AND "DB2100_GENERAL".MACHINE_READY_POWER_ENABLED AND #SP.SELECTED);
END_REGION

